REGION Network 51: TOUT Error TR
   RUNG wire#powerrail
      "FC911_CNT_Tiempo_UHS"(Temporizar := wire#w1, Valor_Tiempo := #V_TOut_TR, Base_tiempo_ms := 1, Valor_Actual := #TOUT_Movimiento_transfer, Tiempo_OK => #Tout_movimiento_transfer_q)
   END_RUNG
   RUNG wire#powerrail
      Contact( "DB1_SalidasExterioresDeMesa".Mesa[#Mesa].Ir_Pos_E2E4 )
      I_Contact( #PosTR_E2 )
   END_RUNG wire#w1
   RUNG wire#powerrail
      Contact( "DB1_SalidasExterioresDeMesa".Mesa[#Mesa].Ir_Pos_E1E3 )
      I_Contact( #PosTR_E1 )
   END_RUNG wire#w1
   // the same network as SCL:
   "FC911_CNT_Tiempo_UHS"(Temporizar := ("DB1_SalidasExterioresDeMesa".Mesa[#Mesa].Ir_Pos_E2E4 AND NOT #PosTR_E2) OR ("DB1_SalidasExterioresDeMesa".Mesa[#Mesa].Ir_Pos_E1E3 AND NOT #PosTR_E1),
                          Valor_Tiempo := #V_TOut_TR,
                          Base_tiempo_ms := 1,
                          Valor_Actual := #TOUT_Movimiento_transfer,
                          Tiempo_OK => #Tout_movimiento_transfer_q);
END_REGION

REGION Network 52: ERROR SUBIDA TR
   RUNG wire#powerrail
      Contact( #EstadoZona.Rearme_CBx )
      S_RS(operand := #EstadoVI.Err_TOut_Subida, s1 := wire#w1)
      S_Coil( #EstadoVI.Error_Mx )
   END_RUNG
   RUNG wire#powerrail
      Contact( #Tout_movimiento_transfer_q )
      Contact( "DB1_SalidasExterioresDeMesa".Mesa[#Mesa].Ir_Pos_E2E4 )
   END_RUNG wire#w1
   // the same network as SCL:
   IF #EstadoZona.Rearme_CBx THEN
       #EstadoVI.Err_TOut_Subida := FALSE;   // RS flip-flop
   END_IF;
   IF #Tout_movimiento_transfer_q AND "DB1_SalidasExterioresDeMesa".Mesa[#Mesa].Ir_Pos_E2E4 THEN
       #EstadoVI.Err_TOut_Subida := TRUE;
   END_IF;
   IF #EstadoVI.Err_TOut_Subida THEN #EstadoVI.Error_Mx := TRUE; END_IF;
END_REGION

REGION Network 53: ERROR BAJADA TR
   RUNG wire#powerrail
      Contact( #EstadoZona.Rearme_CBx )
      S_RS(operand := #EstadoVI.Err_TOut_Bajada, s1 := wire#w1)
      S_Coil( #EstadoVI.Error_Mx )
   END_RUNG
   RUNG wire#powerrail
      Contact( #Tout_movimiento_transfer_q )
      Contact( "DB1_SalidasExterioresDeMesa".Mesa[#Mesa].Ir_Pos_E1E3 )
   END_RUNG wire#w1
   // the same network as SCL:
   IF #EstadoZona.Rearme_CBx THEN
       #EstadoVI.Err_TOut_Bajada := FALSE;   // RS flip-flop
   END_IF;
   IF #Tout_movimiento_transfer_q AND "DB1_SalidasExterioresDeMesa".Mesa[#Mesa].Ir_Pos_E1E3 THEN
       #EstadoVI.Err_TOut_Bajada := TRUE;
   END_IF;
   IF #EstadoVI.Err_TOut_Bajada THEN #EstadoVI.Error_Mx := TRUE; END_IF;
END_REGION

REGION Network 54: TMP Error en Avance Tx
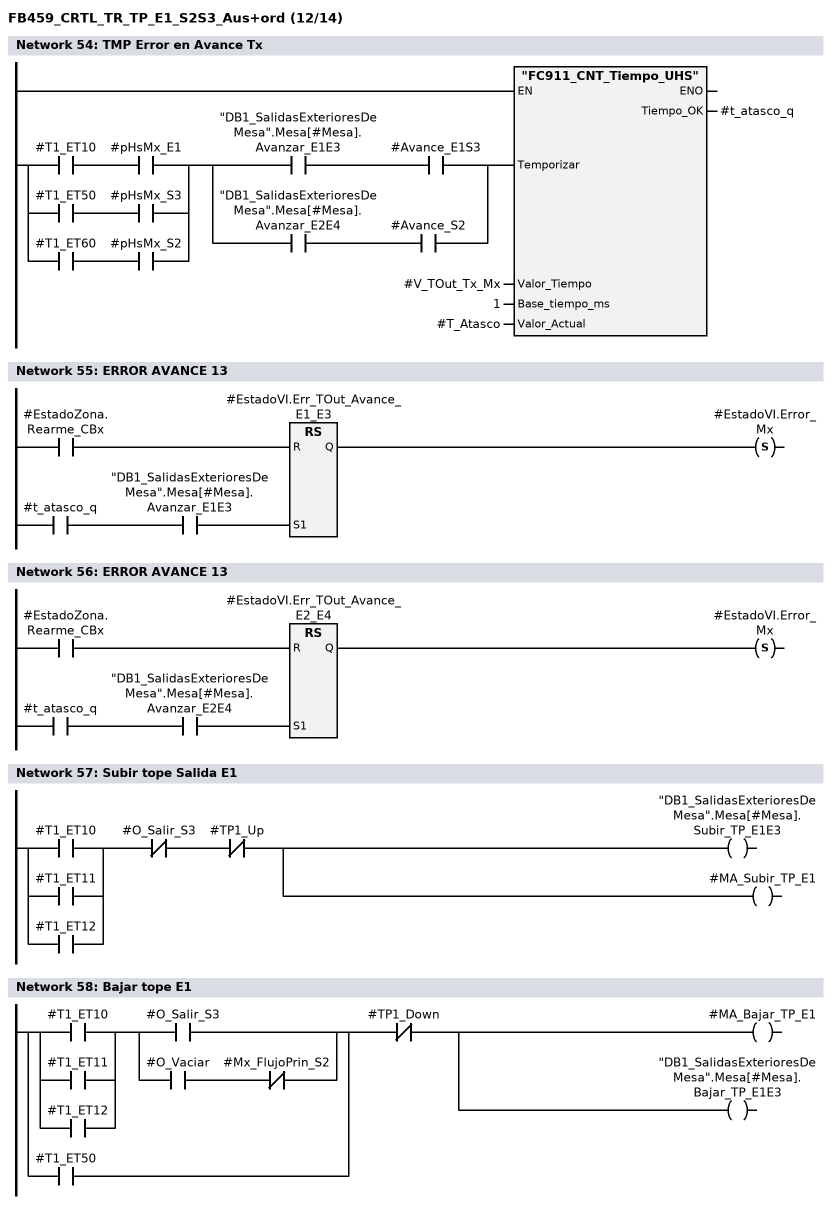
   RUNG wire#powerrail
      "FC911_CNT_Tiempo_UHS"(Temporizar := wire#w2, Valor_Tiempo := #V_TOut_Tx_Mx, Base_tiempo_ms := 1, Valor_Actual := #T_Atasco, Tiempo_OK => #t_atasco_q)
   END_RUNG
   RUNG wire#powerrail
      Contact( #T1_ET10 )
      Contact( #pHsMx_E1 )
      wire#w1
      Contact( "DB1_SalidasExterioresDeMesa".Mesa[#Mesa].Avanzar_E1E3 )
      Contact( #Avance_E1S3 )
   END_RUNG wire#w2
   RUNG wire#powerrail
      Contact( #T1_ET50 )
      Contact( #pHsMx_S3 )
   END_RUNG wire#w1
   RUNG wire#powerrail
      Contact( #T1_ET60 )
      Contact( #pHsMx_S2 )
   END_RUNG wire#w1
   RUNG wire#w1
      Contact( "DB1_SalidasExterioresDeMesa".Mesa[#Mesa].Avanzar_E2E4 )
      Contact( #Avance_S2 )
   END_RUNG wire#w2
   // the same network as SCL:
   "FC911_CNT_Tiempo_UHS"(Temporizar := ((#T1_ET10 AND #pHsMx_E1) OR (#T1_ET50 AND #pHsMx_S3) OR (#T1_ET60 AND #pHsMx_S2)) AND (("DB1_SalidasExterioresDeMesa".Mesa[#Mesa].Avanzar_E1E3 AND #Avance_E1S3) OR ("DB1_SalidasExterioresDeMesa".Mesa[#Mesa].Avanzar_E2E4 AND #Avance_S2)),
                          Valor_Tiempo := #V_TOut_Tx_Mx,
                          Base_tiempo_ms := 1,
                          Valor_Actual := #T_Atasco,
                          Tiempo_OK => #t_atasco_q);
END_REGION

REGION Network 55: ERROR AVANCE 13
   RUNG wire#powerrail
      Contact( #EstadoZona.Rearme_CBx )
      S_RS(operand := #EstadoVI.Err_TOut_Avance_E1_E3, s1 := wire#w1)
      S_Coil( #EstadoVI.Error_Mx )
   END_RUNG
   RUNG wire#powerrail
      Contact( #t_atasco_q )
      Contact( "DB1_SalidasExterioresDeMesa".Mesa[#Mesa].Avanzar_E1E3 )
   END_RUNG wire#w1
   // the same network as SCL:
   IF #EstadoZona.Rearme_CBx THEN
       #EstadoVI.Err_TOut_Avance_E1_E3 := FALSE;   // RS flip-flop
   END_IF;
   IF #t_atasco_q AND "DB1_SalidasExterioresDeMesa".Mesa[#Mesa].Avanzar_E1E3 THEN
       #EstadoVI.Err_TOut_Avance_E1_E3 := TRUE;
   END_IF;
   IF #EstadoVI.Err_TOut_Avance_E1_E3 THEN #EstadoVI.Error_Mx := TRUE; END_IF;
END_REGION

REGION Network 56: ERROR AVANCE 13
   RUNG wire#powerrail
      Contact( #EstadoZona.Rearme_CBx )
      S_RS(operand := #EstadoVI.Err_TOut_Avance_E2_E4, s1 := wire#w1)
      S_Coil( #EstadoVI.Error_Mx )
   END_RUNG
   RUNG wire#powerrail
      Contact( #t_atasco_q )
      Contact( "DB1_SalidasExterioresDeMesa".Mesa[#Mesa].Avanzar_E2E4 )
   END_RUNG wire#w1
   // the same network as SCL:
   IF #EstadoZona.Rearme_CBx THEN
       #EstadoVI.Err_TOut_Avance_E2_E4 := FALSE;   // RS flip-flop
   END_IF;
   IF #t_atasco_q AND "DB1_SalidasExterioresDeMesa".Mesa[#Mesa].Avanzar_E2E4 THEN
       #EstadoVI.Err_TOut_Avance_E2_E4 := TRUE;
   END_IF;
   IF #EstadoVI.Err_TOut_Avance_E2_E4 THEN #EstadoVI.Error_Mx := TRUE; END_IF;
END_REGION

REGION Network 57: Subir tope Salida E1
   RUNG wire#powerrail
      Contact( #T1_ET10 )
      wire#w1
      I_Contact( #O_Salir_S3 )
      I_Contact( #TP1_Up )
      wire#w2
      Coil( "DB1_SalidasExterioresDeMesa".Mesa[#Mesa].Subir_TP_E1E3 )
   END_RUNG
   RUNG wire#powerrail
      Contact( #T1_ET11 )
   END_RUNG wire#w1
   RUNG wire#powerrail
      Contact( #T1_ET12 )
   END_RUNG wire#w1
   RUNG wire#w2
      Coil( #MA_Subir_TP_E1 )
   END_RUNG
   // the same network as SCL:
   "DB1_SalidasExterioresDeMesa".Mesa[#Mesa].Subir_TP_E1E3 := (#T1_ET10 OR #T1_ET11 OR #T1_ET12) AND NOT #O_Salir_S3 AND NOT #TP1_Up;
   #MA_Subir_TP_E1 := (#T1_ET10 OR #T1_ET11 OR #T1_ET12) AND NOT #O_Salir_S3 AND NOT #TP1_Up;
END_REGION

REGION Network 58: Bajar tope E1
   RUNG wire#powerrail
      Contact( #T1_ET10 )
      wire#w1
      Contact( #O_Salir_S3 )
      wire#w2
      I_Contact( #TP1_Down )
      wire#w3
      Coil( #MA_Bajar_TP_E1 )
   END_RUNG
   RUNG wire#powerrail
      Contact( #T1_ET11 )
   END_RUNG wire#w1
   RUNG wire#powerrail
      Contact( #T1_ET12 )
   END_RUNG wire#w1
   RUNG wire#w1
      Contact( #O_Vaciar )
      I_Contact( #Mx_FlujoPrin_S2 )
   END_RUNG wire#w2
   RUNG wire#powerrail
      Contact( #T1_ET50 )
   END_RUNG wire#w2
   RUNG wire#w3
      Coil( "DB1_SalidasExterioresDeMesa".Mesa[#Mesa].Bajar_TP_E1E3 )
   END_RUNG
   // the same network as SCL:
   #MA_Bajar_TP_E1 := (((#T1_ET10 OR #T1_ET11 OR #T1_ET12) AND (#O_Salir_S3 OR (#O_Vaciar AND NOT #Mx_FlujoPrin_S2))) OR #T1_ET50) AND NOT #TP1_Down;
   "DB1_SalidasExterioresDeMesa".Mesa[#Mesa].Bajar_TP_E1E3 := #MA_Bajar_TP_E1;
END_REGION

REGION Network 59: timeout tope
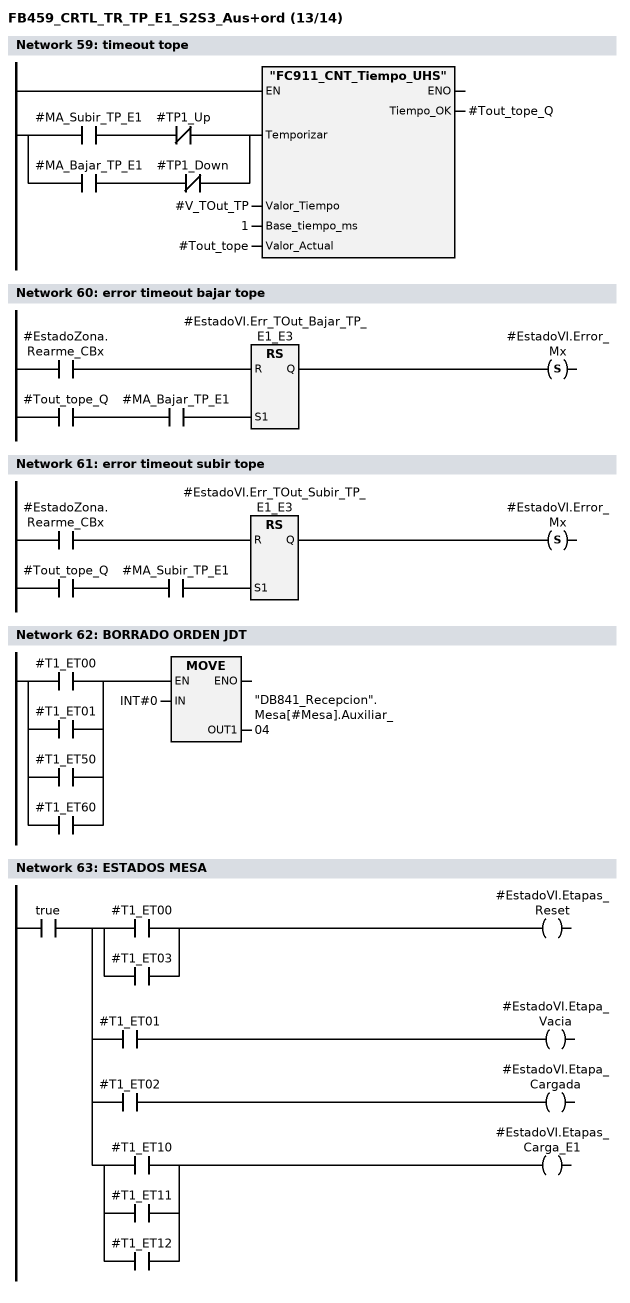
   RUNG wire#powerrail
      "FC911_CNT_Tiempo_UHS"(Temporizar := wire#w1, Valor_Tiempo := #V_TOut_TP, Base_tiempo_ms := 1, Valor_Actual := #Tout_tope, Tiempo_OK => #Tout_tope_Q)
   END_RUNG
   RUNG wire#powerrail
      Contact( #MA_Subir_TP_E1 )
      I_Contact( #TP1_Up )
   END_RUNG wire#w1
   RUNG wire#powerrail
      Contact( #MA_Bajar_TP_E1 )
      I_Contact( #TP1_Down )
   END_RUNG wire#w1
   // the same network as SCL:
   "FC911_CNT_Tiempo_UHS"(Temporizar := (#MA_Subir_TP_E1 AND NOT #TP1_Up) OR (#MA_Bajar_TP_E1 AND NOT #TP1_Down),
                          Valor_Tiempo := #V_TOut_TP,
                          Base_tiempo_ms := 1,
                          Valor_Actual := #Tout_tope,
                          Tiempo_OK => #Tout_tope_Q);
END_REGION

REGION Network 60: error timeout bajar tope
   RUNG wire#powerrail
      Contact( #EstadoZona.Rearme_CBx )
      S_RS(operand := #EstadoVI.Err_TOut_Bajar_TP_E1_E3, s1 := wire#w1)
      S_Coil( #EstadoVI.Error_Mx )
   END_RUNG
   RUNG wire#powerrail
      Contact( #Tout_tope_Q )
      Contact( #MA_Bajar_TP_E1 )
   END_RUNG wire#w1
   // the same network as SCL:
   IF #EstadoZona.Rearme_CBx THEN
       #EstadoVI.Err_TOut_Bajar_TP_E1_E3 := FALSE;   // RS flip-flop
   END_IF;
   IF #Tout_tope_Q AND #MA_Bajar_TP_E1 THEN #EstadoVI.Err_TOut_Bajar_TP_E1_E3 := TRUE; END_IF;
   IF #EstadoVI.Err_TOut_Bajar_TP_E1_E3 THEN #EstadoVI.Error_Mx := TRUE; END_IF;
END_REGION

REGION Network 61: error timeout subir tope
   RUNG wire#powerrail
      Contact( #EstadoZona.Rearme_CBx )
      S_RS(operand := #EstadoVI.Err_TOut_Subir_TP_E1_E3, s1 := wire#w1)
      S_Coil( #EstadoVI.Error_Mx )
   END_RUNG
   RUNG wire#powerrail
      Contact( #Tout_tope_Q )
      Contact( #MA_Subir_TP_E1 )
   END_RUNG wire#w1
   // the same network as SCL:
   IF #EstadoZona.Rearme_CBx THEN
       #EstadoVI.Err_TOut_Subir_TP_E1_E3 := FALSE;   // RS flip-flop
   END_IF;
   IF #Tout_tope_Q AND #MA_Subir_TP_E1 THEN #EstadoVI.Err_TOut_Subir_TP_E1_E3 := TRUE; END_IF;
   IF #EstadoVI.Err_TOut_Subir_TP_E1_E3 THEN #EstadoVI.Error_Mx := TRUE; END_IF;
END_REGION

REGION Network 62: BORRADO ORDEN JDT
   RUNG wire#powerrail
      Contact( #T1_ET00 )
      wire#w1
      { S7_GenerateENO := "TRUE" } Move(in := INT#0, out1 => "DB841_Recepcion".Mesa[#Mesa].Auxiliar_04)
   END_RUNG
   RUNG wire#powerrail
      Contact( #T1_ET01 )
   END_RUNG wire#w1
   RUNG wire#powerrail
      Contact( #T1_ET50 )
   END_RUNG wire#w1
   RUNG wire#powerrail
      Contact( #T1_ET60 )
   END_RUNG wire#w1
   // the same network as SCL:
   IF #T1_ET00 OR #T1_ET01 OR #T1_ET50 OR #T1_ET60 THEN
       "DB841_Recepcion".Mesa[#Mesa].Auxiliar_04 := INT#0;
   END_IF;
END_REGION

REGION Network 63: ESTADOS MESA
   RUNG wire#powerrail
      Contact( true )
      wire#w1
      Contact( #T1_ET00 )
      wire#w2
      Coil( #EstadoVI.Etapas_Reset )
   END_RUNG
   RUNG wire#w1
      Contact( #T1_ET03 )
   END_RUNG wire#w2
   RUNG wire#w1
      Contact( #T1_ET01 )
      Coil( #EstadoVI.Etapa_Vacia )
   END_RUNG
   RUNG wire#w1
      Contact( #T1_ET02 )
      Coil( #EstadoVI.Etapa_Cargada )
   END_RUNG
   RUNG wire#w1
      Contact( #T1_ET10 )
      wire#w3
      Coil( #EstadoVI.Etapas_Carga_E1 )
   END_RUNG
   RUNG wire#w1
      Contact( #T1_ET11 )
   END_RUNG wire#w3
   RUNG wire#w1
      Contact( #T1_ET12 )
   END_RUNG wire#w3
   // the same network as SCL:
   #EstadoVI.Etapas_Reset := true AND (#T1_ET00 OR #T1_ET03);
   #EstadoVI.Etapa_Vacia := true AND #T1_ET01;
   #EstadoVI.Etapa_Cargada := true AND #T1_ET02;
   #EstadoVI.Etapas_Carga_E1 := true AND (#T1_ET10 OR #T1_ET11 OR #T1_ET12);
END_REGION

REGION Network 64: Entradas Mesas
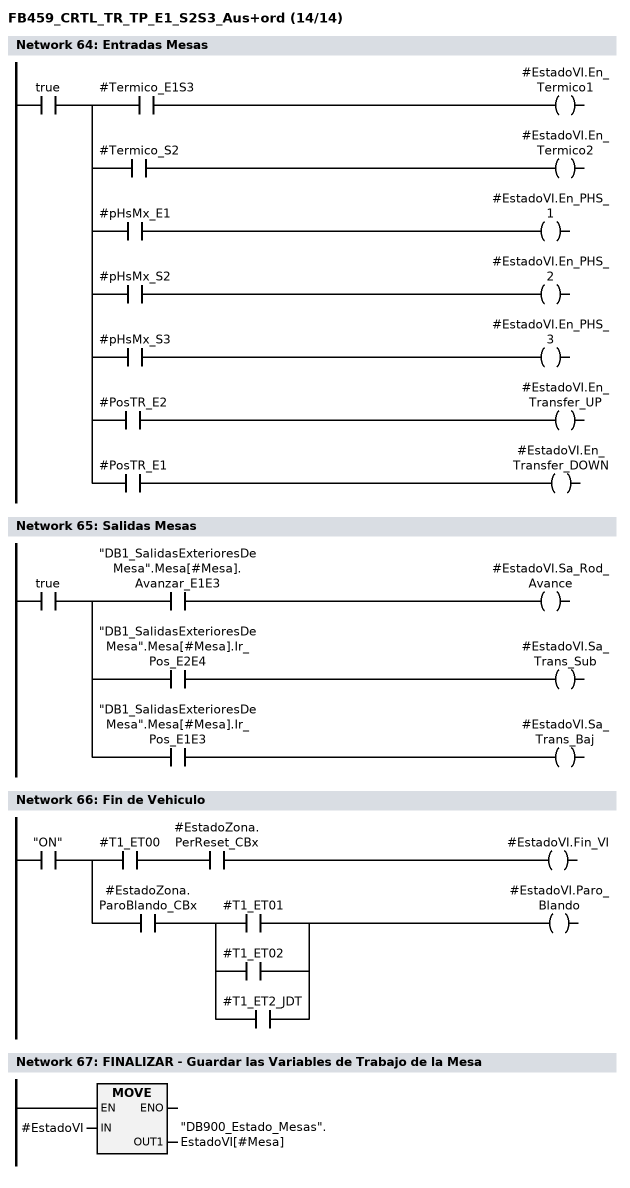
   RUNG wire#powerrail
      Contact( true )
      wire#w1
      Contact( #Termico_E1S3 )
      Coil( #EstadoVI.En_Termico1 )
   END_RUNG
   RUNG wire#w1
      Contact( #Termico_S2 )
      Coil( #EstadoVI.En_Termico2 )
   END_RUNG
   RUNG wire#w1
      Contact( #pHsMx_E1 )
      Coil( #EstadoVI.En_PHS_1 )
   END_RUNG
   RUNG wire#w1
      Contact( #pHsMx_S2 )
      Coil( #EstadoVI.En_PHS_2 )
   END_RUNG
   RUNG wire#w1
      Contact( #pHsMx_S3 )
      Coil( #EstadoVI.En_PHS_3 )
   END_RUNG
   RUNG wire#w1
      Contact( #PosTR_E2 )
      Coil( #EstadoVI.En_Transfer_UP )
   END_RUNG
   RUNG wire#w1
      Contact( #PosTR_E1 )
      Coil( #EstadoVI.En_Transfer_DOWN )
   END_RUNG
   // the same network as SCL:
   #EstadoVI.En_Termico1 := true AND #Termico_E1S3;
   #EstadoVI.En_Termico2 := true AND #Termico_S2;
   #EstadoVI.En_PHS_1 := true AND #pHsMx_E1;
   #EstadoVI.En_PHS_2 := true AND #pHsMx_S2;
   #EstadoVI.En_PHS_3 := true AND #pHsMx_S3;
   #EstadoVI.En_Transfer_UP := true AND #PosTR_E2;
   #EstadoVI.En_Transfer_DOWN := true AND #PosTR_E1;
END_REGION

REGION Network 65: Salidas Mesas
   RUNG wire#powerrail
      Contact( true )
      wire#w1
      Contact( "DB1_SalidasExterioresDeMesa".Mesa[#Mesa].Avanzar_E1E3 )
      Coil( #EstadoVI.Sa_Rod_Avance )
   END_RUNG
   RUNG wire#w1
      Contact( "DB1_SalidasExterioresDeMesa".Mesa[#Mesa].Ir_Pos_E2E4 )
      Coil( #EstadoVI.Sa_Trans_Sub )
   END_RUNG
   RUNG wire#w1
      Contact( "DB1_SalidasExterioresDeMesa".Mesa[#Mesa].Ir_Pos_E1E3 )
      Coil( #EstadoVI.Sa_Trans_Baj )
   END_RUNG
   // the same network as SCL:
   #EstadoVI.Sa_Rod_Avance := true AND "DB1_SalidasExterioresDeMesa".Mesa[#Mesa].Avanzar_E1E3;
   #EstadoVI.Sa_Trans_Sub := true AND "DB1_SalidasExterioresDeMesa".Mesa[#Mesa].Ir_Pos_E2E4;
   #EstadoVI.Sa_Trans_Baj := true AND "DB1_SalidasExterioresDeMesa".Mesa[#Mesa].Ir_Pos_E1E3;
END_REGION

REGION Network 66: Fin de Vehiculo
   RUNG wire#powerrail
      Contact( "ON" )
      wire#w1
      Contact( #T1_ET00 )
      Contact( #EstadoZona.PerReset_CBx )
      Coil( #EstadoVI.Fin_VI )
   END_RUNG
   RUNG wire#w1
      Contact( #EstadoZona.ParoBlando_CBx )
      wire#w2
      Contact( #T1_ET01 )
      wire#w3
      Coil( #EstadoVI.Paro_Blando )
   END_RUNG
   RUNG wire#w2
      Contact( #T1_ET02 )
   END_RUNG wire#w3
   RUNG wire#w2
      Contact( #T1_ET2_JDT )
   END_RUNG wire#w3
   // the same network as SCL:
   #EstadoVI.Fin_VI := "ON" AND #T1_ET00 AND #EstadoZona.PerReset_CBx;
   #EstadoVI.Paro_Blando := "ON" AND #EstadoZona.ParoBlando_CBx AND (#T1_ET01 OR #T1_ET02 OR #T1_ET2_JDT);
END_REGION

REGION Network 67: FINALIZAR - Guardar las Variables de Trabajo de la Mesa
   RUNG wire#powerrail
      Move(in := #EstadoVI, out1 => "DB900_Estado_Mesas".EstadoVI[#Mesa])
   END_RUNG
   // the same network as SCL:
   "DB900_Estado_Mesas".EstadoVI[#Mesa] := #EstadoVI;
END_REGION
END_FUNCTION_BLOCK

FUNCTION_BLOCK "FB45_Mesa_DesRemotador_Remontador_Horquilla"   // FB45, LAD
TITLE = FB120
{ S7_Optimized_Access := 'FALSE' }
AUTHOR : CRUCE
NAME : 20170410
VERSION : 4.0
// stored: AutoNumber false, SetENOAutomatically false
   VAR_INPUT
      Mesa : UInt;   // Mesa de la FB
      Error_Tx : Bool;   // Error en el Tx
      EnTension : Bool;   // Existe Tension en la Mesa
      Termico_E1_Tx : Bool;   // Proteccion del Tx en E1E3
      Termico_E2_Tx : Bool;   // Proteccion del Tx en E2E4
      pHsMx_1 : Bool;   // pHs de la Mesa
      pHsMx_2 : Bool;   // pHs de la Mesa
      pHsMx_Seg_1 : Bool;   // Seguridad de Centrado en la Mesa
      pHsMx_Seg_2 : Bool;   // Seguridad de Centrado en la Mesa
      pHsMx_PR1 : Bool;   // pHs de Protrusion de la Mesa. Nota: No existe >> ON
      pHsMx_PR2 : Bool;   // pHs de Protrusion de la Mesa. Nota: No existe >> ON
      pHsMx_PR3 : Bool;   // pHs de Protrusion de la Mesa. Nota: No existe >> ON
      pHsMx_PR4 : Bool;   // pHs de Protrusion de la Mesa. Nota: No existe >> ON
      Avance_E1_Tx_Ok : Bool;   // Avance del Tx en E1E3
      Avance_E2_Tx_Ok : Bool;   // Avance del Tx en E2E4
      PosTR_E1 : Bool;   // Posicion del TR en E1E3
      PosTR_E2 : Bool;   // Posicion del TR en E2E4
      EnMovimiento_TR : Bool;   // En movimiento el TR
      TP1_UP : Bool;   // TP1 Arriba. Nota Movimiento E1 >> S3
      TP1_DW : Bool;   // TP1 Abajo. Nota Movimiento E1 >> S3
      EnMovimiento_TP1 { ExternalVisible := 'False'} : Bool;   // En movimiento el TP1
      TP2_UP : Bool;   // TP2 Arriba. Nota Movimiento E2 >> S4
      TP2_DW : Bool;   // TP2 Abajo. Nota Movimiento E2 >> S4
      EnMovimiento_TP2 : Bool;   // En movimiento el TP2
      DescargaAct_Ent_M1 : Bool;   // E1 >> Mesa Anterior DescargaAct
      AVTF_Ent_M1 : Bool;   // E1 >> Mesa Anterior AVTF
      P_Mens_Ent_M1 { ExternalWritable := 'False'} : Bool;   // E1 >> Mesa Anterior P_Mens
      DescargaAct_Ent_M2 : Bool;   // E2 >> Mesa Anterior DescargaAct
      AVTF_Ent_M2 : Bool;   // E2 >> Mesa Anterior AVTF
      P_Mens_Ent_M2 : Bool;   // E2 >> Mesa Anterior P_Mens
      DescargaAct_Ent_M3 : Bool;   // E3 >> Mesa Anterior DescargaAct
      AVTF_Ent_M3 : Bool;   // E3 >> Mesa Anterior AVTF
      P_Mens_Ent_M3 : Bool;   // E3 >> Mesa Anterior P_Mens
      DescargaAct_Ent_M4 : Bool;   // E4 >> Mesa Anterior DescargaAct
      AVTF_Ent_M4 : Bool;   // E4 >> Mesa Anterior AVTF
      P_Mens_Ent_M4 : Bool;   // E4 >> Mesa Anterior P_Mens
      PTF_Sal_M1 : Bool;   // S1 >> Mesa Siguiente PTF
      FTF_Sal_M1 : Bool;   // S1 >> Mesa Siguiente FTF
      PTF_Sal_M2 : Bool;   // S2 >> Mesa Siguiente PTF
      FTF_Sal_M2 : Bool;   // S2 >> Mesa Siguiente FTF
      PTF_Sal_M3 : Bool;   // S3 >> Mesa Siguiente PTF
      FTF_Sal_M3 : Bool;   // S3 >> Mesa Siguiente FTF
      PTF_Sal_M4 : Bool;   // S4 >> Mesa Siguiente PTF
      FTF_Sal_M4 : Bool;   // S4 >> Mesa Siguiente FTF
      MSig_CargaAct_Sal_M1 : Bool;   // S1 >> Mesa Siguiente En Carga
      MSig_CargaAct_Sal_M2 : Bool;   // S2 >> Mesa Siguiente En Carga
      MSig_CargaAct_Sal_M3 : Bool;   // S3 >> Mesa Siguiente En Carga
      MSig_CargaAct_Sal_M4 : Bool;   // S4 >> Mesa Siguiente En Carga
      Mx_TRElectrico : Bool;   // Config >> TR Arriba en E1E3
      Mx_UP_E1E3 : Bool;   // Config >> Mesa con Transfer Electrico
      Mx_TP1_Central : Bool;   // Config >> TP1 Es Taco Central
      Mx_TP2_Central : Bool;   // Config >> TP2 Es Taco Central
      Mx_PospHs1_12 : Bool;   // Config >> Está la phs1 entre E1 y E2? ON-OFF
      Mx_PospHs1_23 : Bool;   // Config >> Está la phs1 entre E2 y E3? ON-OFF
      Mx_PospHs1_34 : Bool;   // Config >> Está la phs1 entre E3 y E4? ON-OFF
      Mx_PospHs1_41 : Bool;   // Config >> Está la phs1 entre E4 y E1? ON-OFF
      PosTR_EnReposo_E2 : Bool;   // Posicion de Reposo en E2 para el Transfer
      PosTR_EnReposo_E1 : Bool;   // Posicion de Reposo en E1 para el Transfer
      PermisoMov_PosTR_E2 : Bool;   // Permiso de Mover el Trasnfer hacia E2
      PermisoMov_PosTR_E1 : Bool;   // Permiso de Mover el Trasnfer hacia E1
      Mx_ApiladorDesAplilador : Bool;   // Config >> Apilador / DesApilador
      Mx_RH_PosTR_E1 : Bool := TRUE;   // Config >> Posicion E1E3 para RH
      Mx_RH_PosTR_E2 : Bool;   // Config >> Posicion E2E4 para RH
      RH_Quieto : Bool;   // Interlock >> Quieto
      RH_FinMovimiento : Bool;   // Interlock >> Fin del Movimiento
      Mx_VelocidadLenta_In : Bool;   // Forzar a Velociada Lenta
      F_EnvMens_Mx : Bool;   // Fin de Envio de Mensaje
      OrdSal_DesRemontar : Bool;   // Orden de Salida Con DesRemontado
      OrdSal_M1 : Bool;   // Orden de Salida por S1
      OrdSal_M2 : Bool;   // Orden de Salida por S2
      OrdSal_M3 : Bool;   // Orden de Salida por S3
      OrdSal_M4 : Bool;   // Orden de Salida por S4
      BloqueoActivo_OK : Bool;   // Bloqueo Activo de la Mesa
      V_CNT_pHsMx_E1 : Int := 400;   // Valor de Presencia
      V_CNT_pHsMx_FTF_E1 : Int := 200;   // Valor para activar FTF. Nota: < = V_CNT_pHsMx.
      V_CNTSeg_pHsMx_E1 : Int := 2000;   // Valor de Seguriadad para Presencia
      V_CNT_pHsMx_E2 : Int := 400;   // Valor de Presencia
      V_CNT_pHsMx_FTF_E2 : Int := 200;   // Valor para activar FTF. Nota: < = V_CNT_pHsMx.
      V_CNTSeg_pHsMx_E2 : Int := 2000;   // Valor de Seguriadad para Presencia
      V_Subir_TP_Min : Int := 20;   // Valor Minimo para Subir Tope
      V_Bajar_TP_Max : Int := 40;   // Valor Maximo para Bajar Tope
      V_CNT_ApHsMx : Int := 500;   // Valor de Ausencia
      V_CNTSeg_ApHsMx : Int := 2000;   // Valor de Seguriadad para Ausencia
      V_TIM_Bloqueo : Int := 30000;   // Valor del Tiempo de Espera para Bloqueo
      V_CNT_Simultaneo : Int := 2000;   // Valor de Simultaneo
      V_InicioSimultaneo : Int := 0;   // Inicio de Simultaneo. Nota: <= V_CNT_Simultaneo
      V_FinSimultaneo : Int := 0;   // Final de Simultaneo. Nota: <= V_InicioSimultaneo
      V_TOut_Tx_Mx_E1 : Int := 10000;   // TimeOut de Entrada por E1
      V_TOut_Tx_Mx_E2 : Int := 10000;   // TimeOut de Entrada por E2
      V_TOut_TR : Int := 5000;   // TimeOut de Transfer
      V_TOut_TP : Int := 5000;   // TimeOut de Tope
      V_TMP_Protrusion : Int := 200;   // TMP de Protrusion
      V_CNT_PerdidapHs : Int := 1000;   // CNT de Perdida de pHs
      V_ApHs_CNTSeg_E1 : Int := 200;   // Valor de Ausencia pHsSeg del CNTSeg
      V_ApHs_CNTSeg_E2 : Int := 200;   // Valor de Ausencia pHsSeg del CNTSeg
      V_RecolocaCarga : Int := 500;   // Valor de Recoloca Carga >> Remontado
   END_VAR
   VAR_OUTPUT
      P_EnvMens_PMx : Bool;   // Permiso de Enviar Mensaje de Presencia
      P_EnvMens_PBM : Bool;   // Permiso de Enviar Mensaje de Bloqueo
      P_RecepOK_Mx : Bool;   // Recepcion OK
      PTF_Ent_M1 : Bool;   // E1 >> Mesa Anterior PTF
      FTF_Ent_M1 : Bool;   // E1 >> Mesa Anterior FTF
      PTF_Ent_M2 : Bool;   // E2 >> Mesa Anterior PTF
      FTF_Ent_M2 : Bool;   // E2 >> Mesa Anterior FTF
      PTF_Ent_M3 : Bool;   // E3 >> Mesa Anterior PTF
      FTF_Ent_M3 : Bool;   // E3 >> Mesa Anterior FTF
      PTF_Ent_M4 : Bool;   // E4 >> Mesa Anterior PTF
      FTF_Ent_M4 : Bool;   // E4 >> Mesa Anterior FTF
      AVTF_Sal_M1 : Bool;   // S1 >> Mesa Siguiente AVTF
      P_Mens_Sal_M1 : Bool;   // S1 >> Mesa Siguiente P_Mens
      AVTF_Sal_M2 : Bool;   // S2 >> Mesa Siguiente AVTF
      P_Mens_Sal_M2 : Bool;   // S2 >> Mesa Siguiente P_Mens
      AVTF_Sal_M3 : Bool;   // S3 >> Mesa Siguiente AVTF
      P_Mens_Sal_M3 : Bool;   // S3 >> Mesa Siguiente P_Mens
      AVTF_Sal_M4 : Bool;   // S4 >> Mesa Siguiente AVTF
      P_Mens_Sal_M4 : Bool;   // S4 >> Mesa Siguiente P_Mens
      RH_PasarReposo : Bool;   // Interlock >> Pasar a Reposo
      RH_SubirPaleta : Bool;   // Interlock >> Subir Paleta
      RH_DejarPaleta : Bool;   // Interlock >> Dejar Paleta
      RH_RemontarPaleta : Bool;   // Interlock >> Remontar Paleta
      RH_DesRemontarPaleta : Bool;   // Interlock >> DesRemontar Paleta
   END_VAR
   VAR
      Activar_VarpHsSeg : Bool;
      Anular_PR1 : Bool;   // ???
      Anular_PR2 : Bool;   // ???
      Anular_PR3 : Bool;   // ???
      Anular_PR4 : Bool;   // ???
      Mx_ET00 : Bool;
      Mx_ET01 : Bool;
      Mx_ET02 : Bool;
      Mx_ET08 : Bool;
      Mx_ET09 : Bool;
      Mx_ET10 : Bool;
      Mx_ET11 : Bool;
      Mx_ET12 : Bool;
      Mx_ET110 : Bool;
      Mx_ET111 : Bool;
      Mx_ET50 : Bool;
      Mx_ET51 : Bool;
      Mx_ET150 : Bool;
      Mx_ET151 : Bool;
      Mx_ET20 : Bool;
      Mx_ET21 : Bool;
      Mx_ET22 : Bool;
      Mx_ET120 : Bool;
      Mx_ET121 : Bool;
      Mx_ET60 : Bool;
      Mx_ET61 : Bool;
      Mx_ET160 : Bool;
      Mx_ET161 : Bool;
      Mx_ET180 : Bool;
      MemoRemontando : Bool;   // Interna >> Realizando Remontado
      Mx_ET80 : Bool;
      Mx_ET81 : Bool;
      Mx_ET85 : Bool;
      Mx_ET86 : Bool;
      MemoDesRemontando : Bool;   // Interna >> Realizando DesRemontado
      Mx_ET90 : Bool;
      Mx_ET91 : Bool;
      Mx_ET95 : Bool;
      Mx_ET96 : Bool;
      Mx_ET181 : Bool;
      Selec_M1_Entrada : Bool;   // Seleccionado Entrada por E1
      Selec_M2_Entrada : Bool;   // Seleccionado Entrada por E2
      Selec_M3_Entrada : Bool;   // Seleccionado Entrada por E3
      Selec_M4_Entrada : Bool;   // Seleccionado Entrada por E4
      Selec_M1_Salida : Bool;   // Seleccionado Salida por S1
      Selec_M2_Salida : Bool;   // Seleccionado Salida por S2
      Selec_M3_Salida : Bool;   // Seleccionado Salida por S3
      Selec_M4_Salida : Bool;   // Seleccionado Salida por S4
      MEnt_DescargaAct : Bool;   // Interlock >> DesCargaAct de MAnt >> Mx
      AVTF_MEnt : Bool;   // Interlock >> AVTF de MAnt >> Mx
      P_Mens_MEnt : Bool;   // Interlock >> P_Mens de MAnt >> Mx
      PTF_MEnt : Bool;   // Interlock >> PTF de MAnt >> Mx
      FTF_MEnt : Bool;   // Interlock >> FTF de MAnt >> Mx
      AVTF_MSal : Bool;   // Interlock >> AVTF de Mx >> MSig
      P_Mens_MSal : Bool;   // Interlock >> P_Mens de Mx >> MSig
      PTF_MSal : Bool;   // Interlock >> PTF de Mx >> MSig
      FTF_MSal : Bool;   // Interlock >> FTF de Mx >> MSig
      ProtocoloIniciado_Mx : Bool;   // Iniciado el Envio del Mensaje de Presencia
      Simultaneo_Mx : Bool;   // Activo Simultaneo E1E2E3E4
      SaliendoCarga : Bool;   // Saliendo Carga de la Mesa
      VAR_pHsSeg : Bool;   // Interlock >> pHs de Seguridad, Inicio
      VAR_pHs : Bool;   // Interlock >> pHs de Posicionado
      Pos_TR_OK : Bool;   // Posicion Correcta del TR
      CNT_pHsMx_FTF_OK_E1E3 : Bool;   // Enviar ya FTF
      CNT_pHsMx_FTF_OK_E2E4 : Bool;   // Enviar ya FTF
      STAT_EnvMens_PMx : Bool;   // Interna >> Envio del Mensaje de Presencia
      STAT_EnvMens_PBMx : Bool;   // Interna >> Envio del Mensaje de Bloqueo
      CNT_RecolocaCarga { S7_SetPoint := 'True'} : "FB910_CNT_UHS";   // CNT de la Presencia
      CNT_pHsMx_E1E3 { S7_SetPoint := 'True'} : "FB910_CNT_UHS";   // CNT de la Presencia
      CNTSeg_pHsMx_E1E3 { S7_SetPoint := 'True'} : "FB910_CNT_UHS";   // CNT de Seguridad de la Presencia
      CNT_pHsMx_E2E4 { S7_SetPoint := 'True'} : "FB910_CNT_UHS";   // CNT de la Presencia
      CNTSeg_pHsMx_E2E4 { S7_SetPoint := 'True'} : "FB910_CNT_UHS";   // CNT de Seguridad de la Presencia
      CNT_ApHsMx { S7_SetPoint := 'True'} : "FB910_CNT_UHS";   // CNT de la Ausencia
      CNTSeg_ApHsMx { S7_SetPoint := 'True'} : "FB910_CNT_UHS";   // CNT de Seguridad de la Ausencia
      TIM_Bloqueo { S7_SetPoint := 'True'} : "FB910_CNT_UHS";   // TIM de Espera para Bloqueo
      CNT_Simultaneo { S7_SetPoint := 'True'} : "FB910_CNT_UHS";   // CNT de Simultaneo
      TMP_EnTension { S7_SetPoint := 'True'} : "FB910_CNT_UHS";
      TOut_Av_Mx_E1E3 { S7_SetPoint := 'True'} : "FB910_CNT_UHS";   // Time Out de Entrada de E1
      TOut_Ret_Mx_E1E3 { S7_SetPoint := 'True'} : "FB910_CNT_UHS";   // Time Out de Entrada de E3
      TOut_Av_Mx_E2E4 { S7_SetPoint := 'True'} : "FB910_CNT_UHS";   // Time Out de Entrada de E2
      TOut_Ret_Mx_E2E4 { S7_SetPoint := 'True'} : "FB910_CNT_UHS";   // Time Out de Entrada de E4
      TOut_Subir_TR { S7_SetPoint := 'True'} : "FB910_CNT_UHS";   // Time Out de Subida del TR
      TOut_Bajar_TR { S7_SetPoint := 'True'} : "FB910_CNT_UHS";   // Time Out de Bajada del TR
      TOut_Subir_TP { S7_SetPoint := 'True'} : "FB910_CNT_UHS";   // Time Out de Subida del TP
      TOut_Bajar_TP { ExternalAccessible := 'False'; ExternalVisible := 'False'; ExternalWritable := 'False'; S7_SetPoint := 'True'} : "FB910_CNT_UHS";   // Time Out de Bajada del TP
      TMP_Protrusion { S7_SetPoint := 'True'} : "FB910_CNT_UHS";   // TMP de la Protrusion
      CNT_PerdidapHs { S7_SetPoint := 'True'} : "FB910_CNT_UHS";   // CNT de Perdida de pHs
      CNTApHs_CNTSeg_E2E4 { S7_SetPoint := 'True'} : "FB910_CNT_UHS";   // CNT de Ausnecia para CNTSeg
      CNTApHs_CNTSeg_E1E3 { S7_SetPoint := 'True'} : "FB910_CNT_UHS";   // CNT de Ausnecia para CNTSeg
   END_VAR
   VAR_TEMP
      EstadoZona : "EstadoZona";   // Estado de Zona de la Mesa
      EstadoVI : "EstadosMesa";   // Estado del Vehiculo Inteliguente de la Mesa
      ConfigFB : "UDT_ConfigFB";   // Configuracion de la FB de la Mesa
      V_Protrusion : Int;
      Aux_ET00 : Bool;
      OK_TP1_DW : Bool;
      OK_TP2_DW : Bool;
      InicialesEntrada : Bool;
      PasoEntrada : Bool;
      InicialesSalida : Bool;
      PasoSalida : Bool;
      Remontando : Bool;
      DesRemontando : Bool;
   END_VAR
   VAR_TEMP   // added for the SCL form of the ladder/FBD networks
      _w1 : Bool;
      _w2 : Bool;
      _w3 : Bool;
      _w4 : Bool;
   END_VAR
BEGIN

REGION Network 1: INCIALIZAR - Variables Especiales
END_REGION

REGION Network 2: INICIALIZAR - Recoger las Variables de Estado de la Mesa
   // Se recoge - Estado_CBx
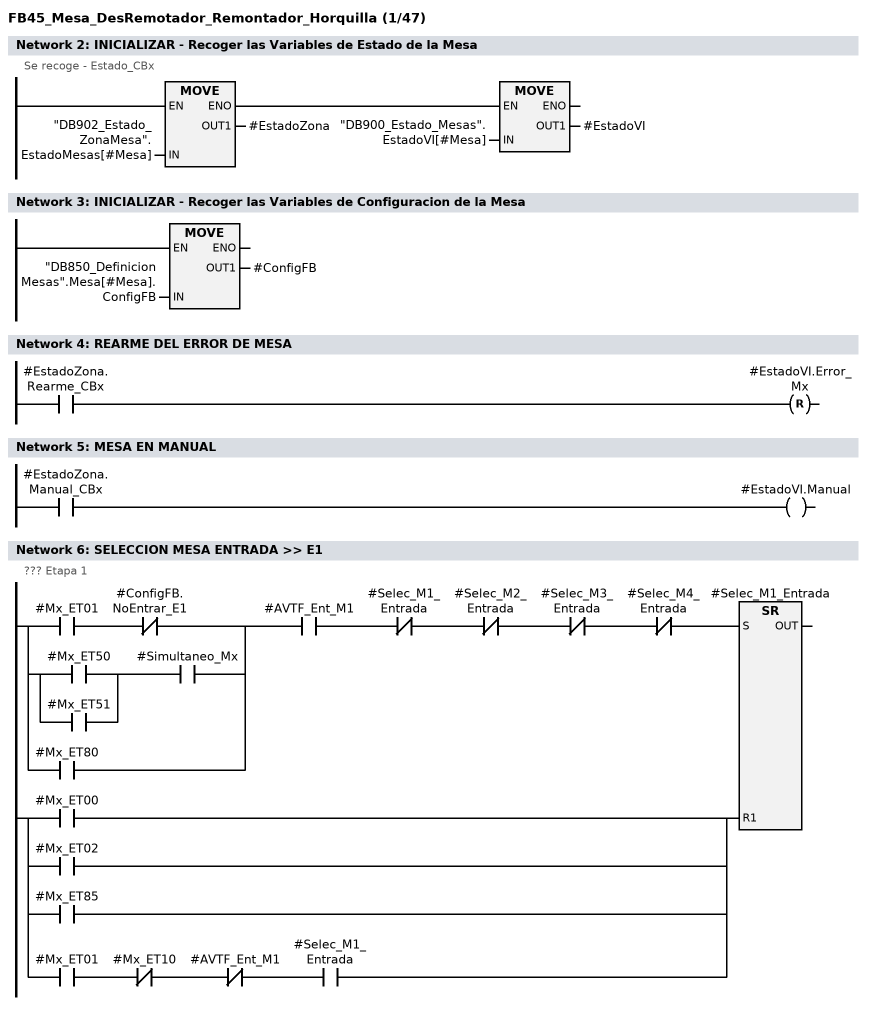
   RUNG wire#powerrail
      Move(in := "DB902_Estado_ZonaMesa".EstadoMesas[#Mesa], out1 => #EstadoZona)
      Move(in := "DB900_Estado_Mesas".EstadoVI[#Mesa], out1 => #EstadoVI)
   END_RUNG
   // the same network as SCL:
   #EstadoZona := "DB902_Estado_ZonaMesa".EstadoMesas[#Mesa];
   #EstadoVI := "DB900_Estado_Mesas".EstadoVI[#Mesa];
END_REGION

REGION Network 3: INICIALIZAR - Recoger las Variables de Configuracion de la Mesa
   RUNG wire#powerrail
      Move(in := "DB850_DefinicionMesas".Mesa[#Mesa].ConfigFB, out1 => #ConfigFB)
   END_RUNG
   // the same network as SCL:
   #ConfigFB := "DB850_DefinicionMesas".Mesa[#Mesa].ConfigFB;
END_REGION

REGION Network 4: REARME DEL ERROR DE MESA
   RUNG wire#powerrail
      Contact( #EstadoZona.Rearme_CBx )
      R_Coil( #EstadoVI.Error_Mx )
   END_RUNG
   // the same network as SCL:
   IF #EstadoZona.Rearme_CBx THEN #EstadoVI.Error_Mx := FALSE; END_IF;
END_REGION

REGION Network 5: MESA EN MANUAL
   RUNG wire#powerrail
      Contact( #EstadoZona.Manual_CBx )
      Coil( #EstadoVI.Manual )
   END_RUNG
   // the same network as SCL:
   #EstadoVI.Manual := #EstadoZona.Manual_CBx;
END_REGION

REGION Network 6: SELECCION MESA ENTRADA >> E1
   // ??? Etapa 1
   RUNG wire#powerrail
      Contact( #Mx_ET01 )
      I_Contact( #ConfigFB.NoEntrar_E1 )
      wire#w1
      Contact( #AVTF_Ent_M1 )
      I_Contact( #Selec_M1_Entrada )
      I_Contact( #Selec_M2_Entrada )
      I_Contact( #Selec_M3_Entrada )
      I_Contact( #Selec_M4_Entrada )
      S_SR(operand := #Selec_M1_Entrada, r1 := wire#w3)
   END_RUNG
   RUNG wire#powerrail
      Contact( #Mx_ET50 )
      wire#w2
      Contact( #Simultaneo_Mx )
   END_RUNG wire#w1
   RUNG wire#powerrail
      Contact( #Mx_ET51 )
   END_RUNG wire#w2
   RUNG wire#powerrail
      Contact( #Mx_ET80 )
   END_RUNG wire#w1
   RUNG wire#powerrail
      Contact( #Mx_ET00 )
   END_RUNG wire#w3
   RUNG wire#powerrail
      Contact( #Mx_ET02 )
   END_RUNG wire#w3
   RUNG wire#powerrail
      Contact( #Mx_ET85 )
   END_RUNG wire#w3
   RUNG wire#powerrail
      Contact( #Mx_ET01 )
      I_Contact( #Mx_ET10 )
      I_Contact( #AVTF_Ent_M1 )
      Contact( #Selec_M1_Entrada )
   END_RUNG wire#w3
   // the same network as SCL:
   #_w1 := #Mx_ET00 OR #Mx_ET02 OR #Mx_ET85 OR (#Mx_ET01 AND NOT #Mx_ET10 AND NOT #AVTF_Ent_M1 AND #Selec_M1_Entrada);
   IF ((#Mx_ET01 AND NOT #ConfigFB.NoEntrar_E1) OR ((#Mx_ET50 OR #Mx_ET51) AND #Simultaneo_Mx) OR #Mx_ET80) AND #AVTF_Ent_M1 AND NOT #Selec_M1_Entrada AND NOT #Selec_M2_Entrada AND NOT #Selec_M3_Entrada AND NOT #Selec_M4_Entrada THEN
       #Selec_M1_Entrada := TRUE;   // SR flip-flop
   END_IF;
   IF #_w1 THEN #Selec_M1_Entrada := FALSE; END_IF;
END_REGION

REGION Network 7: SELECCION MESA ENTRADA >> E2
   // ??? Etapa 1
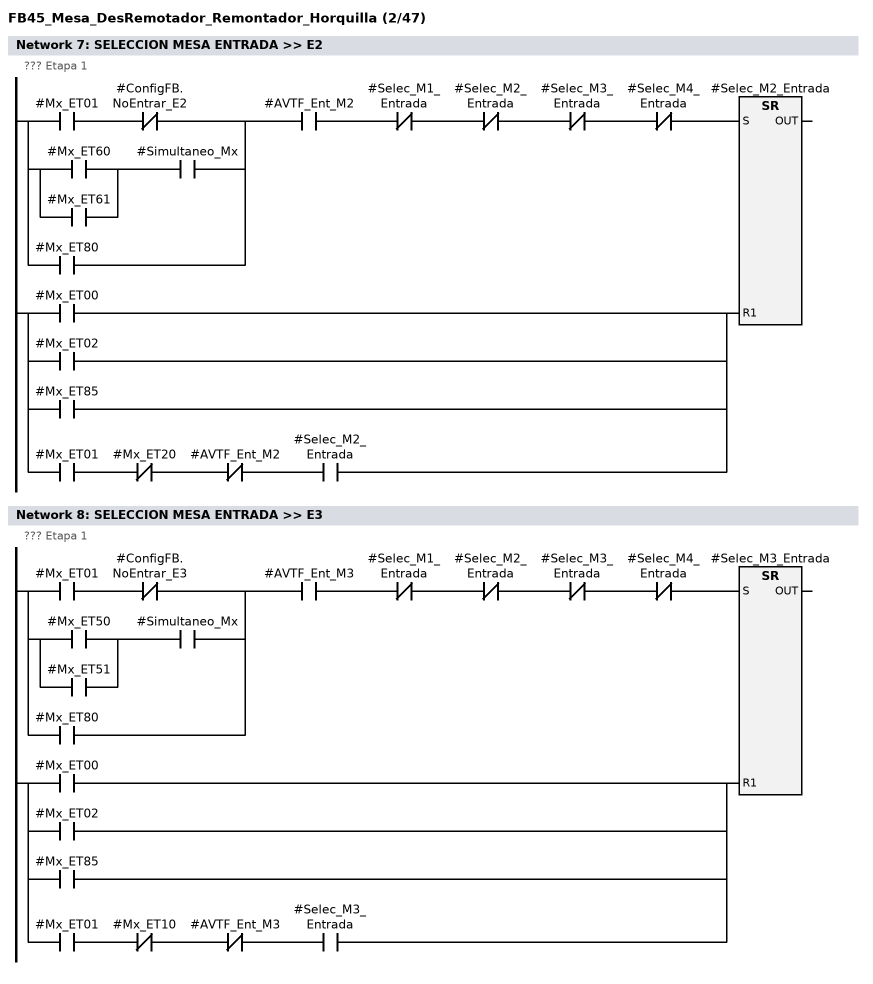
   RUNG wire#powerrail
      Contact( #Mx_ET01 )
      I_Contact( #ConfigFB.NoEntrar_E2 )
      wire#w1
      Contact( #AVTF_Ent_M2 )
      I_Contact( #Selec_M1_Entrada )
      I_Contact( #Selec_M2_Entrada )
      I_Contact( #Selec_M3_Entrada )
      I_Contact( #Selec_M4_Entrada )
      S_SR(operand := #Selec_M2_Entrada, r1 := wire#w3)
   END_RUNG
   RUNG wire#powerrail
      Contact( #Mx_ET60 )
      wire#w2
      Contact( #Simultaneo_Mx )
   END_RUNG wire#w1
   RUNG wire#powerrail
      Contact( #Mx_ET61 )
   END_RUNG wire#w2
   RUNG wire#powerrail
      Contact( #Mx_ET80 )
   END_RUNG wire#w1
   RUNG wire#powerrail
      Contact( #Mx_ET00 )
   END_RUNG wire#w3
   RUNG wire#powerrail
      Contact( #Mx_ET02 )
   END_RUNG wire#w3
   RUNG wire#powerrail
      Contact( #Mx_ET85 )
   END_RUNG wire#w3
   RUNG wire#powerrail
      Contact( #Mx_ET01 )
      I_Contact( #Mx_ET20 )
      I_Contact( #AVTF_Ent_M2 )
      Contact( #Selec_M2_Entrada )
   END_RUNG wire#w3
   // the same network as SCL:
   #_w1 := #Mx_ET00 OR #Mx_ET02 OR #Mx_ET85 OR (#Mx_ET01 AND NOT #Mx_ET20 AND NOT #AVTF_Ent_M2 AND #Selec_M2_Entrada);
   IF ((#Mx_ET01 AND NOT #ConfigFB.NoEntrar_E2) OR ((#Mx_ET60 OR #Mx_ET61) AND #Simultaneo_Mx) OR #Mx_ET80) AND #AVTF_Ent_M2 AND NOT #Selec_M1_Entrada AND NOT #Selec_M2_Entrada AND NOT #Selec_M3_Entrada AND NOT #Selec_M4_Entrada THEN
       #Selec_M2_Entrada := TRUE;   // SR flip-flop
   END_IF;
   IF #_w1 THEN #Selec_M2_Entrada := FALSE; END_IF;
END_REGION

REGION Network 8: SELECCION MESA ENTRADA >> E3
   // ??? Etapa 1
   RUNG wire#powerrail
      Contact( #Mx_ET01 )
      I_Contact( #ConfigFB.NoEntrar_E3 )
      wire#w1
      Contact( #AVTF_Ent_M3 )
      I_Contact( #Selec_M1_Entrada )
      I_Contact( #Selec_M2_Entrada )
      I_Contact( #Selec_M3_Entrada )
      I_Contact( #Selec_M4_Entrada )
      S_SR(operand := #Selec_M3_Entrada, r1 := wire#w3)
   END_RUNG
   RUNG wire#powerrail
      Contact( #Mx_ET50 )
      wire#w2
      Contact( #Simultaneo_Mx )
   END_RUNG wire#w1
   RUNG wire#powerrail
      Contact( #Mx_ET51 )
   END_RUNG wire#w2
   RUNG wire#powerrail
      Contact( #Mx_ET80 )
   END_RUNG wire#w1
   RUNG wire#powerrail
      Contact( #Mx_ET00 )
   END_RUNG wire#w3
   RUNG wire#powerrail
      Contact( #Mx_ET02 )
   END_RUNG wire#w3
   RUNG wire#powerrail
      Contact( #Mx_ET85 )
   END_RUNG wire#w3
   RUNG wire#powerrail
      Contact( #Mx_ET01 )
      I_Contact( #Mx_ET10 )
      I_Contact( #AVTF_Ent_M3 )
      Contact( #Selec_M3_Entrada )
   END_RUNG wire#w3
   // the same network as SCL:
   #_w1 := #Mx_ET00 OR #Mx_ET02 OR #Mx_ET85 OR (#Mx_ET01 AND NOT #Mx_ET10 AND NOT #AVTF_Ent_M3 AND #Selec_M3_Entrada);
   IF ((#Mx_ET01 AND NOT #ConfigFB.NoEntrar_E3) OR ((#Mx_ET50 OR #Mx_ET51) AND #Simultaneo_Mx) OR #Mx_ET80) AND #AVTF_Ent_M3 AND NOT #Selec_M1_Entrada AND NOT #Selec_M2_Entrada AND NOT #Selec_M3_Entrada AND NOT #Selec_M4_Entrada THEN
       #Selec_M3_Entrada := TRUE;   // SR flip-flop
   END_IF;
   IF #_w1 THEN #Selec_M3_Entrada := FALSE; END_IF;
END_REGION

REGION Network 9: SELECCION MESA ENTRADA >> E4
   // ??? Etapa 1
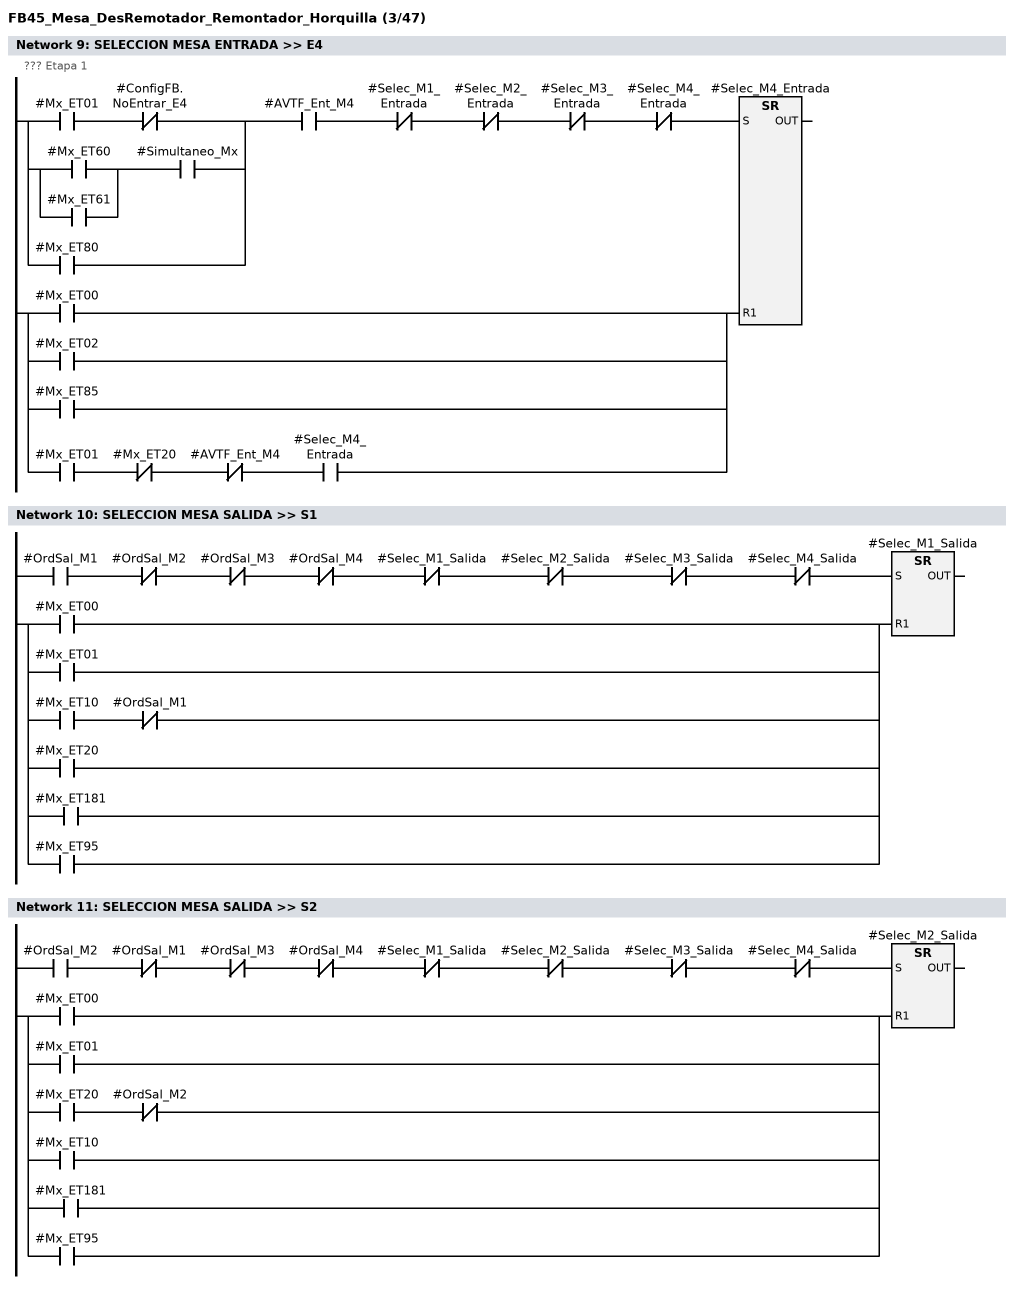
   RUNG wire#powerrail
      Contact( #Mx_ET01 )
      I_Contact( #ConfigFB.NoEntrar_E4 )
      wire#w1
      Contact( #AVTF_Ent_M4 )
      I_Contact( #Selec_M1_Entrada )
      I_Contact( #Selec_M2_Entrada )
      I_Contact( #Selec_M3_Entrada )
      I_Contact( #Selec_M4_Entrada )
      S_SR(operand := #Selec_M4_Entrada, r1 := wire#w3)
   END_RUNG
   RUNG wire#powerrail
      Contact( #Mx_ET60 )
      wire#w2
      Contact( #Simultaneo_Mx )
   END_RUNG wire#w1
   RUNG wire#powerrail
      Contact( #Mx_ET61 )
   END_RUNG wire#w2
   RUNG wire#powerrail
      Contact( #Mx_ET80 )
   END_RUNG wire#w1
   RUNG wire#powerrail
      Contact( #Mx_ET00 )
   END_RUNG wire#w3
   RUNG wire#powerrail
      Contact( #Mx_ET02 )
   END_RUNG wire#w3
   RUNG wire#powerrail
      Contact( #Mx_ET85 )
   END_RUNG wire#w3
   RUNG wire#powerrail
      Contact( #Mx_ET01 )
      I_Contact( #Mx_ET20 )
      I_Contact( #AVTF_Ent_M4 )
      Contact( #Selec_M4_Entrada )
   END_RUNG wire#w3
   // the same network as SCL:
   #_w1 := #Mx_ET00 OR #Mx_ET02 OR #Mx_ET85 OR (#Mx_ET01 AND NOT #Mx_ET20 AND NOT #AVTF_Ent_M4 AND #Selec_M4_Entrada);
   IF ((#Mx_ET01 AND NOT #ConfigFB.NoEntrar_E4) OR ((#Mx_ET60 OR #Mx_ET61) AND #Simultaneo_Mx) OR #Mx_ET80) AND #AVTF_Ent_M4 AND NOT #Selec_M1_Entrada AND NOT #Selec_M2_Entrada AND NOT #Selec_M3_Entrada AND NOT #Selec_M4_Entrada THEN
       #Selec_M4_Entrada := TRUE;   // SR flip-flop
   END_IF;
   IF #_w1 THEN #Selec_M4_Entrada := FALSE; END_IF;
END_REGION

REGION Network 10: SELECCION MESA SALIDA >> S1
   RUNG wire#powerrail
      Contact( #OrdSal_M1 )
      I_Contact( #OrdSal_M2 )
      I_Contact( #OrdSal_M3 )
      I_Contact( #OrdSal_M4 )
      I_Contact( #Selec_M1_Salida )
      I_Contact( #Selec_M2_Salida )
      I_Contact( #Selec_M3_Salida )
      I_Contact( #Selec_M4_Salida )
      S_SR(operand := #Selec_M1_Salida, r1 := wire#w1)
   END_RUNG
   RUNG wire#powerrail
      Contact( #Mx_ET00 )
   END_RUNG wire#w1
   RUNG wire#powerrail
      Contact( #Mx_ET01 )
   END_RUNG wire#w1
   RUNG wire#powerrail
      Contact( #Mx_ET10 )
      I_Contact( #OrdSal_M1 )
   END_RUNG wire#w1
   RUNG wire#powerrail
      Contact( #Mx_ET20 )
   END_RUNG wire#w1
   RUNG wire#powerrail
      Contact( #Mx_ET181 )
   END_RUNG wire#w1
   RUNG wire#powerrail
      Contact( #Mx_ET95 )
   END_RUNG wire#w1
   // the same network as SCL:
   IF #OrdSal_M1 AND NOT #OrdSal_M2 AND NOT #OrdSal_M3 AND NOT #OrdSal_M4 AND NOT #Selec_M1_Salida AND NOT #Selec_M2_Salida AND NOT #Selec_M3_Salida AND NOT #Selec_M4_Salida THEN
       #Selec_M1_Salida := TRUE;   // SR flip-flop
   END_IF;
   IF #Mx_ET00 OR #Mx_ET01 OR (#Mx_ET10 AND NOT #OrdSal_M1) OR #Mx_ET20 OR #Mx_ET181 OR #Mx_ET95 THEN
       #Selec_M1_Salida := FALSE;
   END_IF;
END_REGION

REGION Network 11: SELECCION MESA SALIDA >> S2
   RUNG wire#powerrail
      Contact( #OrdSal_M2 )
      I_Contact( #OrdSal_M1 )
      I_Contact( #OrdSal_M3 )
      I_Contact( #OrdSal_M4 )
      I_Contact( #Selec_M1_Salida )
      I_Contact( #Selec_M2_Salida )
      I_Contact( #Selec_M3_Salida )
      I_Contact( #Selec_M4_Salida )
      S_SR(operand := #Selec_M2_Salida, r1 := wire#w1)
   END_RUNG
   RUNG wire#powerrail
      Contact( #Mx_ET00 )
   END_RUNG wire#w1
   RUNG wire#powerrail
      Contact( #Mx_ET01 )
   END_RUNG wire#w1
   RUNG wire#powerrail
      Contact( #Mx_ET20 )
      I_Contact( #OrdSal_M2 )
   END_RUNG wire#w1
   RUNG wire#powerrail
      Contact( #Mx_ET10 )
   END_RUNG wire#w1
   RUNG wire#powerrail
      Contact( #Mx_ET181 )
   END_RUNG wire#w1
   RUNG wire#powerrail
      Contact( #Mx_ET95 )
   END_RUNG wire#w1
   // the same network as SCL:
   IF #OrdSal_M2 AND NOT #OrdSal_M1 AND NOT #OrdSal_M3 AND NOT #OrdSal_M4 AND NOT #Selec_M1_Salida AND NOT #Selec_M2_Salida AND NOT #Selec_M3_Salida AND NOT #Selec_M4_Salida THEN
       #Selec_M2_Salida := TRUE;   // SR flip-flop
   END_IF;
   IF #Mx_ET00 OR #Mx_ET01 OR (#Mx_ET20 AND NOT #OrdSal_M2) OR #Mx_ET10 OR #Mx_ET181 OR #Mx_ET95 THEN
       #Selec_M2_Salida := FALSE;
   END_IF;
END_REGION

REGION Network 12: SELECCION MESA SALIDA >> S3
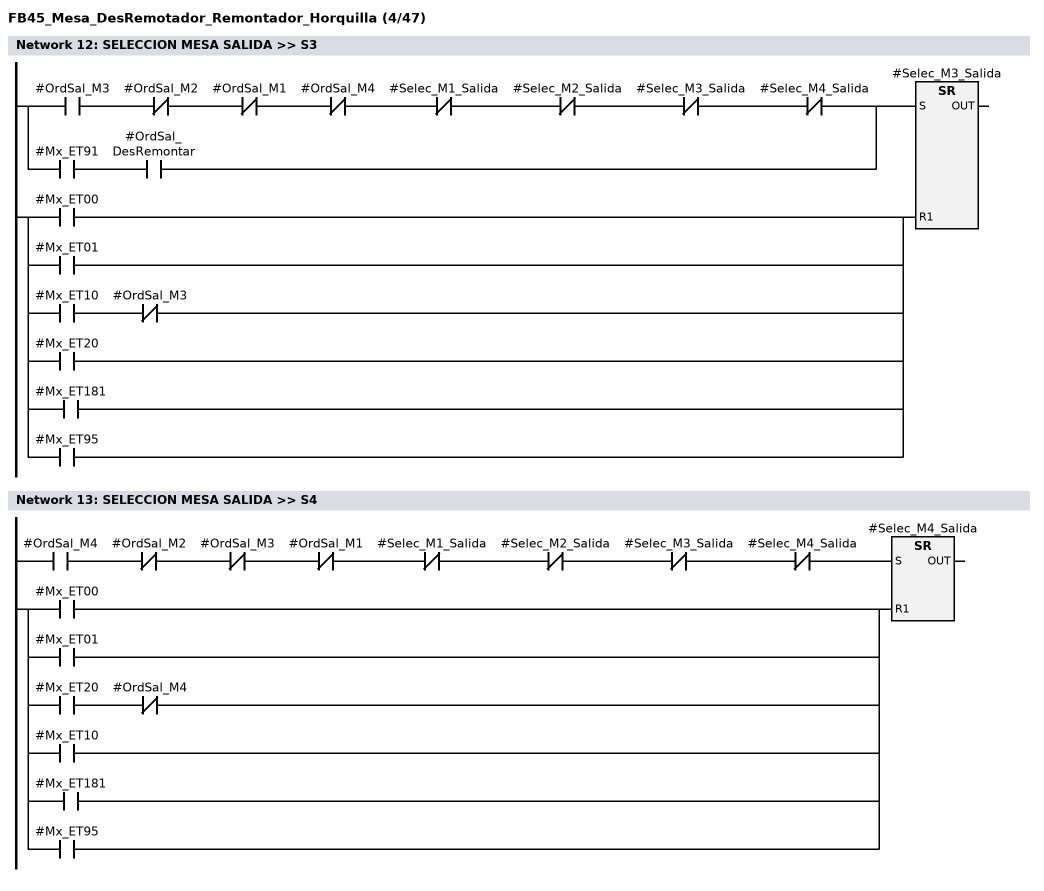
   RUNG wire#powerrail
      Contact( #OrdSal_M3 )
      I_Contact( #OrdSal_M2 )
      I_Contact( #OrdSal_M1 )
      I_Contact( #OrdSal_M4 )
      I_Contact( #Selec_M1_Salida )
      I_Contact( #Selec_M2_Salida )
      I_Contact( #Selec_M3_Salida )
      I_Contact( #Selec_M4_Salida )
      wire#w1
      S_SR(operand := #Selec_M3_Salida, r1 := wire#w2)
   END_RUNG
   RUNG wire#powerrail
      Contact( #Mx_ET91 )
      Contact( #OrdSal_DesRemontar )
   END_RUNG wire#w1
   RUNG wire#powerrail
      Contact( #Mx_ET00 )
   END_RUNG wire#w2
   RUNG wire#powerrail
      Contact( #Mx_ET01 )
   END_RUNG wire#w2
   RUNG wire#powerrail
      Contact( #Mx_ET10 )
      I_Contact( #OrdSal_M3 )
   END_RUNG wire#w2
   RUNG wire#powerrail
      Contact( #Mx_ET20 )
   END_RUNG wire#w2
   RUNG wire#powerrail
      Contact( #Mx_ET181 )
   END_RUNG wire#w2
   RUNG wire#powerrail
      Contact( #Mx_ET95 )
   END_RUNG wire#w2
   // the same network as SCL:
   IF (#OrdSal_M3 AND NOT #OrdSal_M2 AND NOT #OrdSal_M1 AND NOT #OrdSal_M4 AND NOT #Selec_M1_Salida AND NOT #Selec_M2_Salida AND NOT #Selec_M3_Salida AND NOT #Selec_M4_Salida) OR (#Mx_ET91 AND #OrdSal_DesRemontar) THEN
       #Selec_M3_Salida := TRUE;   // SR flip-flop
   END_IF;
   IF #Mx_ET00 OR #Mx_ET01 OR (#Mx_ET10 AND NOT #OrdSal_M3) OR #Mx_ET20 OR #Mx_ET181 OR #Mx_ET95 THEN
       #Selec_M3_Salida := FALSE;
   END_IF;
END_REGION

REGION Network 13: SELECCION MESA SALIDA >> S4
   RUNG wire#powerrail
      Contact( #OrdSal_M4 )
      I_Contact( #OrdSal_M2 )
      I_Contact( #OrdSal_M3 )
      I_Contact( #OrdSal_M1 )
      I_Contact( #Selec_M1_Salida )
      I_Contact( #Selec_M2_Salida )
      I_Contact( #Selec_M3_Salida )
      I_Contact( #Selec_M4_Salida )
      S_SR(operand := #Selec_M4_Salida, r1 := wire#w1)
   END_RUNG
   RUNG wire#powerrail
      Contact( #Mx_ET00 )
   END_RUNG wire#w1
   RUNG wire#powerrail
      Contact( #Mx_ET01 )
   END_RUNG wire#w1
   RUNG wire#powerrail
      Contact( #Mx_ET20 )
      I_Contact( #OrdSal_M4 )
   END_RUNG wire#w1
   RUNG wire#powerrail
      Contact( #Mx_ET10 )
   END_RUNG wire#w1
   RUNG wire#powerrail
      Contact( #Mx_ET181 )
   END_RUNG wire#w1
   RUNG wire#powerrail
      Contact( #Mx_ET95 )
   END_RUNG wire#w1
   // the same network as SCL:
   IF #OrdSal_M4 AND NOT #OrdSal_M2 AND NOT #OrdSal_M3 AND NOT #OrdSal_M1 AND NOT #Selec_M1_Salida AND NOT #Selec_M2_Salida AND NOT #Selec_M3_Salida AND NOT #Selec_M4_Salida THEN
       #Selec_M4_Salida := TRUE;   // SR flip-flop
   END_IF;
   IF #Mx_ET00 OR #Mx_ET01 OR (#Mx_ET20 AND NOT #OrdSal_M4) OR #Mx_ET10 OR #Mx_ET181 OR #Mx_ET95 THEN
       #Selec_M4_Salida := FALSE;
   END_IF;
END_REGION

REGION Network 14: VARIABLES AUXILIARES - PASAR DE LAS pHs HARDWARE >> VARIABLES --- VAR_pHsSeg >> Inico CNTSeguridad
   // El Contador de seguridad va a ir con la phs VAR_PHS_SEG y  el contador de posicionamiento con VAR_PHS.
   // Así, no tenemos que unir la posición de las fotocelulas con la posición E1,E2,E3,E4...
   // En el programa trabajamos con variables.
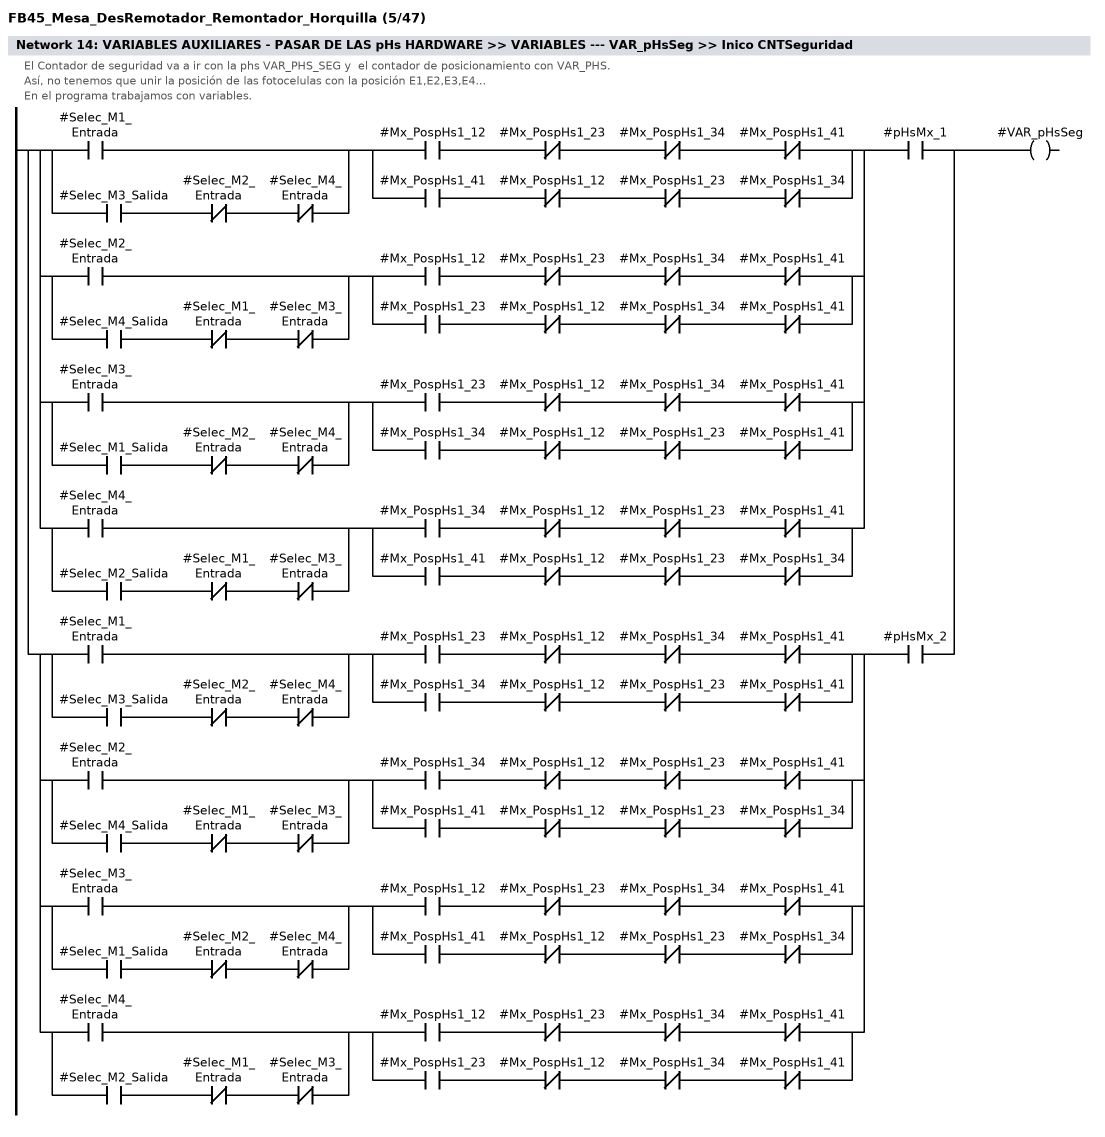
   RUNG wire#powerrail
      Contact( #Selec_M1_Entrada )
      wire#w1
      Contact( #Mx_PospHs1_12 )
      I_Contact( #Mx_PospHs1_23 )
      I_Contact( #Mx_PospHs1_34 )
      I_Contact( #Mx_PospHs1_41 )
      wire#w2
      Contact( #pHsMx_1 )
      wire#w6
      Coil( #VAR_pHsSeg )
   END_RUNG
   RUNG wire#powerrail
      Contact( #Selec_M3_Salida )
      I_Contact( #Selec_M2_Entrada )
      I_Contact( #Selec_M4_Entrada )
   END_RUNG wire#w1
   RUNG wire#w1
      Contact( #Mx_PospHs1_41 )
      I_Contact( #Mx_PospHs1_12 )
      I_Contact( #Mx_PospHs1_23 )
      I_Contact( #Mx_PospHs1_34 )
   END_RUNG wire#w2
   RUNG wire#powerrail
      Contact( #Selec_M2_Entrada )
      wire#w3
      Contact( #Mx_PospHs1_12 )
      I_Contact( #Mx_PospHs1_23 )
      I_Contact( #Mx_PospHs1_34 )
      I_Contact( #Mx_PospHs1_41 )
   END_RUNG wire#w2
   RUNG wire#powerrail
      Contact( #Selec_M4_Salida )
      I_Contact( #Selec_M1_Entrada )
      I_Contact( #Selec_M3_Entrada )
   END_RUNG wire#w3
   RUNG wire#w3
      Contact( #Mx_PospHs1_23 )
      I_Contact( #Mx_PospHs1_12 )
      I_Contact( #Mx_PospHs1_34 )
      I_Contact( #Mx_PospHs1_41 )
   END_RUNG wire#w2
   RUNG wire#powerrail
      Contact( #Selec_M3_Entrada )
      wire#w4
      Contact( #Mx_PospHs1_23 )
      I_Contact( #Mx_PospHs1_12 )
      I_Contact( #Mx_PospHs1_34 )
      I_Contact( #Mx_PospHs1_41 )
   END_RUNG wire#w2
   RUNG wire#powerrail
      Contact( #Selec_M1_Salida )
      I_Contact( #Selec_M2_Entrada )
      I_Contact( #Selec_M4_Entrada )
   END_RUNG wire#w4
   RUNG wire#w4
      Contact( #Mx_PospHs1_34 )
      I_Contact( #Mx_PospHs1_12 )
      I_Contact( #Mx_PospHs1_23 )
      I_Contact( #Mx_PospHs1_41 )
   END_RUNG wire#w2
   RUNG wire#powerrail
      Contact( #Selec_M4_Entrada )
      wire#w5
      Contact( #Mx_PospHs1_34 )
      I_Contact( #Mx_PospHs1_12 )
      I_Contact( #Mx_PospHs1_23 )
      I_Contact( #Mx_PospHs1_41 )
   END_RUNG wire#w2
   RUNG wire#powerrail
      Contact( #Selec_M2_Salida )
      I_Contact( #Selec_M1_Entrada )
      I_Contact( #Selec_M3_Entrada )
   END_RUNG wire#w5
   RUNG wire#w5
      Contact( #Mx_PospHs1_41 )
      I_Contact( #Mx_PospHs1_12 )
      I_Contact( #Mx_PospHs1_23 )
      I_Contact( #Mx_PospHs1_34 )
   END_RUNG wire#w2
   RUNG wire#powerrail
      Contact( #Selec_M1_Entrada )
      wire#w7
      Contact( #Mx_PospHs1_23 )
      I_Contact( #Mx_PospHs1_12 )
      I_Contact( #Mx_PospHs1_34 )
      I_Contact( #Mx_PospHs1_41 )
      wire#w8
      Contact( #pHsMx_2 )
   END_RUNG wire#w6
   RUNG wire#powerrail
      Contact( #Selec_M3_Salida )
      I_Contact( #Selec_M2_Entrada )
      I_Contact( #Selec_M4_Entrada )
   END_RUNG wire#w7
   RUNG wire#w7
      Contact( #Mx_PospHs1_34 )
      I_Contact( #Mx_PospHs1_12 )
      I_Contact( #Mx_PospHs1_23 )
      I_Contact( #Mx_PospHs1_41 )
   END_RUNG wire#w8
   RUNG wire#powerrail
      Contact( #Selec_M2_Entrada )
      wire#w9
      Contact( #Mx_PospHs1_34 )
      I_Contact( #Mx_PospHs1_12 )
      I_Contact( #Mx_PospHs1_23 )
      I_Contact( #Mx_PospHs1_41 )
   END_RUNG wire#w8
   RUNG wire#powerrail
      Contact( #Selec_M4_Salida )
      I_Contact( #Selec_M1_Entrada )
      I_Contact( #Selec_M3_Entrada )
   END_RUNG wire#w9
   RUNG wire#w9
      Contact( #Mx_PospHs1_41 )
      I_Contact( #Mx_PospHs1_12 )
      I_Contact( #Mx_PospHs1_23 )
      I_Contact( #Mx_PospHs1_34 )
   END_RUNG wire#w8
   RUNG wire#powerrail
      Contact( #Selec_M3_Entrada )
      wire#w10
      Contact( #Mx_PospHs1_12 )
      I_Contact( #Mx_PospHs1_23 )
      I_Contact( #Mx_PospHs1_34 )
      I_Contact( #Mx_PospHs1_41 )
   END_RUNG wire#w8
   RUNG wire#powerrail
      Contact( #Selec_M1_Salida )
      I_Contact( #Selec_M2_Entrada )
      I_Contact( #Selec_M4_Entrada )
   END_RUNG wire#w10
   RUNG wire#w10
      Contact( #Mx_PospHs1_41 )
      I_Contact( #Mx_PospHs1_12 )
      I_Contact( #Mx_PospHs1_23 )
      I_Contact( #Mx_PospHs1_34 )
   END_RUNG wire#w8
   RUNG wire#powerrail
      Contact( #Selec_M4_Entrada )
      wire#w11
      Contact( #Mx_PospHs1_12 )
      I_Contact( #Mx_PospHs1_23 )
      I_Contact( #Mx_PospHs1_34 )
      I_Contact( #Mx_PospHs1_41 )
   END_RUNG wire#w8
   RUNG wire#powerrail
      Contact( #Selec_M2_Salida )
      I_Contact( #Selec_M1_Entrada )
      I_Contact( #Selec_M3_Entrada )
   END_RUNG wire#w11
   RUNG wire#w11
      Contact( #Mx_PospHs1_23 )
      I_Contact( #Mx_PospHs1_12 )
      I_Contact( #Mx_PospHs1_34 )
      I_Contact( #Mx_PospHs1_41 )
   END_RUNG wire#w8
   // the same network as SCL:
   #VAR_pHsSeg := ((((#Selec_M1_Entrada OR (#Selec_M3_Salida AND NOT #Selec_M2_Entrada AND NOT #Selec_M4_Entrada)) AND ((#Mx_PospHs1_12 AND NOT #Mx_PospHs1_23 AND NOT #Mx_PospHs1_34 AND NOT #Mx_PospHs1_41) OR (#Mx_PospHs1_41 AND NOT #Mx_PospHs1_12 AND NOT #Mx_PospHs1_23 AND NOT #Mx_PospHs1_34))) OR ((#Selec_M2_Entrada OR (#Selec_M4_Salida AND NOT #Selec_M1_Entrada AND NOT #Selec_M3_Entrada)) AND ((#Mx_PospHs1_12 AND NOT #Mx_PospHs1_23 AND NOT #Mx_PospHs1_34 AND NOT #Mx_PospHs1_41) OR (#Mx_PospHs1_23 AND NOT #Mx_PospHs1_12 AND NOT #Mx_PospHs1_34 AND NOT #Mx_PospHs1_41))) OR ((#Selec_M3_Entrada OR (#Selec_M1_Salida AND NOT #Selec_M2_Entrada AND NOT #Selec_M4_Entrada)) AND ((#Mx_PospHs1_23 AND NOT #Mx_PospHs1_12 AND NOT #Mx_PospHs1_34 AND NOT #Mx_PospHs1_41) OR (#Mx_PospHs1_34 AND NOT #Mx_PospHs1_12 AND NOT #Mx_PospHs1_23 AND NOT #Mx_PospHs1_41))) OR ((#Selec_M4_Entrada OR (#Selec_M2_Salida AND NOT #Selec_M1_Entrada AND NOT #Selec_M3_Entrada)) AND ((#Mx_PospHs1_34 AND NOT #Mx_PospHs1_12 AND NOT #Mx_PospHs1_23 AND NOT #Mx_PospHs1_41) OR (#Mx_PospHs1_41 AND NOT #Mx_PospHs1_12 AND NOT #Mx_PospHs1_23 AND NOT #Mx_PospHs1_34)))) AND #pHsMx_1) OR ((((#Selec_M1_Entrada OR (#Selec_M3_Salida AND NOT #Selec_M2_Entrada AND NOT #Selec_M4_Entrada)) AND ((#Mx_PospHs1_23 AND NOT #Mx_PospHs1_12 AND NOT #Mx_PospHs1_34 AND NOT #Mx_PospHs1_41) OR (#Mx_PospHs1_34 AND NOT #Mx_PospHs1_12 AND NOT #Mx_PospHs1_23 AND NOT #Mx_PospHs1_41))) OR ((#Selec_M2_Entrada OR (#Selec_M4_Salida AND NOT #Selec_M1_Entrada AND NOT #Selec_M3_Entrada)) AND ((#Mx_PospHs1_34 AND NOT #Mx_PospHs1_12 AND NOT #Mx_PospHs1_23 AND NOT #Mx_PospHs1_41) OR (#Mx_PospHs1_41 AND NOT #Mx_PospHs1_12 AND NOT #Mx_PospHs1_23 AND NOT #Mx_PospHs1_34))) OR ((#Selec_M3_Entrada OR (#Selec_M1_Salida AND NOT #Selec_M2_Entrada AND NOT #Selec_M4_Entrada)) AND ((#Mx_PospHs1_12 AND NOT #Mx_PospHs1_23 AND NOT #Mx_PospHs1_34 AND NOT #Mx_PospHs1_41) OR (#Mx_PospHs1_41 AND NOT #Mx_PospHs1_12 AND NOT #Mx_PospHs1_23 AND NOT #Mx_PospHs1_34))) OR ((#Selec_M4_Entrada OR (#Selec_M2_Salida AND NOT #Selec_M1_Entrada AND NOT #Selec_M3_Entrada)) AND ((#Mx_PospHs1_12 AND NOT #Mx_PospHs1_23 AND NOT #Mx_PospHs1_34 AND NOT #Mx_PospHs1_41) OR (#Mx_PospHs1_23 AND NOT #Mx_PospHs1_12 AND NOT #Mx_PospHs1_34 AND NOT #Mx_PospHs1_41)))) AND #pHsMx_2);
END_REGION

REGION Network 15: VARIABLES AUXILIARES - PASAR DE LAS pHs HARDWARE >> VARIABLES --- VAR_pHs >> Inico CNTPosicionado
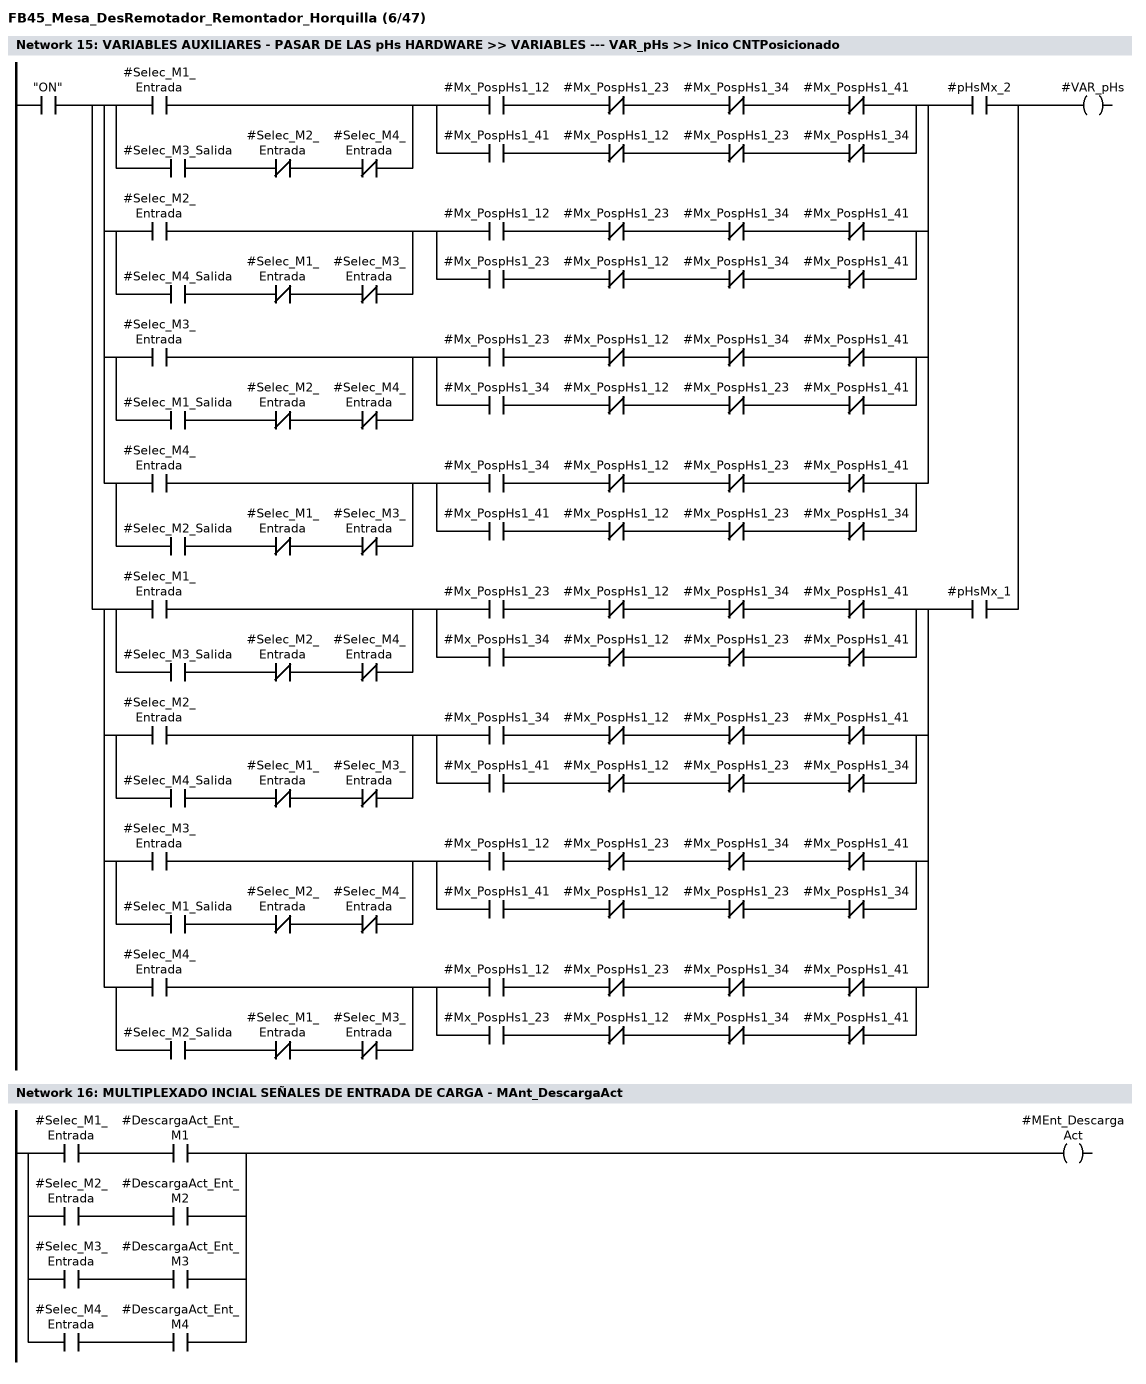
   RUNG wire#powerrail
      Contact( "ON" )
      wire#w1
      Contact( #Selec_M1_Entrada )
      wire#w2
      Contact( #Mx_PospHs1_12 )
      I_Contact( #Mx_PospHs1_23 )
      I_Contact( #Mx_PospHs1_34 )
      I_Contact( #Mx_PospHs1_41 )
      wire#w3
      Contact( #pHsMx_2 )
      wire#w7
      Coil( #VAR_pHs )
   END_RUNG
   RUNG wire#w1
      Contact( #Selec_M3_Salida )
      I_Contact( #Selec_M2_Entrada )
      I_Contact( #Selec_M4_Entrada )
   END_RUNG wire#w2
   RUNG wire#w2
      Contact( #Mx_PospHs1_41 )
      I_Contact( #Mx_PospHs1_12 )
      I_Contact( #Mx_PospHs1_23 )
      I_Contact( #Mx_PospHs1_34 )
   END_RUNG wire#w3
   RUNG wire#w1
      Contact( #Selec_M2_Entrada )
      wire#w4
      Contact( #Mx_PospHs1_12 )
      I_Contact( #Mx_PospHs1_23 )
      I_Contact( #Mx_PospHs1_34 )
      I_Contact( #Mx_PospHs1_41 )
   END_RUNG wire#w3
   RUNG wire#w1
      Contact( #Selec_M4_Salida )
      I_Contact( #Selec_M1_Entrada )
      I_Contact( #Selec_M3_Entrada )
   END_RUNG wire#w4
   RUNG wire#w4
      Contact( #Mx_PospHs1_23 )
      I_Contact( #Mx_PospHs1_12 )
      I_Contact( #Mx_PospHs1_34 )
      I_Contact( #Mx_PospHs1_41 )
   END_RUNG wire#w3
   RUNG wire#w1
      Contact( #Selec_M3_Entrada )
      wire#w5
      Contact( #Mx_PospHs1_23 )
      I_Contact( #Mx_PospHs1_12 )
      I_Contact( #Mx_PospHs1_34 )
      I_Contact( #Mx_PospHs1_41 )
   END_RUNG wire#w3
   RUNG wire#w1
      Contact( #Selec_M1_Salida )
      I_Contact( #Selec_M2_Entrada )
      I_Contact( #Selec_M4_Entrada )
   END_RUNG wire#w5
   RUNG wire#w5
      Contact( #Mx_PospHs1_34 )
      I_Contact( #Mx_PospHs1_12 )
      I_Contact( #Mx_PospHs1_23 )
      I_Contact( #Mx_PospHs1_41 )
   END_RUNG wire#w3
   RUNG wire#w1
      Contact( #Selec_M4_Entrada )
      wire#w6
      Contact( #Mx_PospHs1_34 )
      I_Contact( #Mx_PospHs1_12 )
      I_Contact( #Mx_PospHs1_23 )
      I_Contact( #Mx_PospHs1_41 )
   END_RUNG wire#w3
   RUNG wire#w1
      Contact( #Selec_M2_Salida )
      I_Contact( #Selec_M1_Entrada )
      I_Contact( #Selec_M3_Entrada )
   END_RUNG wire#w6
   RUNG wire#w6
      Contact( #Mx_PospHs1_41 )
      I_Contact( #Mx_PospHs1_12 )
      I_Contact( #Mx_PospHs1_23 )
      I_Contact( #Mx_PospHs1_34 )
   END_RUNG wire#w3
   RUNG wire#w1
      Contact( #Selec_M1_Entrada )
      wire#w8
      Contact( #Mx_PospHs1_23 )
      I_Contact( #Mx_PospHs1_12 )
      I_Contact( #Mx_PospHs1_34 )
      I_Contact( #Mx_PospHs1_41 )
      wire#w9
      Contact( #pHsMx_1 )
   END_RUNG wire#w7
   RUNG wire#w1
      Contact( #Selec_M3_Salida )
      I_Contact( #Selec_M2_Entrada )
      I_Contact( #Selec_M4_Entrada )
   END_RUNG wire#w8
   RUNG wire#w8
      Contact( #Mx_PospHs1_34 )
      I_Contact( #Mx_PospHs1_12 )
      I_Contact( #Mx_PospHs1_23 )
      I_Contact( #Mx_PospHs1_41 )
   END_RUNG wire#w9
   RUNG wire#w1
      Contact( #Selec_M2_Entrada )
      wire#w10
      Contact( #Mx_PospHs1_34 )
      I_Contact( #Mx_PospHs1_12 )
      I_Contact( #Mx_PospHs1_23 )
      I_Contact( #Mx_PospHs1_41 )
   END_RUNG wire#w9
   RUNG wire#w1
      Contact( #Selec_M4_Salida )
      I_Contact( #Selec_M1_Entrada )
      I_Contact( #Selec_M3_Entrada )
   END_RUNG wire#w10
   RUNG wire#w10
      Contact( #Mx_PospHs1_41 )
      I_Contact( #Mx_PospHs1_12 )
      I_Contact( #Mx_PospHs1_23 )
      I_Contact( #Mx_PospHs1_34 )
   END_RUNG wire#w9
   RUNG wire#w1
      Contact( #Selec_M3_Entrada )
      wire#w11
      Contact( #Mx_PospHs1_12 )
      I_Contact( #Mx_PospHs1_23 )
      I_Contact( #Mx_PospHs1_34 )
      I_Contact( #Mx_PospHs1_41 )
   END_RUNG wire#w9
   RUNG wire#w1
      Contact( #Selec_M1_Salida )
      I_Contact( #Selec_M2_Entrada )
      I_Contact( #Selec_M4_Entrada )
   END_RUNG wire#w11
   RUNG wire#w11
      Contact( #Mx_PospHs1_41 )
      I_Contact( #Mx_PospHs1_12 )
      I_Contact( #Mx_PospHs1_23 )
      I_Contact( #Mx_PospHs1_34 )
   END_RUNG wire#w9
   RUNG wire#w1
      Contact( #Selec_M4_Entrada )
      wire#w12
      Contact( #Mx_PospHs1_12 )
      I_Contact( #Mx_PospHs1_23 )
      I_Contact( #Mx_PospHs1_34 )
      I_Contact( #Mx_PospHs1_41 )
   END_RUNG wire#w9
   RUNG wire#w1
      Contact( #Selec_M2_Salida )
      I_Contact( #Selec_M1_Entrada )
      I_Contact( #Selec_M3_Entrada )
   END_RUNG wire#w12
   RUNG wire#w12
      Contact( #Mx_PospHs1_23 )
      I_Contact( #Mx_PospHs1_12 )
      I_Contact( #Mx_PospHs1_34 )
      I_Contact( #Mx_PospHs1_41 )
   END_RUNG wire#w9
   // the same network as SCL:
   #VAR_pHs := "ON" AND (((((#Selec_M1_Entrada OR (#Selec_M3_Salida AND NOT #Selec_M2_Entrada AND NOT #Selec_M4_Entrada)) AND ((#Mx_PospHs1_12 AND NOT #Mx_PospHs1_23 AND NOT #Mx_PospHs1_34 AND NOT #Mx_PospHs1_41) OR (#Mx_PospHs1_41 AND NOT #Mx_PospHs1_12 AND NOT #Mx_PospHs1_23 AND NOT #Mx_PospHs1_34))) OR ((#Selec_M2_Entrada OR (#Selec_M4_Salida AND NOT #Selec_M1_Entrada AND NOT #Selec_M3_Entrada)) AND ((#Mx_PospHs1_12 AND NOT #Mx_PospHs1_23 AND NOT #Mx_PospHs1_34 AND NOT #Mx_PospHs1_41) OR (#Mx_PospHs1_23 AND NOT #Mx_PospHs1_12 AND NOT #Mx_PospHs1_34 AND NOT #Mx_PospHs1_41))) OR ((#Selec_M3_Entrada OR (#Selec_M1_Salida AND NOT #Selec_M2_Entrada AND NOT #Selec_M4_Entrada)) AND ((#Mx_PospHs1_23 AND NOT #Mx_PospHs1_12 AND NOT #Mx_PospHs1_34 AND NOT #Mx_PospHs1_41) OR (#Mx_PospHs1_34 AND NOT #Mx_PospHs1_12 AND NOT #Mx_PospHs1_23 AND NOT #Mx_PospHs1_41))) OR ((#Selec_M4_Entrada OR (#Selec_M2_Salida AND NOT #Selec_M1_Entrada AND NOT #Selec_M3_Entrada)) AND ((#Mx_PospHs1_34 AND NOT #Mx_PospHs1_12 AND NOT #Mx_PospHs1_23 AND NOT #Mx_PospHs1_41) OR (#Mx_PospHs1_41 AND NOT #Mx_PospHs1_12 AND NOT #Mx_PospHs1_23 AND NOT #Mx_PospHs1_34)))) AND #pHsMx_2) OR ((((#Selec_M1_Entrada OR (#Selec_M3_Salida AND NOT #Selec_M2_Entrada AND NOT #Selec_M4_Entrada)) AND ((#Mx_PospHs1_23 AND NOT #Mx_PospHs1_12 AND NOT #Mx_PospHs1_34 AND NOT #Mx_PospHs1_41) OR (#Mx_PospHs1_34 AND NOT #Mx_PospHs1_12 AND NOT #Mx_PospHs1_23 AND NOT #Mx_PospHs1_41))) OR ((#Selec_M2_Entrada OR (#Selec_M4_Salida AND NOT #Selec_M1_Entrada AND NOT #Selec_M3_Entrada)) AND ((#Mx_PospHs1_34 AND NOT #Mx_PospHs1_12 AND NOT #Mx_PospHs1_23 AND NOT #Mx_PospHs1_41) OR (#Mx_PospHs1_41 AND NOT #Mx_PospHs1_12 AND NOT #Mx_PospHs1_23 AND NOT #Mx_PospHs1_34))) OR ((#Selec_M3_Entrada OR (#Selec_M1_Salida AND NOT #Selec_M2_Entrada AND NOT #Selec_M4_Entrada)) AND ((#Mx_PospHs1_12 AND NOT #Mx_PospHs1_23 AND NOT #Mx_PospHs1_34 AND NOT #Mx_PospHs1_41) OR (#Mx_PospHs1_41 AND NOT #Mx_PospHs1_12 AND NOT #Mx_PospHs1_23 AND NOT #Mx_PospHs1_34))) OR ((#Selec_M4_Entrada OR (#Selec_M2_Salida AND NOT #Selec_M1_Entrada AND NOT #Selec_M3_Entrada)) AND ((#Mx_PospHs1_12 AND NOT #Mx_PospHs1_23 AND NOT #Mx_PospHs1_34 AND NOT #Mx_PospHs1_41) OR (#Mx_PospHs1_23 AND NOT #Mx_PospHs1_12 AND NOT #Mx_PospHs1_34 AND NOT #Mx_PospHs1_41)))) AND #pHsMx_1));
END_REGION

REGION Network 16: MULTIPLEXADO INCIAL SEÑALES DE ENTRADA DE CARGA - MAnt_DescargaAct
   RUNG wire#powerrail
      Contact( #Selec_M1_Entrada )
      Contact( #DescargaAct_Ent_M1 )
      wire#w1
      Coil( #MEnt_DescargaAct )
   END_RUNG
   RUNG wire#powerrail
      Contact( #Selec_M2_Entrada )
      Contact( #DescargaAct_Ent_M2 )
   END_RUNG wire#w1
   RUNG wire#powerrail
      Contact( #Selec_M3_Entrada )
      Contact( #DescargaAct_Ent_M3 )
   END_RUNG wire#w1
   RUNG wire#powerrail
      Contact( #Selec_M4_Entrada )
      Contact( #DescargaAct_Ent_M4 )
   END_RUNG wire#w1
   // the same network as SCL:
   #MEnt_DescargaAct := (#Selec_M1_Entrada AND #DescargaAct_Ent_M1) OR (#Selec_M2_Entrada AND #DescargaAct_Ent_M2) OR (#Selec_M3_Entrada AND #DescargaAct_Ent_M3) OR (#Selec_M4_Entrada AND #DescargaAct_Ent_M4);
END_REGION

REGION Network 17: MULTIPLEXADO INCIAL SEÑALES DE ENTRADA DE CARGA - AVTF_MEnt
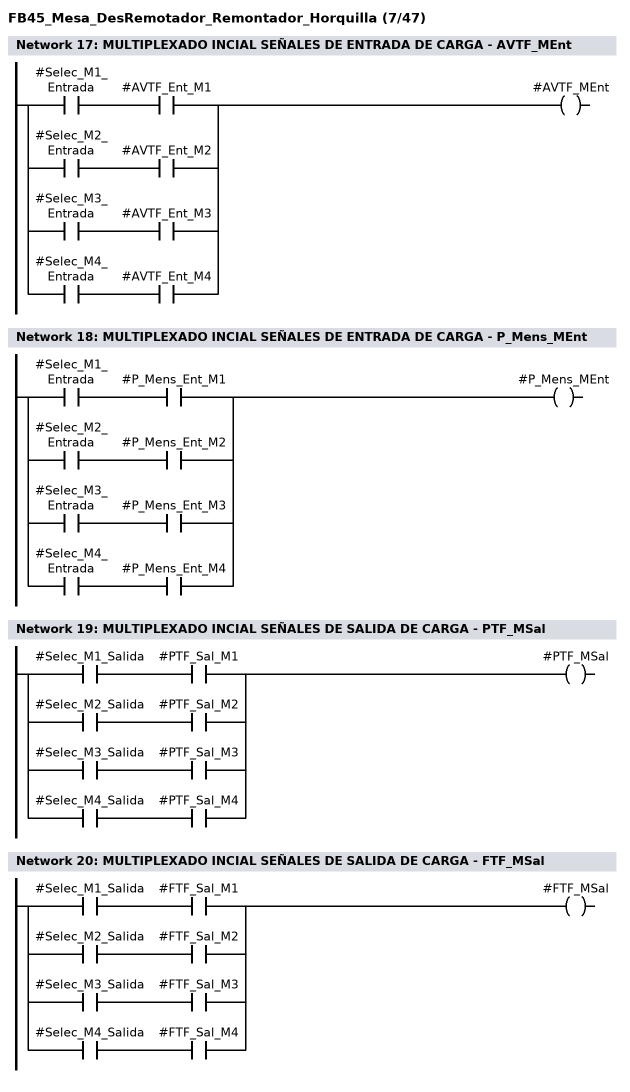
   RUNG wire#powerrail
      Contact( #Selec_M1_Entrada )
      Contact( #AVTF_Ent_M1 )
      wire#w1
      Coil( #AVTF_MEnt )
   END_RUNG
   RUNG wire#powerrail
      Contact( #Selec_M2_Entrada )
      Contact( #AVTF_Ent_M2 )
   END_RUNG wire#w1
   RUNG wire#powerrail
      Contact( #Selec_M3_Entrada )
      Contact( #AVTF_Ent_M3 )
   END_RUNG wire#w1
   RUNG wire#powerrail
      Contact( #Selec_M4_Entrada )
      Contact( #AVTF_Ent_M4 )
   END_RUNG wire#w1
   // the same network as SCL:
   #AVTF_MEnt := (#Selec_M1_Entrada AND #AVTF_Ent_M1) OR (#Selec_M2_Entrada AND #AVTF_Ent_M2) OR (#Selec_M3_Entrada AND #AVTF_Ent_M3) OR (#Selec_M4_Entrada AND #AVTF_Ent_M4);
END_REGION

REGION Network 18: MULTIPLEXADO INCIAL SEÑALES DE ENTRADA DE CARGA - P_Mens_MEnt
   RUNG wire#powerrail
      Contact( #Selec_M1_Entrada )
      Contact( #P_Mens_Ent_M1 )
      wire#w1
      Coil( #P_Mens_MEnt )
   END_RUNG
   RUNG wire#powerrail
      Contact( #Selec_M2_Entrada )
      Contact( #P_Mens_Ent_M2 )
   END_RUNG wire#w1
   RUNG wire#powerrail
      Contact( #Selec_M3_Entrada )
      Contact( #P_Mens_Ent_M3 )
   END_RUNG wire#w1
   RUNG wire#powerrail
      Contact( #Selec_M4_Entrada )
      Contact( #P_Mens_Ent_M4 )
   END_RUNG wire#w1
   // the same network as SCL:
   #P_Mens_MEnt := (#Selec_M1_Entrada AND #P_Mens_Ent_M1) OR (#Selec_M2_Entrada AND #P_Mens_Ent_M2) OR (#Selec_M3_Entrada AND #P_Mens_Ent_M3) OR (#Selec_M4_Entrada AND #P_Mens_Ent_M4);
END_REGION

REGION Network 19: MULTIPLEXADO INCIAL SEÑALES DE SALIDA DE CARGA - PTF_MSal
   RUNG wire#powerrail
      Contact( #Selec_M1_Salida )
      Contact( #PTF_Sal_M1 )
      wire#w1
      Coil( #PTF_MSal )
   END_RUNG
   RUNG wire#powerrail
      Contact( #Selec_M2_Salida )
      Contact( #PTF_Sal_M2 )
   END_RUNG wire#w1
   RUNG wire#powerrail
      Contact( #Selec_M3_Salida )
      Contact( #PTF_Sal_M3 )
   END_RUNG wire#w1
   RUNG wire#powerrail
      Contact( #Selec_M4_Salida )
      Contact( #PTF_Sal_M4 )
   END_RUNG wire#w1
   // the same network as SCL:
   #PTF_MSal := (#Selec_M1_Salida AND #PTF_Sal_M1) OR (#Selec_M2_Salida AND #PTF_Sal_M2) OR (#Selec_M3_Salida AND #PTF_Sal_M3) OR (#Selec_M4_Salida AND #PTF_Sal_M4);
END_REGION

REGION Network 20: MULTIPLEXADO INCIAL SEÑALES DE SALIDA DE CARGA - FTF_MSal
   RUNG wire#powerrail
      Contact( #Selec_M1_Salida )
      Contact( #FTF_Sal_M1 )
      wire#w1
      Coil( #FTF_MSal )
   END_RUNG
   RUNG wire#powerrail
      Contact( #Selec_M2_Salida )
      Contact( #FTF_Sal_M2 )
   END_RUNG wire#w1
   RUNG wire#powerrail
      Contact( #Selec_M3_Salida )
      Contact( #FTF_Sal_M3 )
   END_RUNG wire#w1
   RUNG wire#powerrail
      Contact( #Selec_M4_Salida )
      Contact( #FTF_Sal_M4 )
   END_RUNG wire#w1
   // the same network as SCL:
   #FTF_MSal := (#Selec_M1_Salida AND #FTF_Sal_M1) OR (#Selec_M2_Salida AND #FTF_Sal_M2) OR (#Selec_M3_Salida AND #FTF_Sal_M3) OR (#Selec_M4_Salida AND #FTF_Sal_M4);
END_REGION

REGION Network 21: VARIABLES AUXILIARES - Saliendo la Carga de la Mesa
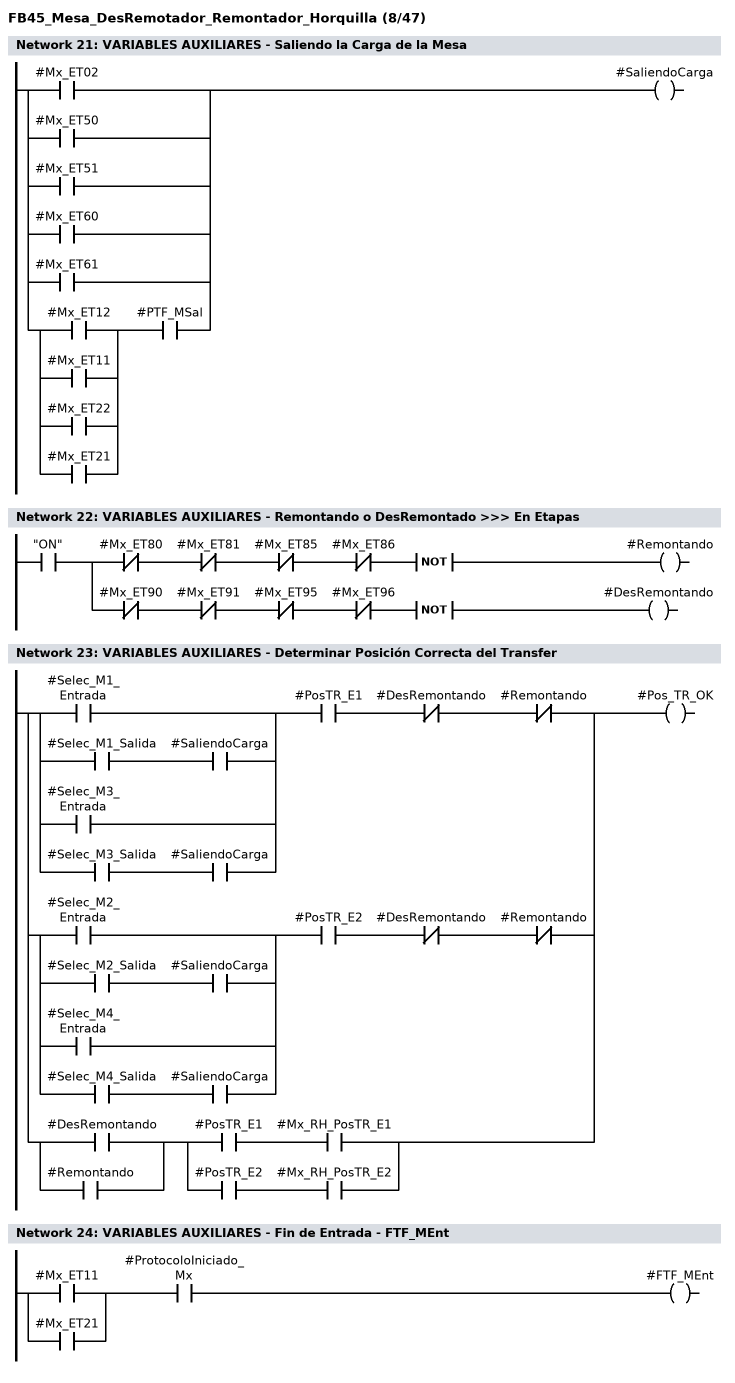
   RUNG wire#powerrail
      Contact( #Mx_ET02 )
      wire#w1
      Coil( #SaliendoCarga )
   END_RUNG
   RUNG wire#powerrail
      Contact( #Mx_ET50 )
   END_RUNG wire#w1
   RUNG wire#powerrail
      Contact( #Mx_ET51 )
   END_RUNG wire#w1
   RUNG wire#powerrail
      Contact( #Mx_ET60 )
   END_RUNG wire#w1
   RUNG wire#powerrail
      Contact( #Mx_ET61 )
   END_RUNG wire#w1
   RUNG wire#powerrail
      Contact( #Mx_ET12 )
      wire#w2
      Contact( #PTF_MSal )
   END_RUNG wire#w1
   RUNG wire#powerrail
      Contact( #Mx_ET11 )
   END_RUNG wire#w2
   RUNG wire#powerrail
      Contact( #Mx_ET22 )
   END_RUNG wire#w2
   RUNG wire#powerrail
      Contact( #Mx_ET21 )
   END_RUNG wire#w2
   // the same network as SCL:
   #SaliendoCarga := #Mx_ET02 OR #Mx_ET50 OR #Mx_ET51 OR #Mx_ET60 OR #Mx_ET61 OR ((#Mx_ET12 OR #Mx_ET11 OR #Mx_ET22 OR #Mx_ET21) AND #PTF_MSal);
END_REGION

REGION Network 22: VARIABLES AUXILIARES - Remontando o DesRemontado >>> En Etapas
   RUNG wire#powerrail
      Contact( "ON" )
      wire#w1
      I_Contact( #Mx_ET80 )
      I_Contact( #Mx_ET81 )
      I_Contact( #Mx_ET85 )
      I_Contact( #Mx_ET86 )
      Not()
      Coil( #Remontando )
   END_RUNG
   RUNG wire#w1
      I_Contact( #Mx_ET90 )
      I_Contact( #Mx_ET91 )
      I_Contact( #Mx_ET95 )
      I_Contact( #Mx_ET96 )
      Not()
      Coil( #DesRemontando )
   END_RUNG
   // the same network as SCL:
   #Remontando := NOT ("ON" AND NOT #Mx_ET80 AND NOT #Mx_ET81 AND NOT #Mx_ET85 AND NOT #Mx_ET86);
   #DesRemontando := NOT ("ON" AND NOT #Mx_ET90 AND NOT #Mx_ET91 AND NOT #Mx_ET95 AND NOT #Mx_ET96);
END_REGION

REGION Network 23: VARIABLES AUXILIARES - Determinar Posición Correcta del Transfer
   RUNG wire#powerrail
      Contact( #Selec_M1_Entrada )
      wire#w1
      Contact( #PosTR_E1 )
      I_Contact( #DesRemontando )
      I_Contact( #Remontando )
      wire#w2
      Coil( #Pos_TR_OK )
   END_RUNG
   RUNG wire#powerrail
      Contact( #Selec_M1_Salida )
      Contact( #SaliendoCarga )
   END_RUNG wire#w1
   RUNG wire#powerrail
      Contact( #Selec_M3_Entrada )
   END_RUNG wire#w1
   RUNG wire#powerrail
      Contact( #Selec_M3_Salida )
      Contact( #SaliendoCarga )
   END_RUNG wire#w1
   RUNG wire#powerrail
      Contact( #Selec_M2_Entrada )
      wire#w3
      Contact( #PosTR_E2 )
      I_Contact( #DesRemontando )
      I_Contact( #Remontando )
   END_RUNG wire#w2
   RUNG wire#powerrail
      Contact( #Selec_M2_Salida )
      Contact( #SaliendoCarga )
   END_RUNG wire#w3
   RUNG wire#powerrail
      Contact( #Selec_M4_Entrada )
   END_RUNG wire#w3
   RUNG wire#powerrail
      Contact( #Selec_M4_Salida )
      Contact( #SaliendoCarga )
   END_RUNG wire#w3
   RUNG wire#powerrail
      Contact( #DesRemontando )
      wire#w4
      Contact( #PosTR_E1 )
      Contact( #Mx_RH_PosTR_E1 )
   END_RUNG wire#w2
   RUNG wire#powerrail
      Contact( #Remontando )
   END_RUNG wire#w4
   RUNG wire#w4
      Contact( #PosTR_E2 )
      Contact( #Mx_RH_PosTR_E2 )
   END_RUNG wire#w2
   // the same network as SCL:
   #Pos_TR_OK := ((#Selec_M1_Entrada OR (#Selec_M1_Salida AND #SaliendoCarga) OR #Selec_M3_Entrada OR (#Selec_M3_Salida AND #SaliendoCarga)) AND #PosTR_E1 AND NOT #DesRemontando AND NOT #Remontando) OR ((#Selec_M2_Entrada OR (#Selec_M2_Salida AND #SaliendoCarga) OR #Selec_M4_Entrada OR (#Selec_M4_Salida AND #SaliendoCarga)) AND #PosTR_E2 AND NOT #DesRemontando AND NOT #Remontando) OR ((#DesRemontando OR #Remontando) AND ((#PosTR_E1 AND #Mx_RH_PosTR_E1) OR (#PosTR_E2 AND #Mx_RH_PosTR_E2)));
END_REGION

REGION Network 24: VARIABLES AUXILIARES - Fin de Entrada - FTF_MEnt
   RUNG wire#powerrail
      Contact( #Mx_ET11 )
      wire#w1
      Contact( #ProtocoloIniciado_Mx )
      Coil( #FTF_MEnt )
   END_RUNG
   RUNG wire#powerrail
      Contact( #Mx_ET21 )
   END_RUNG wire#w1
   // the same network as SCL:
   #FTF_MEnt := (#Mx_ET11 OR #Mx_ET21) AND #ProtocoloIniciado_Mx;
END_REGION

REGION Network 25: ESTADO DE LA MESA - DesCarga Activa
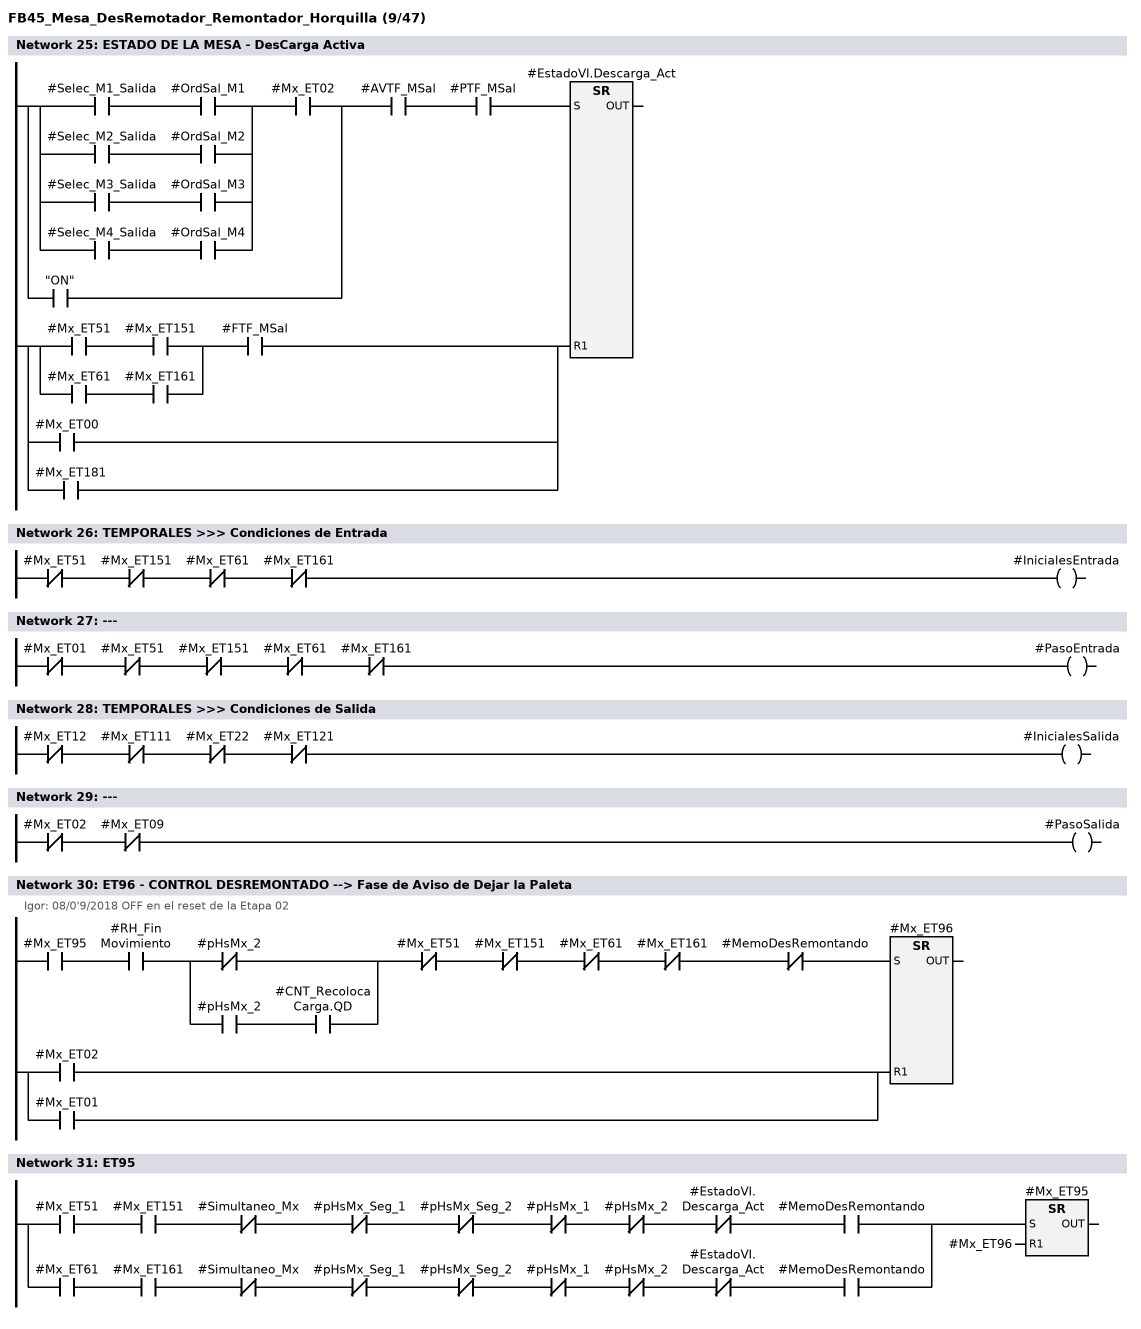
   RUNG wire#powerrail
      Contact( #Selec_M1_Salida )
      Contact( #OrdSal_M1 )
      wire#w1
      Contact( #Mx_ET02 )
      wire#w2
      Contact( #AVTF_MSal )
      Contact( #PTF_MSal )
      S_SR(operand := #EstadoVI.Descarga_Act, r1 := wire#w4)
   END_RUNG
   RUNG wire#powerrail
      Contact( #Selec_M2_Salida )
      Contact( #OrdSal_M2 )
   END_RUNG wire#w1
   RUNG wire#powerrail
      Contact( #Selec_M3_Salida )
      Contact( #OrdSal_M3 )
   END_RUNG wire#w1
   RUNG wire#powerrail
      Contact( #Selec_M4_Salida )
      Contact( #OrdSal_M4 )
   END_RUNG wire#w1
   RUNG wire#powerrail
      Contact( "ON" )
   END_RUNG wire#w2
   RUNG wire#powerrail
      Contact( #Mx_ET51 )
      Contact( #Mx_ET151 )
      wire#w3
      Contact( #FTF_MSal )
   END_RUNG wire#w4
   RUNG wire#powerrail
      Contact( #Mx_ET61 )
      Contact( #Mx_ET161 )
   END_RUNG wire#w3
   RUNG wire#powerrail
      Contact( #Mx_ET00 )
   END_RUNG wire#w4
   RUNG wire#powerrail
      Contact( #Mx_ET181 )
   END_RUNG wire#w4
   // the same network as SCL:
   IF ((((#Selec_M1_Salida AND #OrdSal_M1) OR (#Selec_M2_Salida AND #OrdSal_M2) OR (#Selec_M3_Salida AND #OrdSal_M3) OR (#Selec_M4_Salida AND #OrdSal_M4)) AND #Mx_ET02) OR "ON") AND #AVTF_MSal AND #PTF_MSal THEN
       #EstadoVI.Descarga_Act := TRUE;   // SR flip-flop
   END_IF;
   IF (((#Mx_ET51 AND #Mx_ET151) OR (#Mx_ET61 AND #Mx_ET161)) AND #FTF_MSal) OR #Mx_ET00 OR #Mx_ET181 THEN
       #EstadoVI.Descarga_Act := FALSE;
   END_IF;
END_REGION

REGION Network 26: TEMPORALES >>> Condiciones de Entrada
   RUNG wire#powerrail
      I_Contact( #Mx_ET51 )
      I_Contact( #Mx_ET151 )
      I_Contact( #Mx_ET61 )
      I_Contact( #Mx_ET161 )
      Coil( #InicialesEntrada )
   END_RUNG
   // the same network as SCL:
   #InicialesEntrada := NOT #Mx_ET51 AND NOT #Mx_ET151 AND NOT #Mx_ET61 AND NOT #Mx_ET161;
END_REGION

REGION Network 27: ---
   RUNG wire#powerrail
      I_Contact( #Mx_ET01 )
      I_Contact( #Mx_ET51 )
      I_Contact( #Mx_ET151 )
      I_Contact( #Mx_ET61 )
      I_Contact( #Mx_ET161 )
      Coil( #PasoEntrada )
   END_RUNG
   // the same network as SCL:
   #PasoEntrada := NOT #Mx_ET01 AND NOT #Mx_ET51 AND NOT #Mx_ET151 AND NOT #Mx_ET61 AND NOT #Mx_ET161;
END_REGION

REGION Network 28: TEMPORALES >>> Condiciones de Salida
   RUNG wire#powerrail
      I_Contact( #Mx_ET12 )
      I_Contact( #Mx_ET111 )
      I_Contact( #Mx_ET22 )
      I_Contact( #Mx_ET121 )
      Coil( #InicialesSalida )
   END_RUNG
   // the same network as SCL:
   #InicialesSalida := NOT #Mx_ET12 AND NOT #Mx_ET111 AND NOT #Mx_ET22 AND NOT #Mx_ET121;
END_REGION

REGION Network 29: ---
   RUNG wire#powerrail
      I_Contact( #Mx_ET02 )
      I_Contact( #Mx_ET09 )
      Coil( #PasoSalida )
   END_RUNG
   // the same network as SCL:
   #PasoSalida := NOT #Mx_ET02 AND NOT #Mx_ET09;
END_REGION

REGION Network 30: ET96 - CONTROL DESREMONTADO --> Fase de Aviso de Dejar la Paleta
   // Igor: 08/0'9/2018 OFF en el reset de la Etapa 02
   RUNG wire#powerrail
      Contact( #Mx_ET95 )
      Contact( #RH_FinMovimiento )
      wire#w1
      I_Contact( #pHsMx_2 )
      wire#w2
      I_Contact( #Mx_ET51 )
      I_Contact( #Mx_ET151 )
      I_Contact( #Mx_ET61 )
      I_Contact( #Mx_ET161 )
      I_Contact( #MemoDesRemontando )
      S_SR(operand := #Mx_ET96, r1 := wire#w3)
   END_RUNG
   RUNG wire#w1
      Contact( #pHsMx_2 )
      Contact( #CNT_RecolocaCarga.QD )
   END_RUNG wire#w2
   RUNG wire#powerrail
      Contact( #Mx_ET02 )
   END_RUNG wire#w3
   RUNG wire#powerrail
      Contact( #Mx_ET01 )
   END_RUNG wire#w3
   // the same network as SCL:
   IF #Mx_ET95 AND #RH_FinMovimiento AND (NOT #pHsMx_2 OR (#pHsMx_2 AND #CNT_RecolocaCarga.QD)) AND NOT #Mx_ET51 AND NOT #Mx_ET151 AND NOT #Mx_ET61 AND NOT #Mx_ET161 AND NOT #MemoDesRemontando THEN
       #Mx_ET96 := TRUE;   // SR flip-flop
   END_IF;
   IF #Mx_ET02 OR #Mx_ET01 THEN #Mx_ET96 := FALSE; END_IF;
END_REGION

REGION Network 31: ET95
   RUNG wire#powerrail
      Contact( #Mx_ET51 )
      Contact( #Mx_ET151 )
      I_Contact( #Simultaneo_Mx )
      I_Contact( #pHsMx_Seg_1 )
      I_Contact( #pHsMx_Seg_2 )
      I_Contact( #pHsMx_1 )
      I_Contact( #pHsMx_2 )
      I_Contact( #EstadoVI.Descarga_Act )
      Contact( #MemoDesRemontando )
      wire#w1
      S_SR(operand := #Mx_ET95, r1 := #Mx_ET96)
   END_RUNG
   RUNG wire#powerrail
      Contact( #Mx_ET61 )
      Contact( #Mx_ET161 )
      I_Contact( #Simultaneo_Mx )
      I_Contact( #pHsMx_Seg_1 )
      I_Contact( #pHsMx_Seg_2 )
      I_Contact( #pHsMx_1 )
      I_Contact( #pHsMx_2 )
      I_Contact( #EstadoVI.Descarga_Act )
      Contact( #MemoDesRemontando )
   END_RUNG wire#w1
   // the same network as SCL:
   IF (#Mx_ET51 AND #Mx_ET151 AND NOT #Simultaneo_Mx AND NOT #pHsMx_Seg_1 AND NOT #pHsMx_Seg_2 AND NOT #pHsMx_1 AND NOT #pHsMx_2 AND NOT #EstadoVI.Descarga_Act AND #MemoDesRemontando) OR (#Mx_ET61 AND #Mx_ET161 AND NOT #Simultaneo_Mx AND NOT #pHsMx_Seg_1 AND NOT #pHsMx_Seg_2 AND NOT #pHsMx_1 AND NOT #pHsMx_2 AND NOT #EstadoVI.Descarga_Act AND #MemoDesRemontando) THEN
       #Mx_ET95 := TRUE;   // SR flip-flop
   END_IF;
   IF #Mx_ET96 THEN #Mx_ET95 := FALSE; END_IF;
END_REGION

REGION Network 32: ET91 - CONTROL DESREMONTADO --> Fase de Aviso de DesRemontado de la Paleta
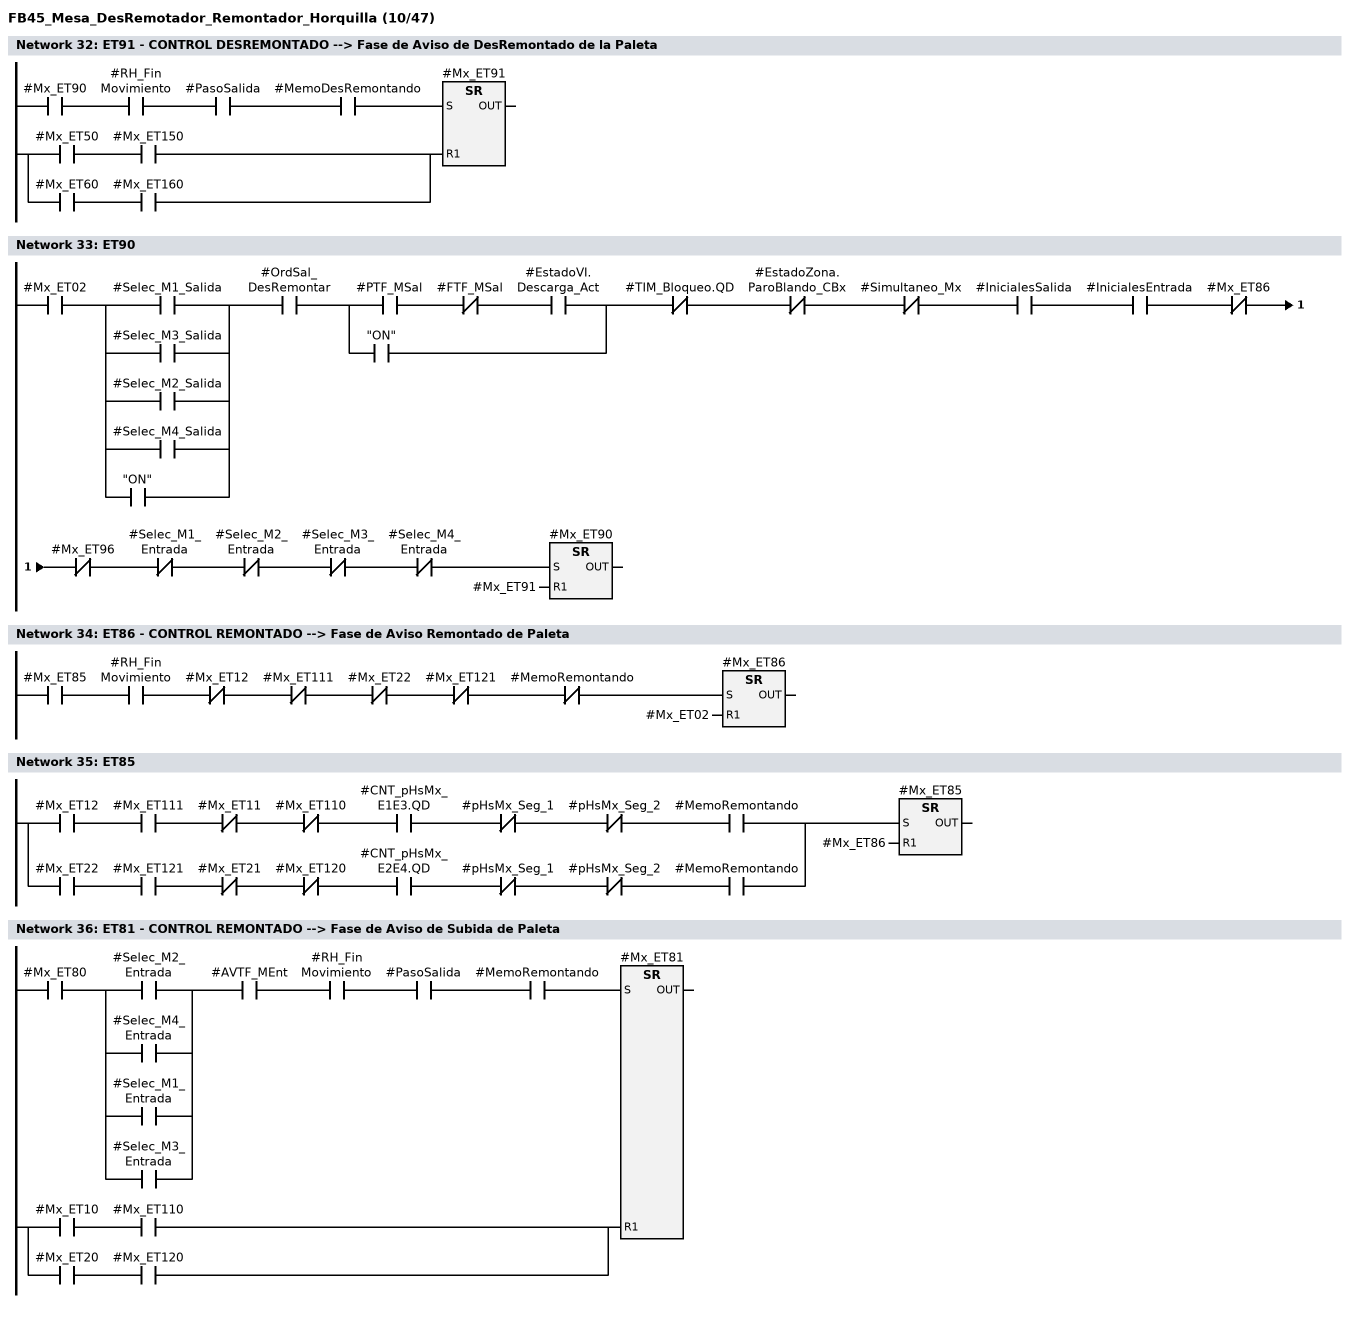
   RUNG wire#powerrail
      Contact( #Mx_ET90 )
      Contact( #RH_FinMovimiento )
      Contact( #PasoSalida )
      Contact( #MemoDesRemontando )
      S_SR(operand := #Mx_ET91, r1 := wire#w1)
   END_RUNG
   RUNG wire#powerrail
      Contact( #Mx_ET50 )
      Contact( #Mx_ET150 )
   END_RUNG wire#w1
   RUNG wire#powerrail
      Contact( #Mx_ET60 )
      Contact( #Mx_ET160 )
   END_RUNG wire#w1
   // the same network as SCL:
   IF #Mx_ET90 AND #RH_FinMovimiento AND #PasoSalida AND #MemoDesRemontando THEN
       #Mx_ET91 := TRUE;   // SR flip-flop
   END_IF;
   IF (#Mx_ET50 AND #Mx_ET150) OR (#Mx_ET60 AND #Mx_ET160) THEN #Mx_ET91 := FALSE; END_IF;
END_REGION

REGION Network 33: ET90
   RUNG wire#powerrail
      Contact( #Mx_ET02 )
      wire#w1
      Contact( #Selec_M1_Salida )
      wire#w2
      Contact( #OrdSal_DesRemontar )
      wire#w3
      Contact( #PTF_MSal )
      I_Contact( #FTF_MSal )
      Contact( #EstadoVI.Descarga_Act )
      wire#w4
      I_Contact( #TIM_Bloqueo.QD )
      I_Contact( #EstadoZona.ParoBlando_CBx )
      I_Contact( #Simultaneo_Mx )
      Contact( #InicialesSalida )
      Contact( #InicialesEntrada )
      I_Contact( #Mx_ET86 )
      I_Contact( #Mx_ET96 )
      I_Contact( #Selec_M1_Entrada )
      I_Contact( #Selec_M2_Entrada )
      I_Contact( #Selec_M3_Entrada )
      I_Contact( #Selec_M4_Entrada )
      S_SR(operand := #Mx_ET90, r1 := #Mx_ET91)
   END_RUNG
   RUNG wire#w1
      Contact( #Selec_M3_Salida )
   END_RUNG wire#w2
   RUNG wire#w1
      Contact( #Selec_M2_Salida )
   END_RUNG wire#w2
   RUNG wire#w1
      Contact( #Selec_M4_Salida )
   END_RUNG wire#w2
   RUNG wire#w1
      Contact( "ON" )
   END_RUNG wire#w2
   RUNG wire#w3
      Contact( "ON" )
   END_RUNG wire#w4
   // the same network as SCL:
   IF #Mx_ET02 AND (#Selec_M1_Salida OR #Selec_M3_Salida OR #Selec_M2_Salida OR #Selec_M4_Salida OR "ON") AND #OrdSal_DesRemontar AND ((#PTF_MSal AND NOT #FTF_MSal AND #EstadoVI.Descarga_Act) OR "ON") AND NOT #TIM_Bloqueo.QD AND NOT #EstadoZona.ParoBlando_CBx AND NOT #Simultaneo_Mx AND #InicialesSalida AND #InicialesEntrada AND NOT #Mx_ET86 AND NOT #Mx_ET96 AND NOT #Selec_M1_Entrada AND NOT #Selec_M2_Entrada AND NOT #Selec_M3_Entrada AND NOT #Selec_M4_Entrada THEN
       #Mx_ET90 := TRUE;   // SR flip-flop
   END_IF;
   IF #Mx_ET91 THEN #Mx_ET90 := FALSE; END_IF;
END_REGION

REGION Network 34: ET86 - CONTROL REMONTADO --> Fase de Aviso Remontado de Paleta
   RUNG wire#powerrail
      Contact( #Mx_ET85 )
      Contact( #RH_FinMovimiento )
      I_Contact( #Mx_ET12 )
      I_Contact( #Mx_ET111 )
      I_Contact( #Mx_ET22 )
      I_Contact( #Mx_ET121 )
      I_Contact( #MemoRemontando )
      S_SR(operand := #Mx_ET86, r1 := #Mx_ET02)
   END_RUNG
   // the same network as SCL:
   IF #Mx_ET85 AND #RH_FinMovimiento AND NOT #Mx_ET12 AND NOT #Mx_ET111 AND NOT #Mx_ET22 AND NOT #Mx_ET121 AND NOT #MemoRemontando THEN
       #Mx_ET86 := TRUE;   // SR flip-flop
   END_IF;
   IF #Mx_ET02 THEN #Mx_ET86 := FALSE; END_IF;
END_REGION

REGION Network 35: ET85
   RUNG wire#powerrail
      Contact( #Mx_ET12 )
      Contact( #Mx_ET111 )
      I_Contact( #Mx_ET11 )
      I_Contact( #Mx_ET110 )
      Contact( #CNT_pHsMx_E1E3.QD )
      I_Contact( #pHsMx_Seg_1 )
      I_Contact( #pHsMx_Seg_2 )
      Contact( #MemoRemontando )
      wire#w1
      S_SR(operand := #Mx_ET85, r1 := #Mx_ET86)
   END_RUNG
   RUNG wire#powerrail
      Contact( #Mx_ET22 )
      Contact( #Mx_ET121 )
      I_Contact( #Mx_ET21 )
      I_Contact( #Mx_ET120 )
      Contact( #CNT_pHsMx_E2E4.QD )
      I_Contact( #pHsMx_Seg_1 )
      I_Contact( #pHsMx_Seg_2 )
      Contact( #MemoRemontando )
   END_RUNG wire#w1
   // the same network as SCL:
   IF (#Mx_ET12 AND #Mx_ET111 AND NOT #Mx_ET11 AND NOT #Mx_ET110 AND #CNT_pHsMx_E1E3.QD AND NOT #pHsMx_Seg_1 AND NOT #pHsMx_Seg_2 AND #MemoRemontando) OR (#Mx_ET22 AND #Mx_ET121 AND NOT #Mx_ET21 AND NOT #Mx_ET120 AND #CNT_pHsMx_E2E4.QD AND NOT #pHsMx_Seg_1 AND NOT #pHsMx_Seg_2 AND #MemoRemontando) THEN
       #Mx_ET85 := TRUE;   // SR flip-flop
   END_IF;
   IF #Mx_ET86 THEN #Mx_ET85 := FALSE; END_IF;
END_REGION

REGION Network 36: ET81 - CONTROL REMONTADO --> Fase de Aviso de Subida de Paleta
   RUNG wire#powerrail
      Contact( #Mx_ET80 )
      wire#w1
      Contact( #Selec_M2_Entrada )
      wire#w2
      Contact( #AVTF_MEnt )
      Contact( #RH_FinMovimiento )
      Contact( #PasoSalida )
      Contact( #MemoRemontando )
      S_SR(operand := #Mx_ET81, r1 := wire#w3)
   END_RUNG
   RUNG wire#w1
      Contact( #Selec_M4_Entrada )
   END_RUNG wire#w2
   RUNG wire#w1
      Contact( #Selec_M1_Entrada )
   END_RUNG wire#w2
   RUNG wire#w1
      Contact( #Selec_M3_Entrada )
   END_RUNG wire#w2
   RUNG wire#powerrail
      Contact( #Mx_ET10 )
      Contact( #Mx_ET110 )
   END_RUNG wire#w3
   RUNG wire#powerrail
      Contact( #Mx_ET20 )
      Contact( #Mx_ET120 )
   END_RUNG wire#w3
   // the same network as SCL:
   IF #Mx_ET80 AND (#Selec_M2_Entrada OR #Selec_M4_Entrada OR #Selec_M1_Entrada OR #Selec_M3_Entrada) AND #AVTF_MEnt AND #RH_FinMovimiento AND #PasoSalida AND #MemoRemontando THEN
       #Mx_ET81 := TRUE;   // SR flip-flop
   END_IF;
   IF (#Mx_ET10 AND #Mx_ET110) OR (#Mx_ET20 AND #Mx_ET120) THEN #Mx_ET81 := FALSE; END_IF;
END_REGION

REGION Network 37: ET80
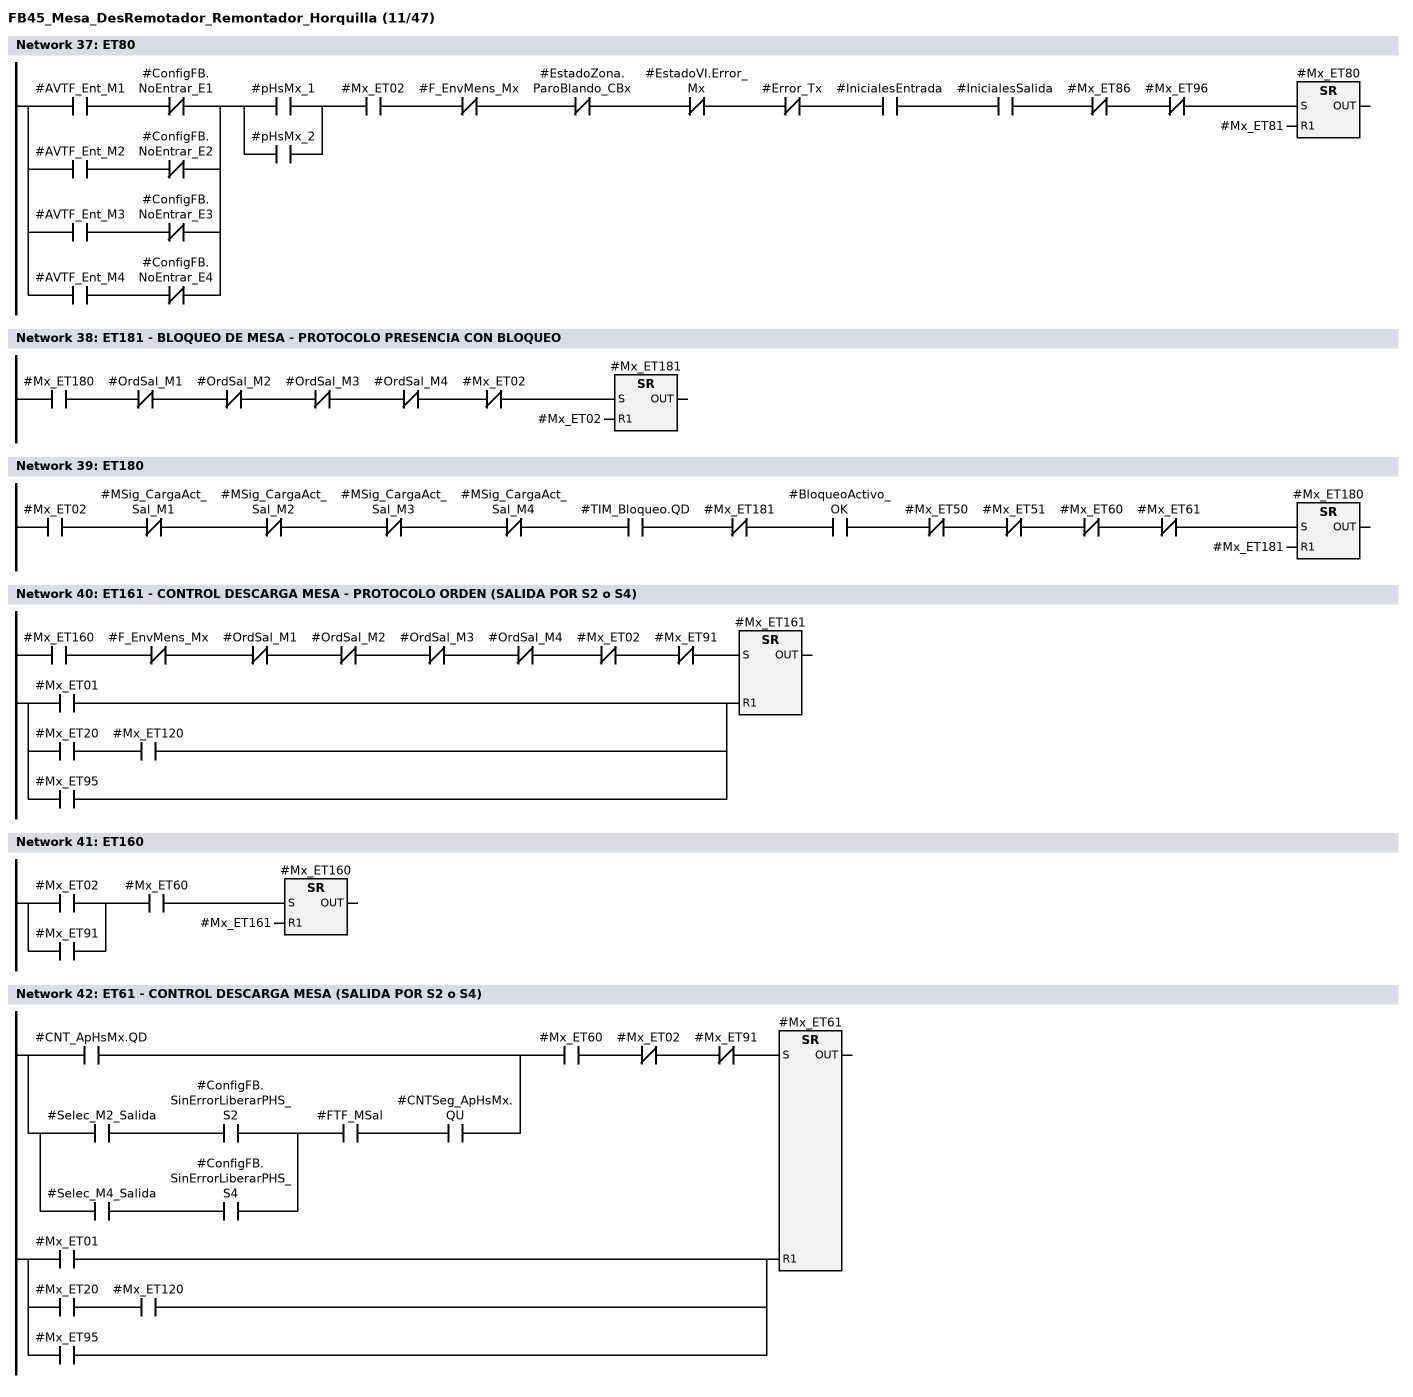
   RUNG wire#powerrail
      Contact( #AVTF_Ent_M1 )
      I_Contact( #ConfigFB.NoEntrar_E1 )
      wire#w1
      Contact( #pHsMx_1 )
      wire#w2
      Contact( #Mx_ET02 )
      I_Contact( #F_EnvMens_Mx )
      I_Contact( #EstadoZona.ParoBlando_CBx )
      I_Contact( #EstadoVI.Error_Mx )
      I_Contact( #Error_Tx )
      Contact( #InicialesEntrada )
      Contact( #InicialesSalida )
      I_Contact( #Mx_ET86 )
      I_Contact( #Mx_ET96 )
      S_SR(operand := #Mx_ET80, r1 := #Mx_ET81)
   END_RUNG
   RUNG wire#powerrail
      Contact( #AVTF_Ent_M2 )
      I_Contact( #ConfigFB.NoEntrar_E2 )
   END_RUNG wire#w1
   RUNG wire#powerrail
      Contact( #AVTF_Ent_M3 )
      I_Contact( #ConfigFB.NoEntrar_E3 )
   END_RUNG wire#w1
   RUNG wire#powerrail
      Contact( #AVTF_Ent_M4 )
      I_Contact( #ConfigFB.NoEntrar_E4 )
   END_RUNG wire#w1
   RUNG wire#w1
      Contact( #pHsMx_2 )
   END_RUNG wire#w2
   // the same network as SCL:
   IF ((#AVTF_Ent_M1 AND NOT #ConfigFB.NoEntrar_E1) OR (#AVTF_Ent_M2 AND NOT #ConfigFB.NoEntrar_E2) OR (#AVTF_Ent_M3 AND NOT #ConfigFB.NoEntrar_E3) OR (#AVTF_Ent_M4 AND NOT #ConfigFB.NoEntrar_E4)) AND (#pHsMx_1 OR #pHsMx_2) AND #Mx_ET02 AND NOT #F_EnvMens_Mx AND NOT #EstadoZona.ParoBlando_CBx AND NOT #EstadoVI.Error_Mx AND NOT #Error_Tx AND #InicialesEntrada AND #InicialesSalida AND NOT #Mx_ET86 AND NOT #Mx_ET96 THEN
       #Mx_ET80 := TRUE;   // SR flip-flop
   END_IF;
   IF #Mx_ET81 THEN #Mx_ET80 := FALSE; END_IF;
END_REGION

REGION Network 38: ET181 - BLOQUEO DE MESA - PROTOCOLO PRESENCIA CON BLOQUEO
   RUNG wire#powerrail
      Contact( #Mx_ET180 )
      I_Contact( #OrdSal_M1 )
      I_Contact( #OrdSal_M2 )
      I_Contact( #OrdSal_M3 )
      I_Contact( #OrdSal_M4 )
      I_Contact( #Mx_ET02 )
      S_SR(operand := #Mx_ET181, r1 := #Mx_ET02)
   END_RUNG
   // the same network as SCL:
   IF #Mx_ET180 AND NOT #OrdSal_M1 AND NOT #OrdSal_M2 AND NOT #OrdSal_M3 AND NOT #OrdSal_M4 AND NOT #Mx_ET02 THEN
       #Mx_ET181 := TRUE;   // SR flip-flop
   END_IF;
   IF #Mx_ET02 THEN #Mx_ET181 := FALSE; END_IF;
END_REGION

REGION Network 39: ET180
   RUNG wire#powerrail
      Contact( #Mx_ET02 )
      I_Contact( #MSig_CargaAct_Sal_M1 )
      I_Contact( #MSig_CargaAct_Sal_M2 )
      I_Contact( #MSig_CargaAct_Sal_M3 )
      I_Contact( #MSig_CargaAct_Sal_M4 )
      Contact( #TIM_Bloqueo.QD )
      I_Contact( #Mx_ET181 )
      Contact( #BloqueoActivo_OK )
      I_Contact( #Mx_ET50 )
      I_Contact( #Mx_ET51 )
      I_Contact( #Mx_ET60 )
      I_Contact( #Mx_ET61 )
      S_SR(operand := #Mx_ET180, r1 := #Mx_ET181)
   END_RUNG
   // the same network as SCL:
   IF #Mx_ET02 AND NOT #MSig_CargaAct_Sal_M1 AND NOT #MSig_CargaAct_Sal_M2 AND NOT #MSig_CargaAct_Sal_M3 AND NOT #MSig_CargaAct_Sal_M4 AND #TIM_Bloqueo.QD AND NOT #Mx_ET181 AND #BloqueoActivo_OK AND NOT #Mx_ET50 AND NOT #Mx_ET51 AND NOT #Mx_ET60 AND NOT #Mx_ET61 THEN
       #Mx_ET180 := TRUE;   // SR flip-flop
   END_IF;
   IF #Mx_ET181 THEN #Mx_ET180 := FALSE; END_IF;
END_REGION

REGION Network 40: ET161 - CONTROL DESCARGA MESA - PROTOCOLO ORDEN (SALIDA POR S2 o S4)
   RUNG wire#powerrail
      Contact( #Mx_ET160 )
      I_Contact( #F_EnvMens_Mx )
      I_Contact( #OrdSal_M1 )
      I_Contact( #OrdSal_M2 )
      I_Contact( #OrdSal_M3 )
      I_Contact( #OrdSal_M4 )
      I_Contact( #Mx_ET02 )
      I_Contact( #Mx_ET91 )
      S_SR(operand := #Mx_ET161, r1 := wire#w1)
   END_RUNG
   RUNG wire#powerrail
      Contact( #Mx_ET01 )
   END_RUNG wire#w1
   RUNG wire#powerrail
      Contact( #Mx_ET20 )
      Contact( #Mx_ET120 )
   END_RUNG wire#w1
   RUNG wire#powerrail
      Contact( #Mx_ET95 )
   END_RUNG wire#w1
   // the same network as SCL:
   IF #Mx_ET160 AND NOT #F_EnvMens_Mx AND NOT #OrdSal_M1 AND NOT #OrdSal_M2 AND NOT #OrdSal_M3 AND NOT #OrdSal_M4 AND NOT #Mx_ET02 AND NOT #Mx_ET91 THEN
       #Mx_ET161 := TRUE;   // SR flip-flop
   END_IF;
   IF #Mx_ET01 OR (#Mx_ET20 AND #Mx_ET120) OR #Mx_ET95 THEN #Mx_ET161 := FALSE; END_IF;
END_REGION

REGION Network 41: ET160
   RUNG wire#powerrail
      Contact( #Mx_ET02 )
      wire#w1
      Contact( #Mx_ET60 )
      S_SR(operand := #Mx_ET160, r1 := #Mx_ET161)
   END_RUNG
   RUNG wire#powerrail
      Contact( #Mx_ET91 )
   END_RUNG wire#w1
   // the same network as SCL:
   IF (#Mx_ET02 OR #Mx_ET91) AND #Mx_ET60 THEN
       #Mx_ET160 := TRUE;   // SR flip-flop
   END_IF;
   IF #Mx_ET161 THEN #Mx_ET160 := FALSE; END_IF;
END_REGION

REGION Network 42: ET61 - CONTROL DESCARGA MESA (SALIDA POR S2 o S4)
   RUNG wire#powerrail
      Contact( #CNT_ApHsMx.QD )
      wire#w1
      Contact( #Mx_ET60 )
      I_Contact( #Mx_ET02 )
      I_Contact( #Mx_ET91 )
      S_SR(operand := #Mx_ET61, r1 := wire#w3)
   END_RUNG
   RUNG wire#powerrail
      Contact( #Selec_M2_Salida )
      Contact( #ConfigFB.SinErrorLiberarPHS_S2 )
      wire#w2
      Contact( #FTF_MSal )
      Contact( #CNTSeg_ApHsMx.QU )
   END_RUNG wire#w1
   RUNG wire#powerrail
      Contact( #Selec_M4_Salida )
      Contact( #ConfigFB.SinErrorLiberarPHS_S4 )
   END_RUNG wire#w2
   RUNG wire#powerrail
      Contact( #Mx_ET01 )
   END_RUNG wire#w3
   RUNG wire#powerrail
      Contact( #Mx_ET20 )
      Contact( #Mx_ET120 )
   END_RUNG wire#w3
   RUNG wire#powerrail
      Contact( #Mx_ET95 )
   END_RUNG wire#w3
   // the same network as SCL:
   IF (#CNT_ApHsMx.QD OR (((#Selec_M2_Salida AND #ConfigFB.SinErrorLiberarPHS_S2) OR (#Selec_M4_Salida AND #ConfigFB.SinErrorLiberarPHS_S4)) AND #FTF_MSal AND #CNTSeg_ApHsMx.QU)) AND #Mx_ET60 AND NOT #Mx_ET02 AND NOT #Mx_ET91 THEN
       #Mx_ET61 := TRUE;   // SR flip-flop
   END_IF;
   IF #Mx_ET01 OR (#Mx_ET20 AND #Mx_ET120) OR #Mx_ET95 THEN #Mx_ET61 := FALSE; END_IF;
END_REGION

REGION Network 43: ET60
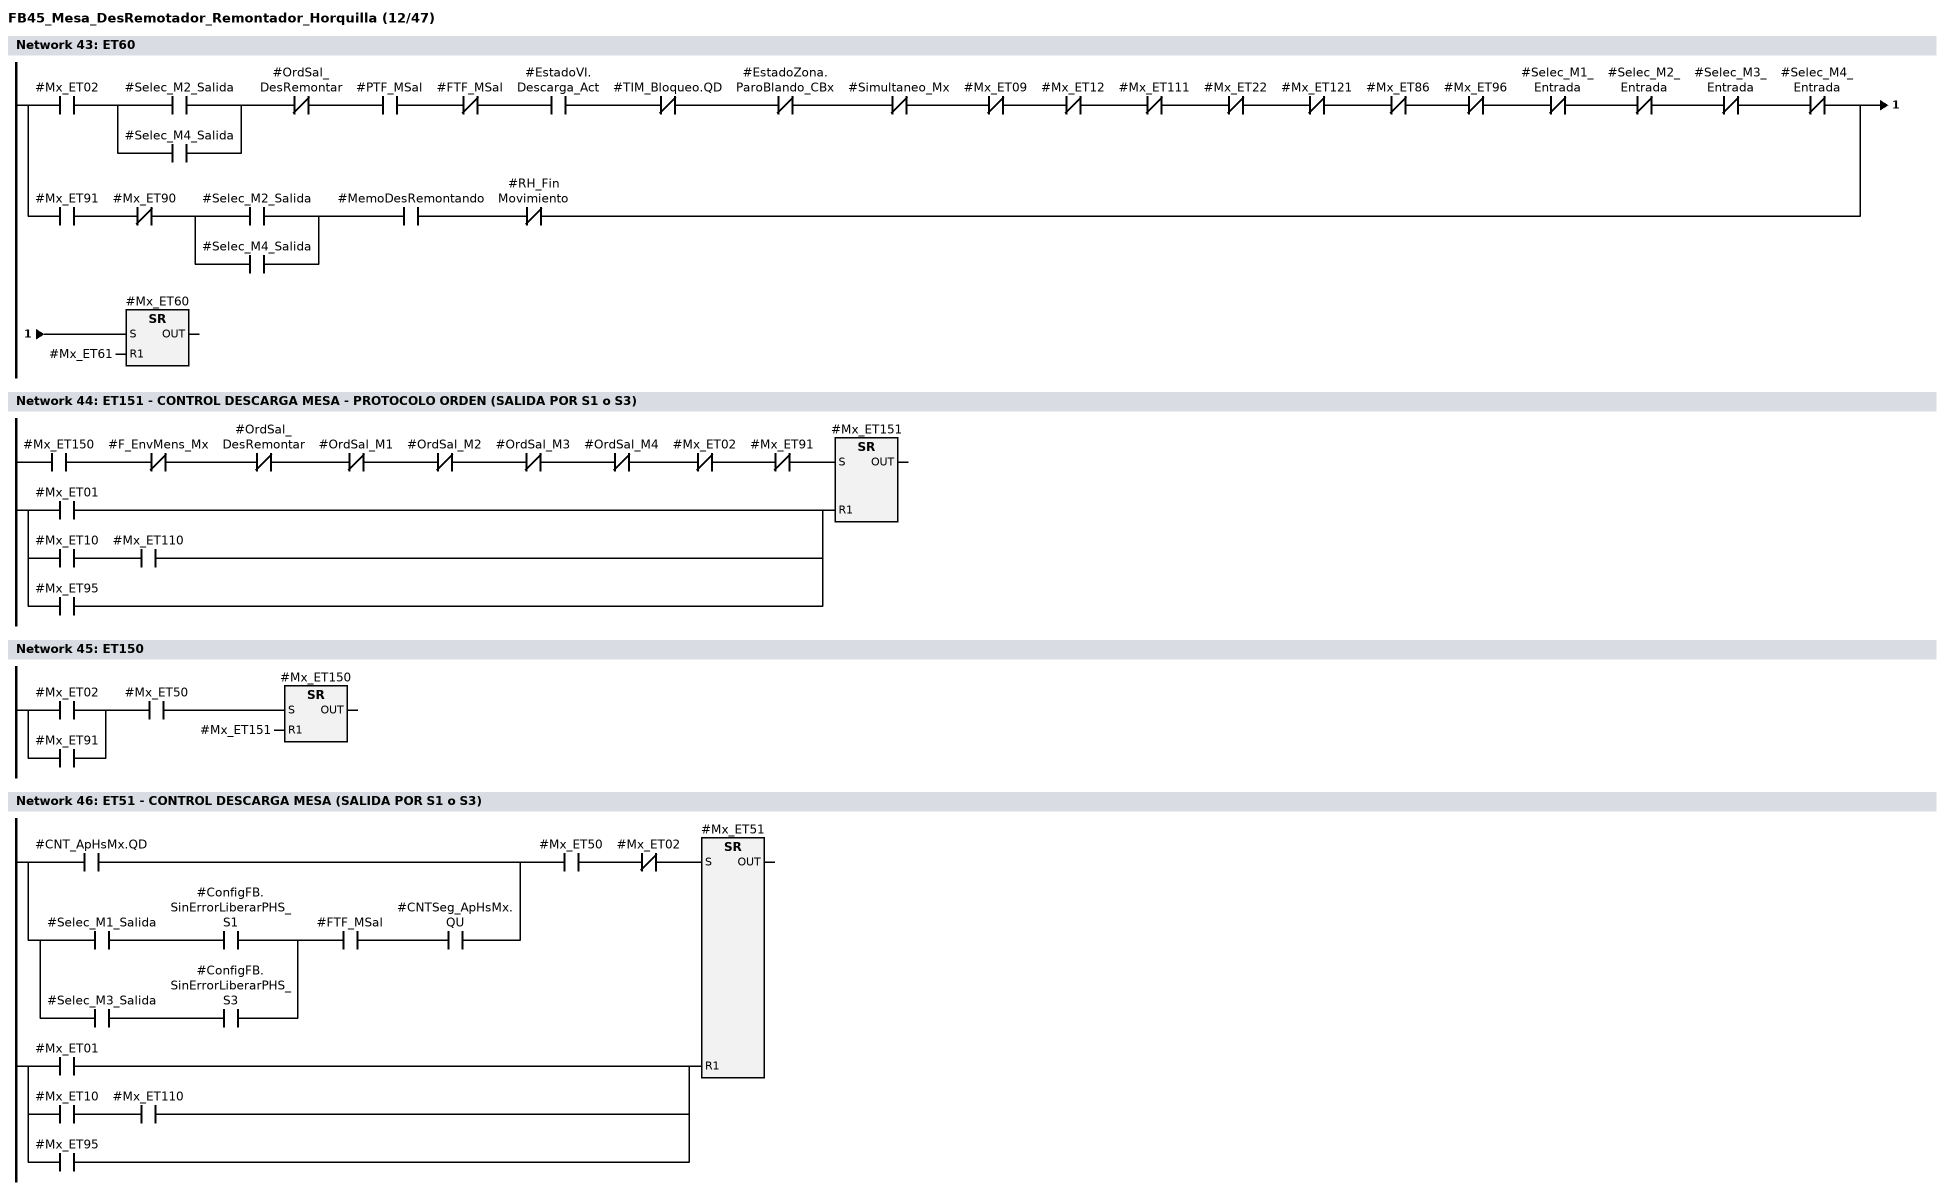
   RUNG wire#powerrail
      Contact( #Mx_ET02 )
      wire#w1
      Contact( #Selec_M2_Salida )
      wire#w2
      I_Contact( #OrdSal_DesRemontar )
      Contact( #PTF_MSal )
      I_Contact( #FTF_MSal )
      Contact( #EstadoVI.Descarga_Act )
      I_Contact( #TIM_Bloqueo.QD )
      I_Contact( #EstadoZona.ParoBlando_CBx )
      I_Contact( #Simultaneo_Mx )
      I_Contact( #Mx_ET09 )
      I_Contact( #Mx_ET12 )
      I_Contact( #Mx_ET111 )
      I_Contact( #Mx_ET22 )
      I_Contact( #Mx_ET121 )
      I_Contact( #Mx_ET86 )
      I_Contact( #Mx_ET96 )
      I_Contact( #Selec_M1_Entrada )
      I_Contact( #Selec_M2_Entrada )
      I_Contact( #Selec_M3_Entrada )
      I_Contact( #Selec_M4_Entrada )
      wire#w3
      S_SR(operand := #Mx_ET60, r1 := #Mx_ET61)
   END_RUNG
   RUNG wire#w1
      Contact( #Selec_M4_Salida )
   END_RUNG wire#w2
   RUNG wire#powerrail
      Contact( #Mx_ET91 )
      I_Contact( #Mx_ET90 )
      wire#w4
      Contact( #Selec_M2_Salida )
      wire#w5
      Contact( #MemoDesRemontando )
      I_Contact( #RH_FinMovimiento )
   END_RUNG wire#w3
   RUNG wire#w4
      Contact( #Selec_M4_Salida )
   END_RUNG wire#w5
   // the same network as SCL:
   IF (#Mx_ET02 AND (#Selec_M2_Salida OR #Selec_M4_Salida) AND NOT #OrdSal_DesRemontar AND #PTF_MSal AND NOT #FTF_MSal AND #EstadoVI.Descarga_Act AND NOT #TIM_Bloqueo.QD AND NOT #EstadoZona.ParoBlando_CBx AND NOT #Simultaneo_Mx AND NOT #Mx_ET09 AND NOT #Mx_ET12 AND NOT #Mx_ET111 AND NOT #Mx_ET22 AND NOT #Mx_ET121 AND NOT #Mx_ET86 AND NOT #Mx_ET96 AND NOT #Selec_M1_Entrada AND NOT #Selec_M2_Entrada AND NOT #Selec_M3_Entrada AND NOT #Selec_M4_Entrada) OR (#Mx_ET91 AND NOT #Mx_ET90 AND (#Selec_M2_Salida OR #Selec_M4_Salida) AND #MemoDesRemontando AND NOT #RH_FinMovimiento) THEN
       #Mx_ET60 := TRUE;   // SR flip-flop
   END_IF;
   IF #Mx_ET61 THEN #Mx_ET60 := FALSE; END_IF;
END_REGION

REGION Network 44: ET151 - CONTROL DESCARGA MESA - PROTOCOLO ORDEN (SALIDA POR S1 o S3)
   RUNG wire#powerrail
      Contact( #Mx_ET150 )
      I_Contact( #F_EnvMens_Mx )
      I_Contact( #OrdSal_DesRemontar )
      I_Contact( #OrdSal_M1 )
      I_Contact( #OrdSal_M2 )
      I_Contact( #OrdSal_M3 )
      I_Contact( #OrdSal_M4 )
      I_Contact( #Mx_ET02 )
      I_Contact( #Mx_ET91 )
      S_SR(operand := #Mx_ET151, r1 := wire#w1)
   END_RUNG
   RUNG wire#powerrail
      Contact( #Mx_ET01 )
   END_RUNG wire#w1
   RUNG wire#powerrail
      Contact( #Mx_ET10 )
      Contact( #Mx_ET110 )
   END_RUNG wire#w1
   RUNG wire#powerrail
      Contact( #Mx_ET95 )
   END_RUNG wire#w1
   // the same network as SCL:
   IF #Mx_ET150 AND NOT #F_EnvMens_Mx AND NOT #OrdSal_DesRemontar AND NOT #OrdSal_M1 AND NOT #OrdSal_M2 AND NOT #OrdSal_M3 AND NOT #OrdSal_M4 AND NOT #Mx_ET02 AND NOT #Mx_ET91 THEN
       #Mx_ET151 := TRUE;   // SR flip-flop
   END_IF;
   IF #Mx_ET01 OR (#Mx_ET10 AND #Mx_ET110) OR #Mx_ET95 THEN #Mx_ET151 := FALSE; END_IF;
END_REGION

REGION Network 45: ET150
   RUNG wire#powerrail
      Contact( #Mx_ET02 )
      wire#w1
      Contact( #Mx_ET50 )
      S_SR(operand := #Mx_ET150, r1 := #Mx_ET151)
   END_RUNG
   RUNG wire#powerrail
      Contact( #Mx_ET91 )
   END_RUNG wire#w1
   // the same network as SCL:
   IF (#Mx_ET02 OR #Mx_ET91) AND #Mx_ET50 THEN
       #Mx_ET150 := TRUE;   // SR flip-flop
   END_IF;
   IF #Mx_ET151 THEN #Mx_ET150 := FALSE; END_IF;
END_REGION

REGION Network 46: ET51 - CONTROL DESCARGA MESA (SALIDA POR S1 o S3)
   RUNG wire#powerrail
      Contact( #CNT_ApHsMx.QD )
      wire#w1
      Contact( #Mx_ET50 )
      I_Contact( #Mx_ET02 )
      S_SR(operand := #Mx_ET51, r1 := wire#w3)
   END_RUNG
   RUNG wire#powerrail
      Contact( #Selec_M1_Salida )
      Contact( #ConfigFB.SinErrorLiberarPHS_S1 )
      wire#w2
      Contact( #FTF_MSal )
      Contact( #CNTSeg_ApHsMx.QU )
   END_RUNG wire#w1
   RUNG wire#powerrail
      Contact( #Selec_M3_Salida )
      Contact( #ConfigFB.SinErrorLiberarPHS_S3 )
   END_RUNG wire#w2
   RUNG wire#powerrail
      Contact( #Mx_ET01 )
   END_RUNG wire#w3
   RUNG wire#powerrail
      Contact( #Mx_ET10 )
      Contact( #Mx_ET110 )
   END_RUNG wire#w3
   RUNG wire#powerrail
      Contact( #Mx_ET95 )
   END_RUNG wire#w3
   // the same network as SCL:
   IF (#CNT_ApHsMx.QD OR (((#Selec_M1_Salida AND #ConfigFB.SinErrorLiberarPHS_S1) OR (#Selec_M3_Salida AND #ConfigFB.SinErrorLiberarPHS_S3)) AND #FTF_MSal AND #CNTSeg_ApHsMx.QU)) AND #Mx_ET50 AND NOT #Mx_ET02 THEN
       #Mx_ET51 := TRUE;   // SR flip-flop
   END_IF;
   IF #Mx_ET01 OR (#Mx_ET10 AND #Mx_ET110) OR #Mx_ET95 THEN #Mx_ET51 := FALSE; END_IF;
END_REGION

REGION Network 47: ET50
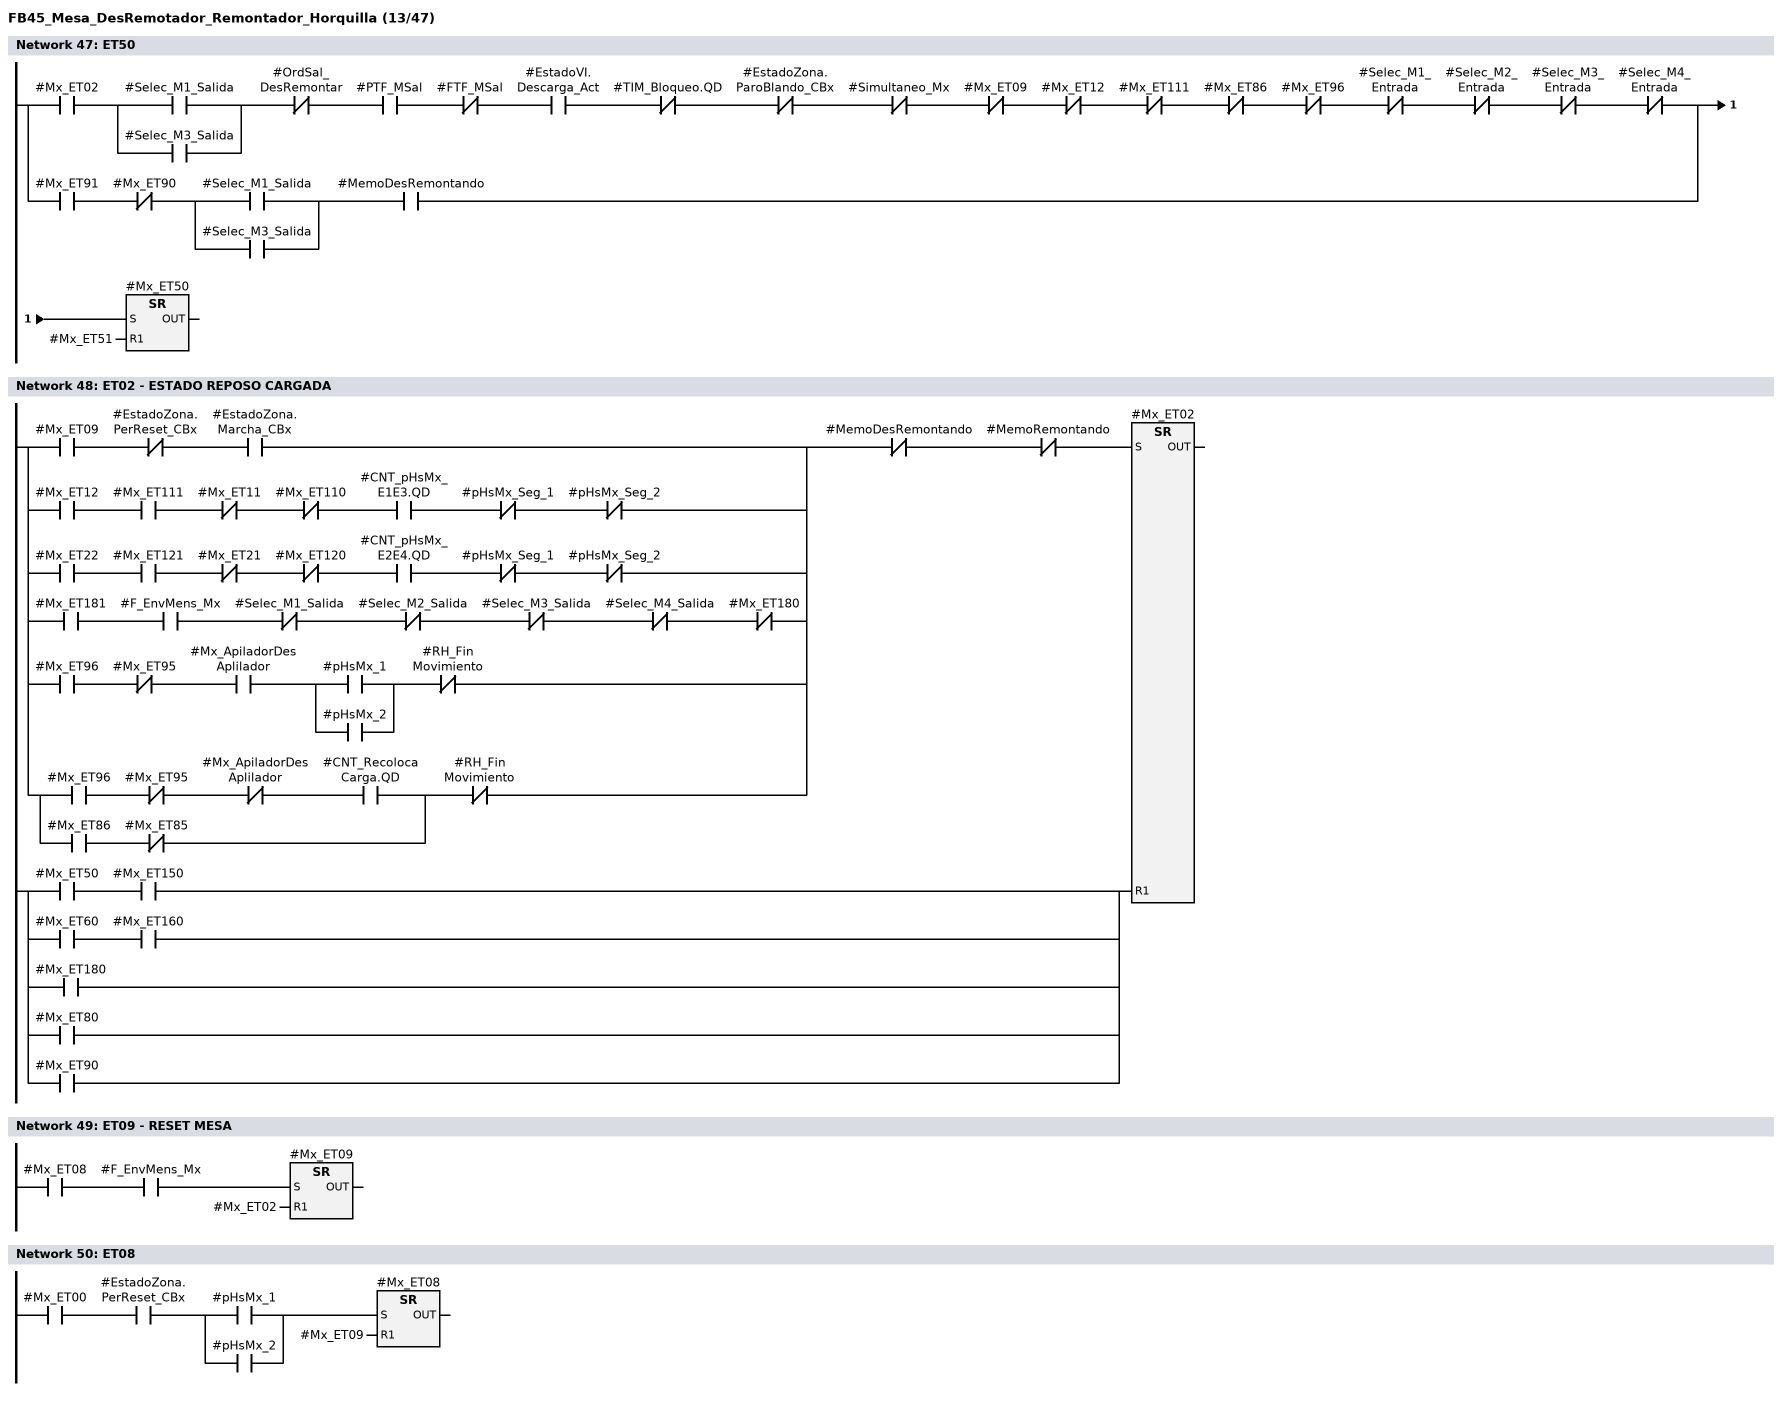
   RUNG wire#powerrail
      Contact( #Mx_ET02 )
      wire#w1
      Contact( #Selec_M1_Salida )
      wire#w2
      I_Contact( #OrdSal_DesRemontar )
      Contact( #PTF_MSal )
      I_Contact( #FTF_MSal )
      Contact( #EstadoVI.Descarga_Act )
      I_Contact( #TIM_Bloqueo.QD )
      I_Contact( #EstadoZona.ParoBlando_CBx )
      I_Contact( #Simultaneo_Mx )
      I_Contact( #Mx_ET09 )
      I_Contact( #Mx_ET12 )
      I_Contact( #Mx_ET111 )
      I_Contact( #Mx_ET86 )
      I_Contact( #Mx_ET96 )
      I_Contact( #Selec_M1_Entrada )
      I_Contact( #Selec_M2_Entrada )
      I_Contact( #Selec_M3_Entrada )
      I_Contact( #Selec_M4_Entrada )
      wire#w3
      S_SR(operand := #Mx_ET50, r1 := #Mx_ET51)
   END_RUNG
   RUNG wire#w1
      Contact( #Selec_M3_Salida )
   END_RUNG wire#w2
   RUNG wire#powerrail
      Contact( #Mx_ET91 )
      I_Contact( #Mx_ET90 )
      wire#w4
      Contact( #Selec_M1_Salida )
      wire#w5
      Contact( #MemoDesRemontando )
   END_RUNG wire#w3
   RUNG wire#w4
      Contact( #Selec_M3_Salida )
   END_RUNG wire#w5
   // the same network as SCL:
   IF (#Mx_ET02 AND (#Selec_M1_Salida OR #Selec_M3_Salida) AND NOT #OrdSal_DesRemontar AND #PTF_MSal AND NOT #FTF_MSal AND #EstadoVI.Descarga_Act AND NOT #TIM_Bloqueo.QD AND NOT #EstadoZona.ParoBlando_CBx AND NOT #Simultaneo_Mx AND NOT #Mx_ET09 AND NOT #Mx_ET12 AND NOT #Mx_ET111 AND NOT #Mx_ET86 AND NOT #Mx_ET96 AND NOT #Selec_M1_Entrada AND NOT #Selec_M2_Entrada AND NOT #Selec_M3_Entrada AND NOT #Selec_M4_Entrada) OR (#Mx_ET91 AND NOT #Mx_ET90 AND (#Selec_M1_Salida OR #Selec_M3_Salida) AND #MemoDesRemontando) THEN
       #Mx_ET50 := TRUE;   // SR flip-flop
   END_IF;
   IF #Mx_ET51 THEN #Mx_ET50 := FALSE; END_IF;
END_REGION

REGION Network 48: ET02 - ESTADO REPOSO CARGADA
   RUNG wire#powerrail
      Contact( #Mx_ET09 )
      I_Contact( #EstadoZona.PerReset_CBx )
      Contact( #EstadoZona.Marcha_CBx )
      wire#w1
      I_Contact( #MemoDesRemontando )
      I_Contact( #MemoRemontando )
      S_SR(operand := #Mx_ET02, r1 := wire#w5)
   END_RUNG
   RUNG wire#powerrail
      Contact( #Mx_ET12 )
      Contact( #Mx_ET111 )
      I_Contact( #Mx_ET11 )
      I_Contact( #Mx_ET110 )
      Contact( #CNT_pHsMx_E1E3.QD )
      I_Contact( #pHsMx_Seg_1 )
      I_Contact( #pHsMx_Seg_2 )
   END_RUNG wire#w1
   RUNG wire#powerrail
      Contact( #Mx_ET22 )
      Contact( #Mx_ET121 )
      I_Contact( #Mx_ET21 )
      I_Contact( #Mx_ET120 )
      Contact( #CNT_pHsMx_E2E4.QD )
      I_Contact( #pHsMx_Seg_1 )
      I_Contact( #pHsMx_Seg_2 )
   END_RUNG wire#w1
   RUNG wire#powerrail
      Contact( #Mx_ET181 )
      Contact( #F_EnvMens_Mx )
      I_Contact( #Selec_M1_Salida )
      I_Contact( #Selec_M2_Salida )
      I_Contact( #Selec_M3_Salida )
      I_Contact( #Selec_M4_Salida )
      I_Contact( #Mx_ET180 )
   END_RUNG wire#w1
   RUNG wire#powerrail
      Contact( #Mx_ET96 )
      I_Contact( #Mx_ET95 )
      Contact( #Mx_ApiladorDesAplilador )
      wire#w2
      Contact( #pHsMx_1 )
      wire#w3
      I_Contact( #RH_FinMovimiento )
   END_RUNG wire#w1
   RUNG wire#w2
      Contact( #pHsMx_2 )
   END_RUNG wire#w3
   RUNG wire#powerrail
      Contact( #Mx_ET96 )
      I_Contact( #Mx_ET95 )
      I_Contact( #Mx_ApiladorDesAplilador )
      Contact( #CNT_RecolocaCarga.QD )
      wire#w4
      I_Contact( #RH_FinMovimiento )
   END_RUNG wire#w1
   RUNG wire#powerrail
      Contact( #Mx_ET86 )
      I_Contact( #Mx_ET85 )
   END_RUNG wire#w4
   RUNG wire#powerrail
      Contact( #Mx_ET50 )
      Contact( #Mx_ET150 )
   END_RUNG wire#w5
   RUNG wire#powerrail
      Contact( #Mx_ET60 )
      Contact( #Mx_ET160 )
   END_RUNG wire#w5
   RUNG wire#powerrail
      Contact( #Mx_ET180 )
   END_RUNG wire#w5
   RUNG wire#powerrail
      Contact( #Mx_ET80 )
   END_RUNG wire#w5
   RUNG wire#powerrail
      Contact( #Mx_ET90 )
   END_RUNG wire#w5
   // the same network as SCL:
   IF ((#Mx_ET09 AND NOT #EstadoZona.PerReset_CBx AND #EstadoZona.Marcha_CBx) OR (#Mx_ET12 AND #Mx_ET111 AND NOT #Mx_ET11 AND NOT #Mx_ET110 AND #CNT_pHsMx_E1E3.QD AND NOT #pHsMx_Seg_1 AND NOT #pHsMx_Seg_2) OR (#Mx_ET22 AND #Mx_ET121 AND NOT #Mx_ET21 AND NOT #Mx_ET120 AND #CNT_pHsMx_E2E4.QD AND NOT #pHsMx_Seg_1 AND NOT #pHsMx_Seg_2) OR (#Mx_ET181 AND #F_EnvMens_Mx AND NOT #Selec_M1_Salida AND NOT #Selec_M2_Salida AND NOT #Selec_M3_Salida AND NOT #Selec_M4_Salida AND NOT #Mx_ET180) OR (#Mx_ET96 AND NOT #Mx_ET95 AND #Mx_ApiladorDesAplilador AND (#pHsMx_1 OR #pHsMx_2) AND NOT #RH_FinMovimiento) OR (((#Mx_ET96 AND NOT #Mx_ET95 AND NOT #Mx_ApiladorDesAplilador AND #CNT_RecolocaCarga.QD) OR (#Mx_ET86 AND NOT #Mx_ET85)) AND NOT #RH_FinMovimiento)) AND NOT #MemoDesRemontando AND NOT #MemoRemontando THEN
       #Mx_ET02 := TRUE;   // SR flip-flop
   END_IF;
   IF (#Mx_ET50 AND #Mx_ET150) OR (#Mx_ET60 AND #Mx_ET160) OR #Mx_ET180 OR #Mx_ET80 OR #Mx_ET90 THEN
       #Mx_ET02 := FALSE;
   END_IF;
END_REGION

REGION Network 49: ET09 - RESET MESA
   RUNG wire#powerrail
      Contact( #Mx_ET08 )
      Contact( #F_EnvMens_Mx )
      S_SR(operand := #Mx_ET09, r1 := #Mx_ET02)
   END_RUNG
   // the same network as SCL:
   IF #Mx_ET08 AND #F_EnvMens_Mx THEN
       #Mx_ET09 := TRUE;   // SR flip-flop
   END_IF;
   IF #Mx_ET02 THEN #Mx_ET09 := FALSE; END_IF;
END_REGION

REGION Network 50: ET08
   RUNG wire#powerrail
      Contact( #Mx_ET00 )
      Contact( #EstadoZona.PerReset_CBx )
      wire#w1
      Contact( #pHsMx_1 )
      wire#w2
      S_SR(operand := #Mx_ET08, r1 := #Mx_ET09)
   END_RUNG
   RUNG wire#w1
      Contact( #pHsMx_2 )
   END_RUNG wire#w2
   // the same network as SCL:
   IF #Mx_ET00 AND #EstadoZona.PerReset_CBx AND (#pHsMx_1 OR #pHsMx_2) THEN
       #Mx_ET08 := TRUE;   // SR flip-flop
   END_IF;
   IF #Mx_ET09 THEN #Mx_ET08 := FALSE; END_IF;
END_REGION

REGION Network 51: ET121- CONTROL CARGA MESA - MENSAJE DE PRESENCIA (ENTRADA POR E2 o E4)
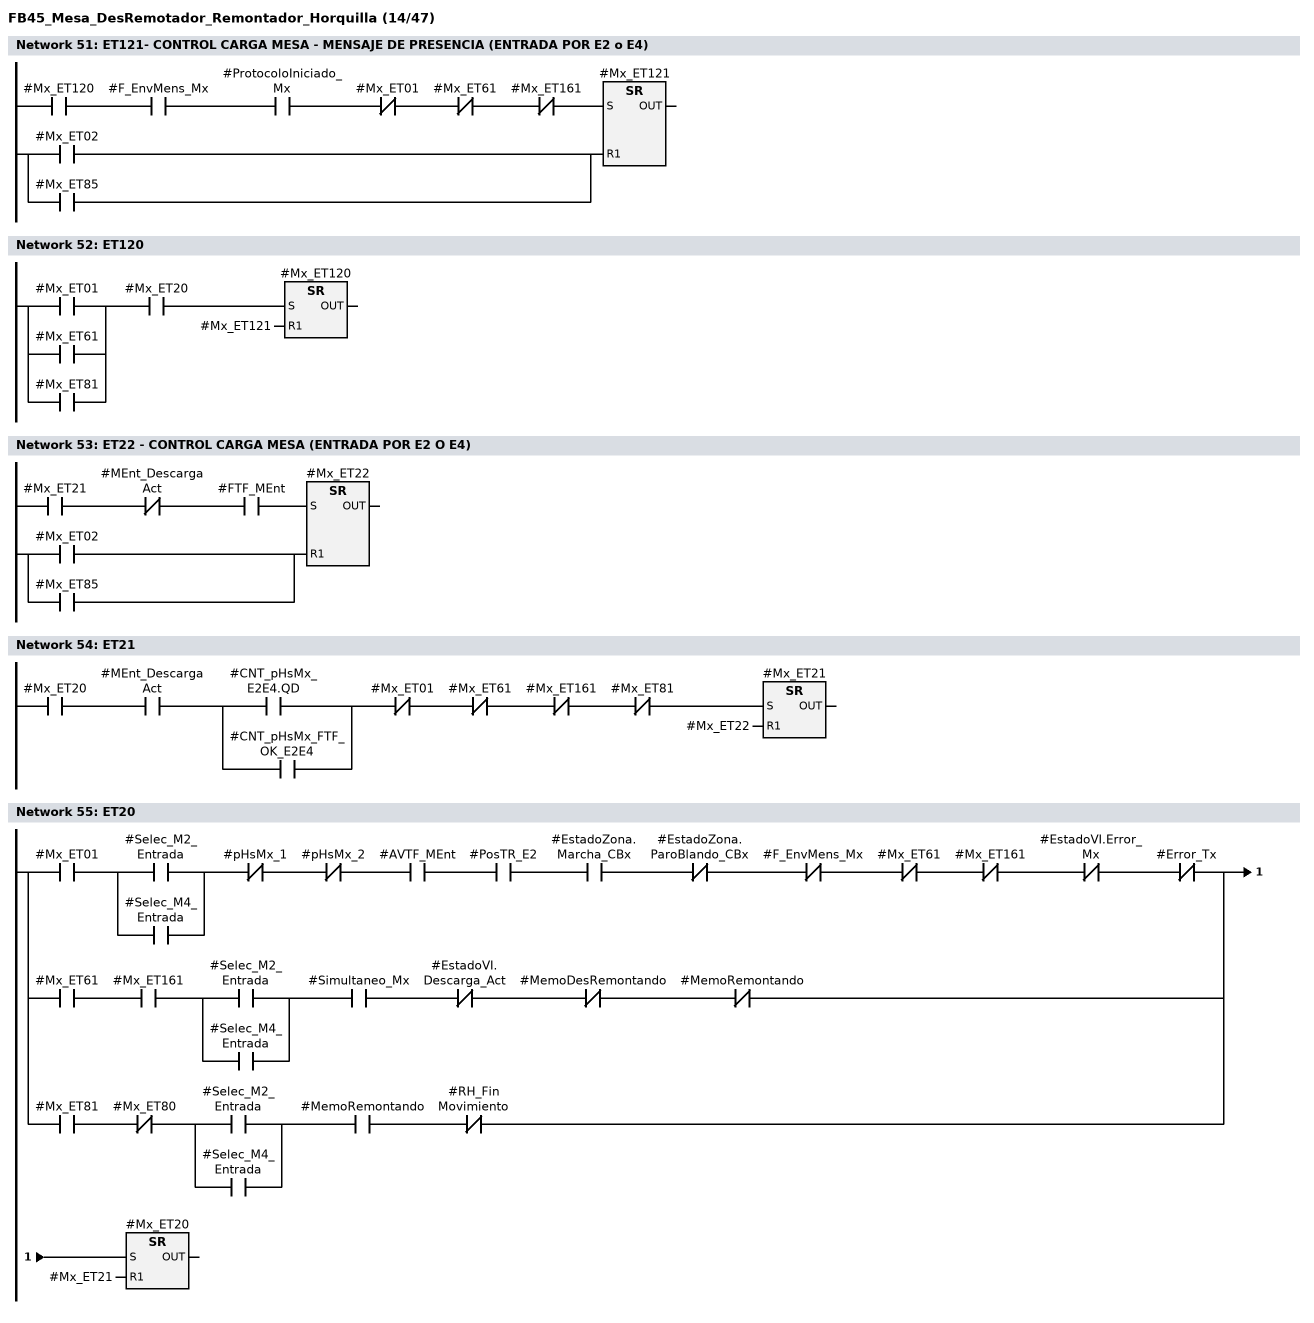
   RUNG wire#powerrail
      Contact( #Mx_ET120 )
      Contact( #F_EnvMens_Mx )
      Contact( #ProtocoloIniciado_Mx )
      I_Contact( #Mx_ET01 )
      I_Contact( #Mx_ET61 )
      I_Contact( #Mx_ET161 )
      S_SR(operand := #Mx_ET121, r1 := wire#w1)
   END_RUNG
   RUNG wire#powerrail
      Contact( #Mx_ET02 )
   END_RUNG wire#w1
   RUNG wire#powerrail
      Contact( #Mx_ET85 )
   END_RUNG wire#w1
   // the same network as SCL:
   IF #Mx_ET120 AND #F_EnvMens_Mx AND #ProtocoloIniciado_Mx AND NOT #Mx_ET01 AND NOT #Mx_ET61 AND NOT #Mx_ET161 THEN
       #Mx_ET121 := TRUE;   // SR flip-flop
   END_IF;
   IF #Mx_ET02 OR #Mx_ET85 THEN #Mx_ET121 := FALSE; END_IF;
END_REGION

REGION Network 52: ET120
   RUNG wire#powerrail
      Contact( #Mx_ET01 )
      wire#w1
      Contact( #Mx_ET20 )
      S_SR(operand := #Mx_ET120, r1 := #Mx_ET121)
   END_RUNG
   RUNG wire#powerrail
      Contact( #Mx_ET61 )
   END_RUNG wire#w1
   RUNG wire#powerrail
      Contact( #Mx_ET81 )
   END_RUNG wire#w1
   // the same network as SCL:
   IF (#Mx_ET01 OR #Mx_ET61 OR #Mx_ET81) AND #Mx_ET20 THEN
       #Mx_ET120 := TRUE;   // SR flip-flop
   END_IF;
   IF #Mx_ET121 THEN #Mx_ET120 := FALSE; END_IF;
END_REGION

REGION Network 53: ET22 - CONTROL CARGA MESA (ENTRADA POR E2 O E4)
   RUNG wire#powerrail
      Contact( #Mx_ET21 )
      I_Contact( #MEnt_DescargaAct )
      Contact( #FTF_MEnt )
      S_SR(operand := #Mx_ET22, r1 := wire#w1)
   END_RUNG
   RUNG wire#powerrail
      Contact( #Mx_ET02 )
   END_RUNG wire#w1
   RUNG wire#powerrail
      Contact( #Mx_ET85 )
   END_RUNG wire#w1
   // the same network as SCL:
   IF #Mx_ET21 AND NOT #MEnt_DescargaAct AND #FTF_MEnt THEN
       #Mx_ET22 := TRUE;   // SR flip-flop
   END_IF;
   IF #Mx_ET02 OR #Mx_ET85 THEN #Mx_ET22 := FALSE; END_IF;
END_REGION

REGION Network 54: ET21
   RUNG wire#powerrail
      Contact( #Mx_ET20 )
      Contact( #MEnt_DescargaAct )
      wire#w1
      Contact( #CNT_pHsMx_E2E4.QD )
      wire#w2
      I_Contact( #Mx_ET01 )
      I_Contact( #Mx_ET61 )
      I_Contact( #Mx_ET161 )
      I_Contact( #Mx_ET81 )
      S_SR(operand := #Mx_ET21, r1 := #Mx_ET22)
   END_RUNG
   RUNG wire#w1
      Contact( #CNT_pHsMx_FTF_OK_E2E4 )
   END_RUNG wire#w2
   // the same network as SCL:
   IF #Mx_ET20 AND #MEnt_DescargaAct AND (#CNT_pHsMx_E2E4.QD OR #CNT_pHsMx_FTF_OK_E2E4) AND NOT #Mx_ET01 AND NOT #Mx_ET61 AND NOT #Mx_ET161 AND NOT #Mx_ET81 THEN
       #Mx_ET21 := TRUE;   // SR flip-flop
   END_IF;
   IF #Mx_ET22 THEN #Mx_ET21 := FALSE; END_IF;
END_REGION

REGION Network 55: ET20
   RUNG wire#powerrail
      Contact( #Mx_ET01 )
      wire#w1
      Contact( #Selec_M2_Entrada )
      wire#w2
      I_Contact( #pHsMx_1 )
      I_Contact( #pHsMx_2 )
      Contact( #AVTF_MEnt )
      Contact( #PosTR_E2 )
      Contact( #EstadoZona.Marcha_CBx )
      I_Contact( #EstadoZona.ParoBlando_CBx )
      I_Contact( #F_EnvMens_Mx )
      I_Contact( #Mx_ET61 )
      I_Contact( #Mx_ET161 )
      I_Contact( #EstadoVI.Error_Mx )
      I_Contact( #Error_Tx )
      wire#w3
      S_SR(operand := #Mx_ET20, r1 := #Mx_ET21)
   END_RUNG
   RUNG wire#w1
      Contact( #Selec_M4_Entrada )
   END_RUNG wire#w2
   RUNG wire#powerrail
      Contact( #Mx_ET61 )
      Contact( #Mx_ET161 )
      wire#w4
      Contact( #Selec_M2_Entrada )
      wire#w5
      Contact( #Simultaneo_Mx )
      I_Contact( #EstadoVI.Descarga_Act )
      I_Contact( #MemoDesRemontando )
      I_Contact( #MemoRemontando )
   END_RUNG wire#w3
   RUNG wire#w4
      Contact( #Selec_M4_Entrada )
   END_RUNG wire#w5
   RUNG wire#powerrail
      Contact( #Mx_ET81 )
      I_Contact( #Mx_ET80 )
      wire#w6
      Contact( #Selec_M2_Entrada )
      wire#w7
      Contact( #MemoRemontando )
      I_Contact( #RH_FinMovimiento )
   END_RUNG wire#w3
   RUNG wire#w6
      Contact( #Selec_M4_Entrada )
   END_RUNG wire#w7
   // the same network as SCL:
   IF (#Mx_ET01 AND (#Selec_M2_Entrada OR #Selec_M4_Entrada) AND NOT #pHsMx_1 AND NOT #pHsMx_2 AND #AVTF_MEnt AND #PosTR_E2 AND #EstadoZona.Marcha_CBx AND NOT #EstadoZona.ParoBlando_CBx AND NOT #F_EnvMens_Mx AND NOT #Mx_ET61 AND NOT #Mx_ET161 AND NOT #EstadoVI.Error_Mx AND NOT #Error_Tx) OR (#Mx_ET61 AND #Mx_ET161 AND (#Selec_M2_Entrada OR #Selec_M4_Entrada) AND #Simultaneo_Mx AND NOT #EstadoVI.Descarga_Act AND NOT #MemoDesRemontando AND NOT #MemoRemontando) OR (#Mx_ET81 AND NOT #Mx_ET80 AND (#Selec_M2_Entrada OR #Selec_M4_Entrada) AND #MemoRemontando AND NOT #RH_FinMovimiento) THEN
       #Mx_ET20 := TRUE;   // SR flip-flop
   END_IF;
   IF #Mx_ET21 THEN #Mx_ET20 := FALSE; END_IF;
END_REGION

REGION Network 56: ET111 - CONTROL CARGA MESA - MENSAJE DE PRESENCIA (ENTRADA POR E1 o E3)
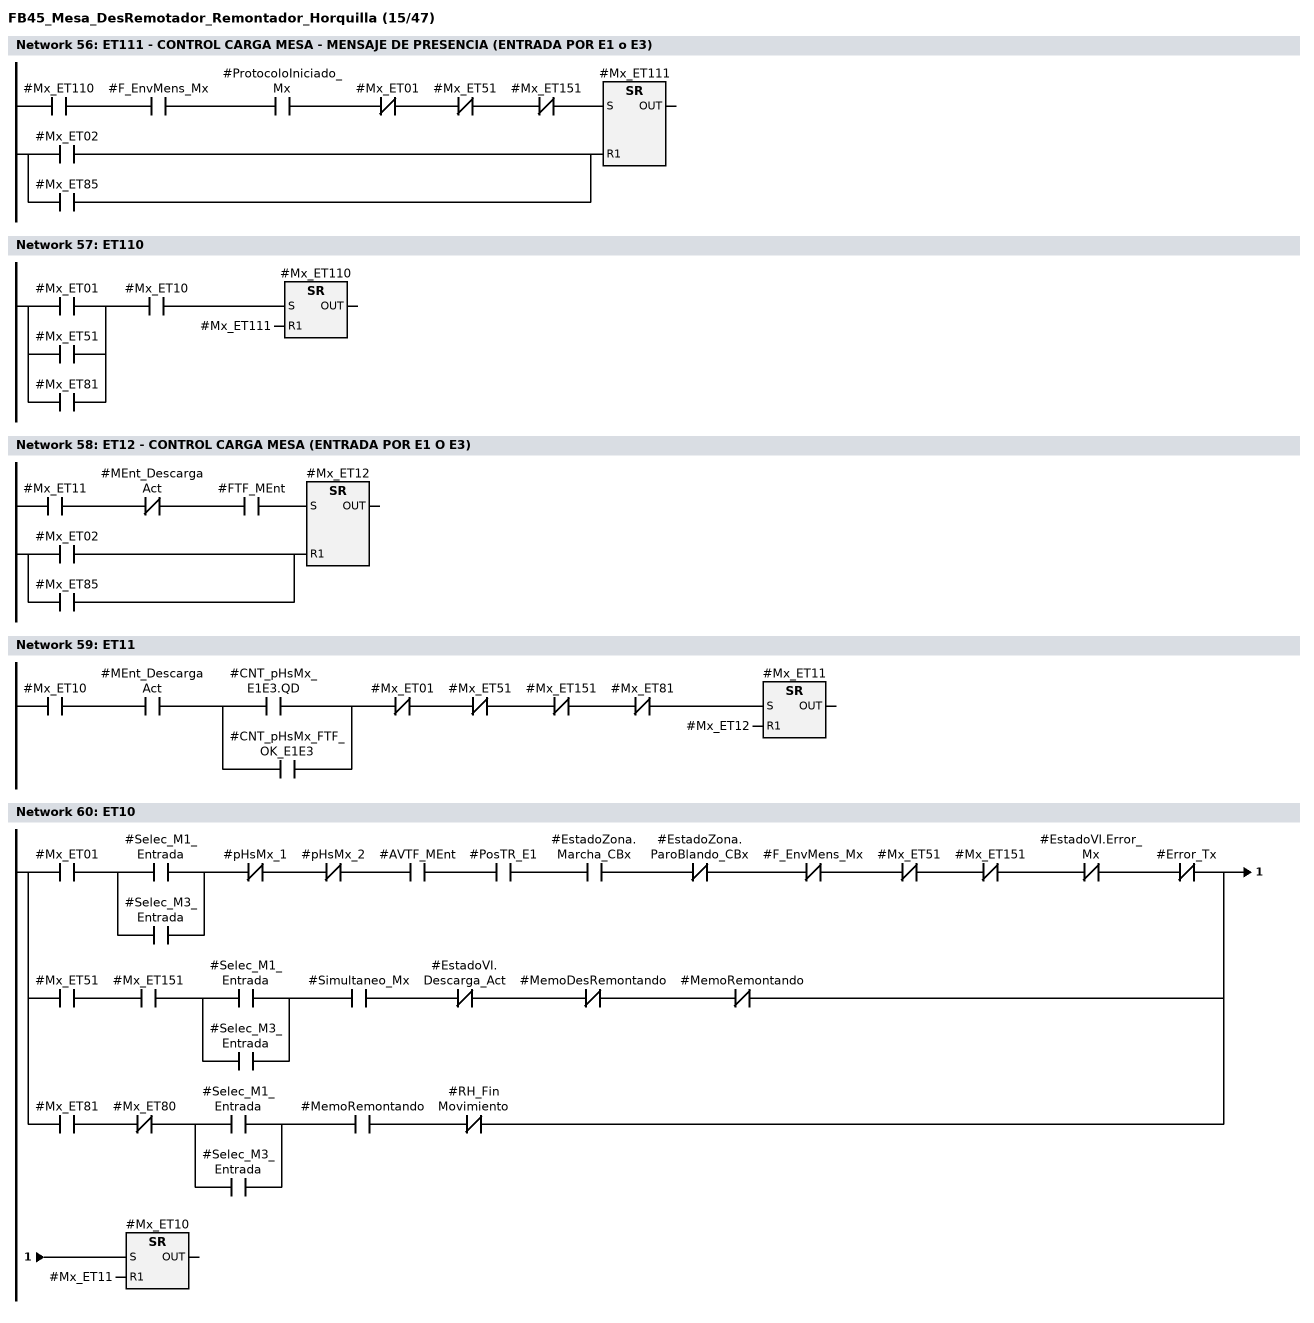
   RUNG wire#powerrail
      Contact( #Mx_ET110 )
      Contact( #F_EnvMens_Mx )
      Contact( #ProtocoloIniciado_Mx )
      I_Contact( #Mx_ET01 )
      I_Contact( #Mx_ET51 )
      I_Contact( #Mx_ET151 )
      S_SR(operand := #Mx_ET111, r1 := wire#w1)
   END_RUNG
   RUNG wire#powerrail
      Contact( #Mx_ET02 )
   END_RUNG wire#w1
   RUNG wire#powerrail
      Contact( #Mx_ET85 )
   END_RUNG wire#w1
   // the same network as SCL:
   IF #Mx_ET110 AND #F_EnvMens_Mx AND #ProtocoloIniciado_Mx AND NOT #Mx_ET01 AND NOT #Mx_ET51 AND NOT #Mx_ET151 THEN
       #Mx_ET111 := TRUE;   // SR flip-flop
   END_IF;
   IF #Mx_ET02 OR #Mx_ET85 THEN #Mx_ET111 := FALSE; END_IF;
END_REGION

REGION Network 57: ET110
   RUNG wire#powerrail
      Contact( #Mx_ET01 )
      wire#w1
      Contact( #Mx_ET10 )
      S_SR(operand := #Mx_ET110, r1 := #Mx_ET111)
   END_RUNG
   RUNG wire#powerrail
      Contact( #Mx_ET51 )
   END_RUNG wire#w1
   RUNG wire#powerrail
      Contact( #Mx_ET81 )
   END_RUNG wire#w1
   // the same network as SCL:
   IF (#Mx_ET01 OR #Mx_ET51 OR #Mx_ET81) AND #Mx_ET10 THEN
       #Mx_ET110 := TRUE;   // SR flip-flop
   END_IF;
   IF #Mx_ET111 THEN #Mx_ET110 := FALSE; END_IF;
END_REGION

REGION Network 58: ET12 - CONTROL CARGA MESA (ENTRADA POR E1 O E3)
   RUNG wire#powerrail
      Contact( #Mx_ET11 )
      I_Contact( #MEnt_DescargaAct )
      Contact( #FTF_MEnt )
      S_SR(operand := #Mx_ET12, r1 := wire#w1)
   END_RUNG
   RUNG wire#powerrail
      Contact( #Mx_ET02 )
   END_RUNG wire#w1
   RUNG wire#powerrail
      Contact( #Mx_ET85 )
   END_RUNG wire#w1
   // the same network as SCL:
   IF #Mx_ET11 AND NOT #MEnt_DescargaAct AND #FTF_MEnt THEN
       #Mx_ET12 := TRUE;   // SR flip-flop
   END_IF;
   IF #Mx_ET02 OR #Mx_ET85 THEN #Mx_ET12 := FALSE; END_IF;
END_REGION

REGION Network 59: ET11
   RUNG wire#powerrail
      Contact( #Mx_ET10 )
      Contact( #MEnt_DescargaAct )
      wire#w1
      Contact( #CNT_pHsMx_E1E3.QD )
      wire#w2
      I_Contact( #Mx_ET01 )
      I_Contact( #Mx_ET51 )
      I_Contact( #Mx_ET151 )
      I_Contact( #Mx_ET81 )
      S_SR(operand := #Mx_ET11, r1 := #Mx_ET12)
   END_RUNG
   RUNG wire#w1
      Contact( #CNT_pHsMx_FTF_OK_E1E3 )
   END_RUNG wire#w2
   // the same network as SCL:
   IF #Mx_ET10 AND #MEnt_DescargaAct AND (#CNT_pHsMx_E1E3.QD OR #CNT_pHsMx_FTF_OK_E1E3) AND NOT #Mx_ET01 AND NOT #Mx_ET51 AND NOT #Mx_ET151 AND NOT #Mx_ET81 THEN
       #Mx_ET11 := TRUE;   // SR flip-flop
   END_IF;
   IF #Mx_ET12 THEN #Mx_ET11 := FALSE; END_IF;
END_REGION

REGION Network 60: ET10
   RUNG wire#powerrail
      Contact( #Mx_ET01 )
      wire#w1
      Contact( #Selec_M1_Entrada )
      wire#w2
      I_Contact( #pHsMx_1 )
      I_Contact( #pHsMx_2 )
      Contact( #AVTF_MEnt )
      Contact( #PosTR_E1 )
      Contact( #EstadoZona.Marcha_CBx )
      I_Contact( #EstadoZona.ParoBlando_CBx )
      I_Contact( #F_EnvMens_Mx )
      I_Contact( #Mx_ET51 )
      I_Contact( #Mx_ET151 )
      I_Contact( #EstadoVI.Error_Mx )
      I_Contact( #Error_Tx )
      wire#w3
      S_SR(operand := #Mx_ET10, r1 := #Mx_ET11)
   END_RUNG
   RUNG wire#w1
      Contact( #Selec_M3_Entrada )
   END_RUNG wire#w2
   RUNG wire#powerrail
      Contact( #Mx_ET51 )
      Contact( #Mx_ET151 )
      wire#w4
      Contact( #Selec_M1_Entrada )
      wire#w5
      Contact( #Simultaneo_Mx )
      I_Contact( #EstadoVI.Descarga_Act )
      I_Contact( #MemoDesRemontando )
      I_Contact( #MemoRemontando )
   END_RUNG wire#w3
   RUNG wire#w4
      Contact( #Selec_M3_Entrada )
   END_RUNG wire#w5
   RUNG wire#powerrail
      Contact( #Mx_ET81 )
      I_Contact( #Mx_ET80 )
      wire#w6
      Contact( #Selec_M1_Entrada )
      wire#w7
      Contact( #MemoRemontando )
      I_Contact( #RH_FinMovimiento )
   END_RUNG wire#w3
   RUNG wire#w6
      Contact( #Selec_M3_Entrada )
   END_RUNG wire#w7
   // the same network as SCL:
   IF (#Mx_ET01 AND (#Selec_M1_Entrada OR #Selec_M3_Entrada) AND NOT #pHsMx_1 AND NOT #pHsMx_2 AND #AVTF_MEnt AND #PosTR_E1 AND #EstadoZona.Marcha_CBx AND NOT #EstadoZona.ParoBlando_CBx AND NOT #F_EnvMens_Mx AND NOT #Mx_ET51 AND NOT #Mx_ET151 AND NOT #EstadoVI.Error_Mx AND NOT #Error_Tx) OR (#Mx_ET51 AND #Mx_ET151 AND (#Selec_M1_Entrada OR #Selec_M3_Entrada) AND #Simultaneo_Mx AND NOT #EstadoVI.Descarga_Act AND NOT #MemoDesRemontando AND NOT #MemoRemontando) OR (#Mx_ET81 AND NOT #Mx_ET80 AND (#Selec_M1_Entrada OR #Selec_M3_Entrada) AND #MemoRemontando AND NOT #RH_FinMovimiento) THEN
       #Mx_ET10 := TRUE;   // SR flip-flop
   END_IF;
   IF #Mx_ET11 THEN #Mx_ET10 := FALSE; END_IF;
END_REGION

